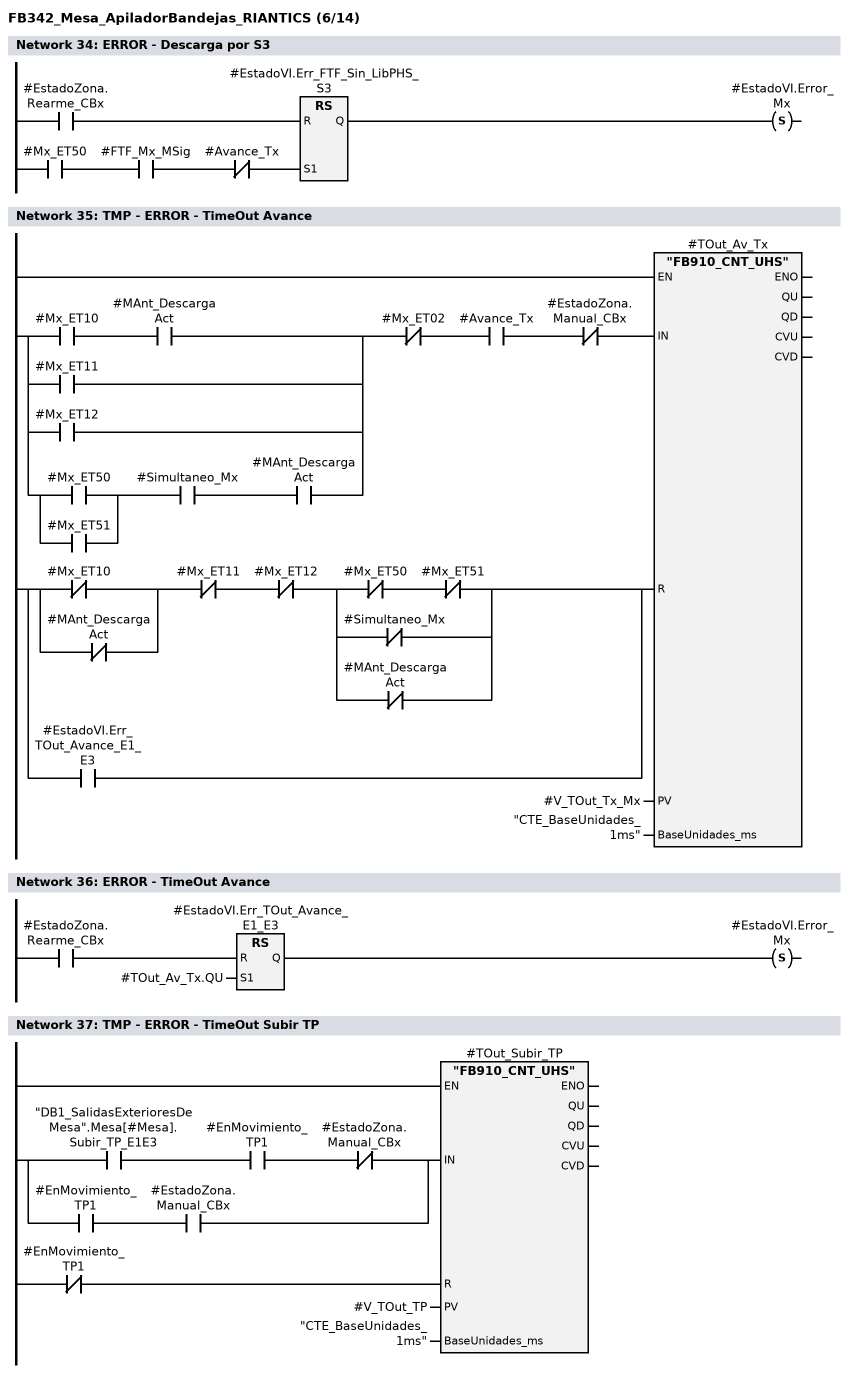
   RUNG wire#powerrail
      Contact( #EstadoZona.Rearme_CBx )
      S_RS(operand := #EstadoVI.Err_FTF_Sin_LibPHS_S3, s1 := wire#w1)
      S_Coil( #EstadoVI.Error_Mx )
   END_RUNG
   RUNG wire#powerrail
      Contact( #Mx_ET50 )
      Contact( #FTF_Mx_MSig )
      I_Contact( #Avance_Tx )
   END_RUNG wire#w1
   // the same network as SCL:
   IF #EstadoZona.Rearme_CBx THEN
       #EstadoVI.Err_FTF_Sin_LibPHS_S3 := FALSE;   // RS flip-flop
   END_IF;
   IF #Mx_ET50 AND #FTF_Mx_MSig AND NOT #Avance_Tx THEN #EstadoVI.Err_FTF_Sin_LibPHS_S3 := TRUE; END_IF;
   IF #EstadoVI.Err_FTF_Sin_LibPHS_S3 THEN #EstadoVI.Error_Mx := TRUE; END_IF;
END_REGION

REGION Network 35: TMP - ERROR - TimeOut Avance
   RUNG wire#powerrail
      #TOut_Av_Tx(IN := wire#w3, R := wire#w6, PV := #V_TOut_Tx_Mx, BaseUnidades_ms := "CTE_BaseUnidades_1ms", QU =>, QD =>, CVU =>, CVD =>)
   END_RUNG
   RUNG wire#powerrail
      Contact( #Mx_ET10 )
      Contact( #MAnt_DescargaAct )
      wire#w1
      I_Contact( #Mx_ET02 )
      Contact( #Avance_Tx )
      I_Contact( #EstadoZona.Manual_CBx )
   END_RUNG wire#w3
   RUNG wire#powerrail
      Contact( #Mx_ET11 )
   END_RUNG wire#w1
   RUNG wire#powerrail
      Contact( #Mx_ET12 )
   END_RUNG wire#w1
   RUNG wire#powerrail
      Contact( #Mx_ET50 )
      wire#w2
      Contact( #Simultaneo_Mx )
      Contact( #MAnt_DescargaAct )
   END_RUNG wire#w1
   RUNG wire#powerrail
      Contact( #Mx_ET51 )
   END_RUNG wire#w2
   RUNG wire#powerrail
      I_Contact( #Mx_ET10 )
      wire#w4
      I_Contact( #Mx_ET11 )
      I_Contact( #Mx_ET12 )
      wire#w5
      I_Contact( #Mx_ET50 )
      I_Contact( #Mx_ET51 )
   END_RUNG wire#w6
   RUNG wire#powerrail
      I_Contact( #MAnt_DescargaAct )
   END_RUNG wire#w4
   RUNG wire#w5
      I_Contact( #Simultaneo_Mx )
   END_RUNG wire#w6
   RUNG wire#w5
      I_Contact( #MAnt_DescargaAct )
   END_RUNG wire#w6
   RUNG wire#powerrail
      Contact( #EstadoVI.Err_TOut_Avance_E1_E3 )
   END_RUNG wire#w6
   // the same network as SCL:
   #TOut_Av_Tx(IN := ((#Mx_ET10 AND #MAnt_DescargaAct) OR #Mx_ET11 OR #Mx_ET12 OR ((#Mx_ET50 OR #Mx_ET51) AND #Simultaneo_Mx AND #MAnt_DescargaAct)) AND NOT #Mx_ET02 AND #Avance_Tx AND NOT #EstadoZona.Manual_CBx,   // "FB910_CNT_UHS"
               R := ((NOT #Mx_ET10 OR NOT #MAnt_DescargaAct) AND NOT #Mx_ET11 AND NOT #Mx_ET12 AND ((NOT #Mx_ET50 AND NOT #Mx_ET51) OR NOT #Simultaneo_Mx OR NOT #MAnt_DescargaAct)) OR #EstadoVI.Err_TOut_Avance_E1_E3,
               PV := #V_TOut_Tx_Mx,
               BaseUnidades_ms := "CTE_BaseUnidades_1ms");
END_REGION

REGION Network 36: ERROR - TimeOut Avance
   RUNG wire#powerrail
      Contact( #EstadoZona.Rearme_CBx )
      S_RS(operand := #EstadoVI.Err_TOut_Avance_E1_E3, s1 := #TOut_Av_Tx.QU)
      S_Coil( #EstadoVI.Error_Mx )
   END_RUNG
   // the same network as SCL:
   IF #EstadoZona.Rearme_CBx THEN
       #EstadoVI.Err_TOut_Avance_E1_E3 := FALSE;   // RS flip-flop
   END_IF;
   IF #TOut_Av_Tx.QU THEN #EstadoVI.Err_TOut_Avance_E1_E3 := TRUE; END_IF;
   IF #EstadoVI.Err_TOut_Avance_E1_E3 THEN #EstadoVI.Error_Mx := TRUE; END_IF;
END_REGION

REGION Network 37: TMP - ERROR - TimeOut Subir TP
   RUNG wire#powerrail
      #TOut_Subir_TP(IN := wire#w1, R := wire#w2, PV := #V_TOut_TP, BaseUnidades_ms := "CTE_BaseUnidades_1ms", QU =>, QD =>, CVU =>, CVD =>)
   END_RUNG
   RUNG wire#powerrail
      Contact( "DB1_SalidasExterioresDeMesa".Mesa[#Mesa].Subir_TP_E1E3 )
      Contact( #EnMovimiento_TP1 )
      I_Contact( #EstadoZona.Manual_CBx )
   END_RUNG wire#w1
   RUNG wire#powerrail
      Contact( #EnMovimiento_TP1 )
      Contact( #EstadoZona.Manual_CBx )
   END_RUNG wire#w1
   RUNG wire#powerrail
      I_Contact( #EnMovimiento_TP1 )
   END_RUNG wire#w2
   // the same network as SCL:
   #TOut_Subir_TP(IN := ("DB1_SalidasExterioresDeMesa".Mesa[#Mesa].Subir_TP_E1E3 AND #EnMovimiento_TP1 AND NOT #EstadoZona.Manual_CBx) OR (#EnMovimiento_TP1 AND #EstadoZona.Manual_CBx),   // "FB910_CNT_UHS"
                  R := NOT #EnMovimiento_TP1,
                  PV := #V_TOut_TP,
                  BaseUnidades_ms := "CTE_BaseUnidades_1ms");
END_REGION

REGION Network 38: ERROR - TimeOut Subir TP
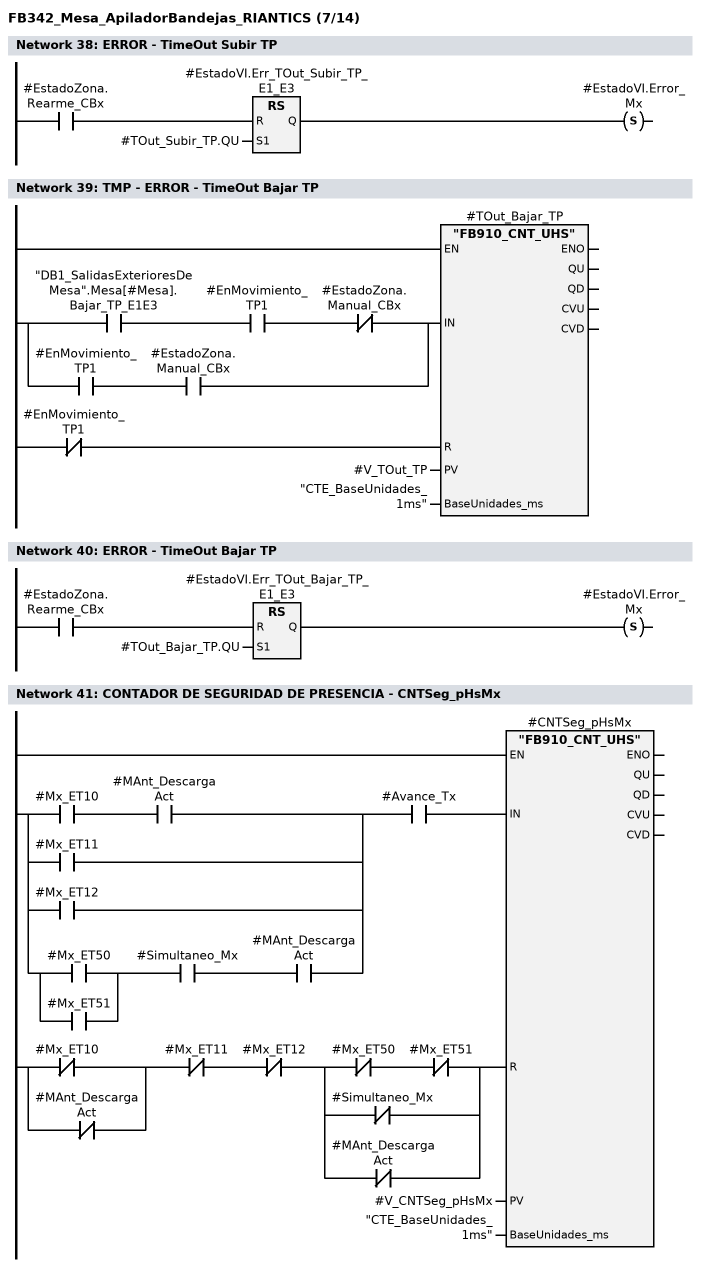
   RUNG wire#powerrail
      Contact( #EstadoZona.Rearme_CBx )
      S_RS(operand := #EstadoVI.Err_TOut_Subir_TP_E1_E3, s1 := #TOut_Subir_TP.QU)
      S_Coil( #EstadoVI.Error_Mx )
   END_RUNG
   // the same network as SCL:
   IF #EstadoZona.Rearme_CBx THEN
       #EstadoVI.Err_TOut_Subir_TP_E1_E3 := FALSE;   // RS flip-flop
   END_IF;
   IF #TOut_Subir_TP.QU THEN #EstadoVI.Err_TOut_Subir_TP_E1_E3 := TRUE; END_IF;
   IF #EstadoVI.Err_TOut_Subir_TP_E1_E3 THEN #EstadoVI.Error_Mx := TRUE; END_IF;
END_REGION

REGION Network 39: TMP - ERROR - TimeOut Bajar TP
   RUNG wire#powerrail
      #TOut_Bajar_TP(IN := wire#w1, R := wire#w2, PV := #V_TOut_TP, BaseUnidades_ms := "CTE_BaseUnidades_1ms", QU =>, QD =>, CVU =>, CVD =>)
   END_RUNG
   RUNG wire#powerrail
      Contact( "DB1_SalidasExterioresDeMesa".Mesa[#Mesa].Bajar_TP_E1E3 )
      Contact( #EnMovimiento_TP1 )
      I_Contact( #EstadoZona.Manual_CBx )
   END_RUNG wire#w1
   RUNG wire#powerrail
      Contact( #EnMovimiento_TP1 )
      Contact( #EstadoZona.Manual_CBx )
   END_RUNG wire#w1
   RUNG wire#powerrail
      I_Contact( #EnMovimiento_TP1 )
   END_RUNG wire#w2
   // the same network as SCL:
   #TOut_Bajar_TP(IN := ("DB1_SalidasExterioresDeMesa".Mesa[#Mesa].Bajar_TP_E1E3 AND #EnMovimiento_TP1 AND NOT #EstadoZona.Manual_CBx) OR (#EnMovimiento_TP1 AND #EstadoZona.Manual_CBx),   // "FB910_CNT_UHS"
                  R := NOT #EnMovimiento_TP1,
                  PV := #V_TOut_TP,
                  BaseUnidades_ms := "CTE_BaseUnidades_1ms");
END_REGION

REGION Network 40: ERROR - TimeOut Bajar TP
   RUNG wire#powerrail
      Contact( #EstadoZona.Rearme_CBx )
      S_RS(operand := #EstadoVI.Err_TOut_Bajar_TP_E1_E3, s1 := #TOut_Bajar_TP.QU)
      S_Coil( #EstadoVI.Error_Mx )
   END_RUNG
   // the same network as SCL:
   IF #EstadoZona.Rearme_CBx THEN
       #EstadoVI.Err_TOut_Bajar_TP_E1_E3 := FALSE;   // RS flip-flop
   END_IF;
   IF #TOut_Bajar_TP.QU THEN #EstadoVI.Err_TOut_Bajar_TP_E1_E3 := TRUE; END_IF;
   IF #EstadoVI.Err_TOut_Bajar_TP_E1_E3 THEN #EstadoVI.Error_Mx := TRUE; END_IF;
END_REGION

REGION Network 41: CONTADOR DE SEGURIDAD DE PRESENCIA - CNTSeg_pHsMx
   RUNG wire#powerrail
      #CNTSeg_pHsMx(IN := wire#w3, R := wire#w6, PV := #V_CNTSeg_pHsMx, BaseUnidades_ms := "CTE_BaseUnidades_1ms", QU =>, QD =>, CVU =>, CVD =>)
   END_RUNG
   RUNG wire#powerrail
      Contact( #Mx_ET10 )
      Contact( #MAnt_DescargaAct )
      wire#w1
      Contact( #Avance_Tx )
   END_RUNG wire#w3
   RUNG wire#powerrail
      Contact( #Mx_ET11 )
   END_RUNG wire#w1
   RUNG wire#powerrail
      Contact( #Mx_ET12 )
   END_RUNG wire#w1
   RUNG wire#powerrail
      Contact( #Mx_ET50 )
      wire#w2
      Contact( #Simultaneo_Mx )
      Contact( #MAnt_DescargaAct )
   END_RUNG wire#w1
   RUNG wire#powerrail
      Contact( #Mx_ET51 )
   END_RUNG wire#w2
   RUNG wire#powerrail
      I_Contact( #Mx_ET10 )
      wire#w4
      I_Contact( #Mx_ET11 )
      I_Contact( #Mx_ET12 )
      wire#w5
      I_Contact( #Mx_ET50 )
      I_Contact( #Mx_ET51 )
   END_RUNG wire#w6
   RUNG wire#powerrail
      I_Contact( #MAnt_DescargaAct )
   END_RUNG wire#w4
   RUNG wire#w5
      I_Contact( #Simultaneo_Mx )
   END_RUNG wire#w6
   RUNG wire#w5
      I_Contact( #MAnt_DescargaAct )
   END_RUNG wire#w6
   // the same network as SCL:
   #CNTSeg_pHsMx(IN := ((#Mx_ET10 AND #MAnt_DescargaAct) OR #Mx_ET11 OR #Mx_ET12 OR ((#Mx_ET50 OR #Mx_ET51) AND #Simultaneo_Mx AND #MAnt_DescargaAct)) AND #Avance_Tx,   // "FB910_CNT_UHS"
                 R := (NOT #Mx_ET10 OR NOT #MAnt_DescargaAct) AND NOT #Mx_ET11 AND NOT #Mx_ET12 AND ((NOT #Mx_ET50 AND NOT #Mx_ET51) OR NOT #Simultaneo_Mx OR NOT #MAnt_DescargaAct),
                 PV := #V_CNTSeg_pHsMx,
                 BaseUnidades_ms := "CTE_BaseUnidades_1ms");
END_REGION

REGION Network 42: CONTADOR DE PRESENCIA - CNT_pHsMx
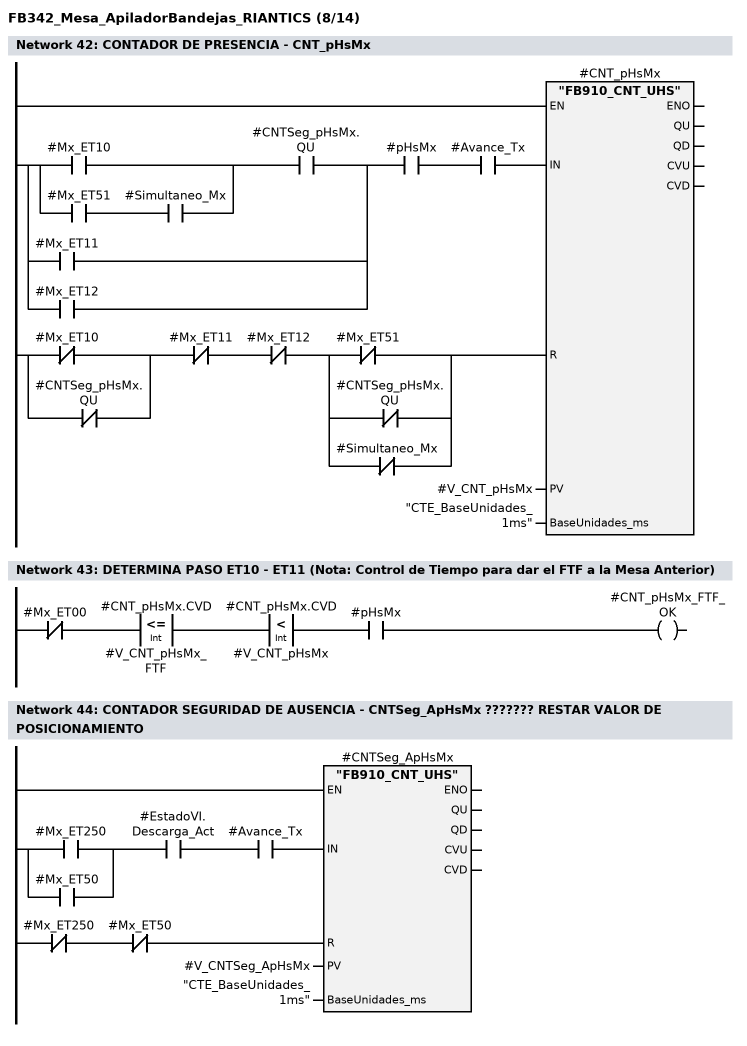
   RUNG wire#powerrail
      #CNT_pHsMx(IN := wire#w3, R := wire#w6, PV := #V_CNT_pHsMx, BaseUnidades_ms := "CTE_BaseUnidades_1ms", QU =>, QD =>, CVU =>, CVD =>)
   END_RUNG
   RUNG wire#powerrail
      Contact( #Mx_ET10 )
      wire#w1
      Contact( #CNTSeg_pHsMx.QU )
      wire#w2
      Contact( #pHsMx )
      Contact( #Avance_Tx )
   END_RUNG wire#w3
   RUNG wire#powerrail
      Contact( #Mx_ET51 )
      Contact( #Simultaneo_Mx )
   END_RUNG wire#w1
   RUNG wire#powerrail
      Contact( #Mx_ET11 )
   END_RUNG wire#w2
   RUNG wire#powerrail
      Contact( #Mx_ET12 )
   END_RUNG wire#w2
   RUNG wire#powerrail
      I_Contact( #Mx_ET10 )
      wire#w4
      I_Contact( #Mx_ET11 )
      I_Contact( #Mx_ET12 )
      wire#w5
      I_Contact( #Mx_ET51 )
   END_RUNG wire#w6
   RUNG wire#powerrail
      I_Contact( #CNTSeg_pHsMx.QU )
   END_RUNG wire#w4
   RUNG wire#w5
      I_Contact( #CNTSeg_pHsMx.QU )
   END_RUNG wire#w6
   RUNG wire#w5
      I_Contact( #Simultaneo_Mx )
   END_RUNG wire#w6
   // the same network as SCL:
   #CNT_pHsMx(IN := (((#Mx_ET10 OR (#Mx_ET51 AND #Simultaneo_Mx)) AND #CNTSeg_pHsMx.QU) OR #Mx_ET11 OR #Mx_ET12) AND #pHsMx AND #Avance_Tx,   // "FB910_CNT_UHS"
              R := (NOT #Mx_ET10 OR NOT #CNTSeg_pHsMx.QU) AND NOT #Mx_ET11 AND NOT #Mx_ET12 AND (NOT #Mx_ET51 OR NOT #CNTSeg_pHsMx.QU OR NOT #Simultaneo_Mx),
              PV := #V_CNT_pHsMx,
              BaseUnidades_ms := "CTE_BaseUnidades_1ms");
END_REGION

REGION Network 43: DETERMINA PASO ET10 - ET11 (Nota: Control de Tiempo para dar el FTF a la Mesa Anterior)
   RUNG wire#powerrail
      I_Contact( #Mx_ET00 )
      { S7_Templates := "SrcType := Int" } LE_Contact(in1 := #CNT_pHsMx.CVD, in2 := #V_CNT_pHsMx_FTF)
      { S7_Templates := "SrcType := Int" } LT_Contact(in1 := #CNT_pHsMx.CVD, in2 := #V_CNT_pHsMx)
      Contact( #pHsMx )
      Coil( #CNT_pHsMx_FTF_OK )
   END_RUNG
   // the same network as SCL:
   #CNT_pHsMx_FTF_OK := NOT #Mx_ET00 AND (#CNT_pHsMx.CVD <= #V_CNT_pHsMx_FTF) AND (#CNT_pHsMx.CVD < #V_CNT_pHsMx) AND #pHsMx;
END_REGION

REGION Network 44: CONTADOR SEGURIDAD DE AUSENCIA - CNTSeg_ApHsMx ??????? RESTAR VALOR DE POSICIONAMIENTO
   RUNG wire#powerrail
      #CNTSeg_ApHsMx(IN := wire#w2, R := wire#w3, PV := #V_CNTSeg_ApHsMx, BaseUnidades_ms := "CTE_BaseUnidades_1ms", QU =>, QD =>, CVU =>, CVD =>)
   END_RUNG
   RUNG wire#powerrail
      Contact( #Mx_ET250 )
      wire#w1
      Contact( #EstadoVI.Descarga_Act )
      Contact( #Avance_Tx )
   END_RUNG wire#w2
   RUNG wire#powerrail
      Contact( #Mx_ET50 )
   END_RUNG wire#w1
   RUNG wire#powerrail
      I_Contact( #Mx_ET250 )
      I_Contact( #Mx_ET50 )
   END_RUNG wire#w3
   // the same network as SCL:
   #CNTSeg_ApHsMx(IN := (#Mx_ET250 OR #Mx_ET50) AND #EstadoVI.Descarga_Act AND #Avance_Tx,   // "FB910_CNT_UHS"
                  R := NOT #Mx_ET250 AND NOT #Mx_ET50,
                  PV := #V_CNTSeg_ApHsMx,
                  BaseUnidades_ms := "CTE_BaseUnidades_1ms");
END_REGION

REGION Network 45: CONTADOR DE LA AUSENCIA - CNT_ApHsMX
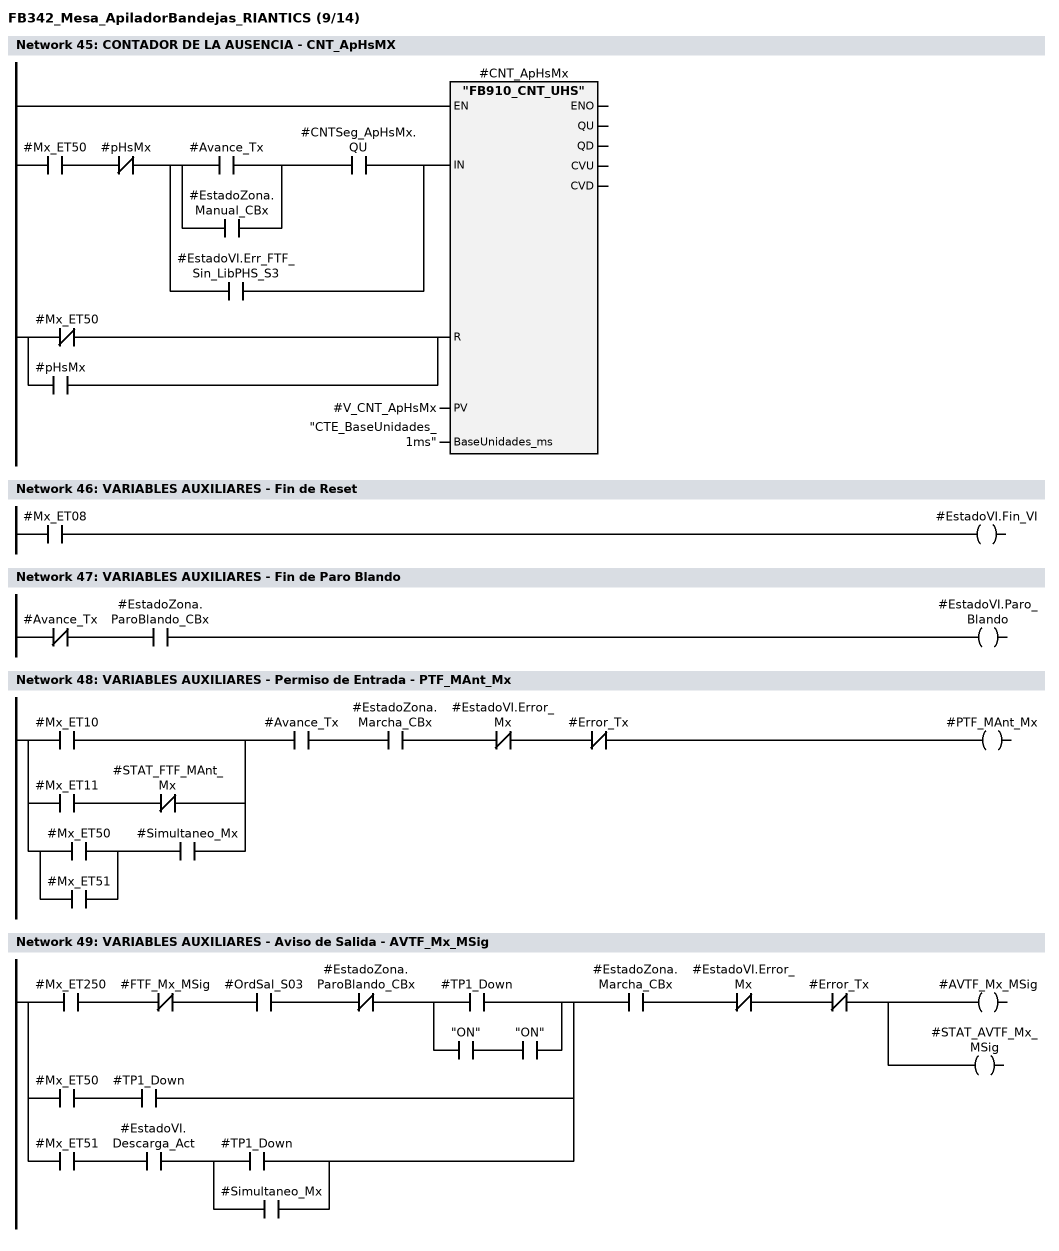
   RUNG wire#powerrail
      #CNT_ApHsMx(IN := wire#w3, R := wire#w4, PV := #V_CNT_ApHsMx, BaseUnidades_ms := "CTE_BaseUnidades_1ms", QU =>, QD =>, CVU =>, CVD =>)
   END_RUNG
   RUNG wire#powerrail
      Contact( #Mx_ET50 )
      I_Contact( #pHsMx )
      wire#w1
      Contact( #Avance_Tx )
      wire#w2
      Contact( #CNTSeg_ApHsMx.QU )
   END_RUNG wire#w3
   RUNG wire#w1
      Contact( #EstadoZona.Manual_CBx )
   END_RUNG wire#w2
   RUNG wire#w1
      Contact( #EstadoVI.Err_FTF_Sin_LibPHS_S3 )
   END_RUNG wire#w3
   RUNG wire#powerrail
      I_Contact( #Mx_ET50 )
   END_RUNG wire#w4
   RUNG wire#powerrail
      Contact( #pHsMx )
   END_RUNG wire#w4
   // the same network as SCL:
   #CNT_ApHsMx(IN := #Mx_ET50 AND NOT #pHsMx AND (((#Avance_Tx OR #EstadoZona.Manual_CBx) AND #CNTSeg_ApHsMx.QU) OR #EstadoVI.Err_FTF_Sin_LibPHS_S3),   // "FB910_CNT_UHS"
               R := NOT #Mx_ET50 OR #pHsMx,
               PV := #V_CNT_ApHsMx,
               BaseUnidades_ms := "CTE_BaseUnidades_1ms");
END_REGION

REGION Network 46: VARIABLES AUXILIARES - Fin de Reset
   RUNG wire#powerrail
      Contact( #Mx_ET08 )
      Coil( #EstadoVI.Fin_VI )
   END_RUNG
   // the same network as SCL:
   #EstadoVI.Fin_VI := #Mx_ET08;
END_REGION

REGION Network 47: VARIABLES AUXILIARES - Fin de Paro Blando
   RUNG wire#powerrail
      I_Contact( #Avance_Tx )
      Contact( #EstadoZona.ParoBlando_CBx )
      Coil( #EstadoVI.Paro_Blando )
   END_RUNG
   // the same network as SCL:
   #EstadoVI.Paro_Blando := NOT #Avance_Tx AND #EstadoZona.ParoBlando_CBx;
END_REGION

REGION Network 48: VARIABLES AUXILIARES - Permiso de Entrada - PTF_MAnt_Mx
   RUNG wire#powerrail
      Contact( #Mx_ET10 )
      wire#w1
      Contact( #Avance_Tx )
      Contact( #EstadoZona.Marcha_CBx )
      I_Contact( #EstadoVI.Error_Mx )
      I_Contact( #Error_Tx )
      Coil( #PTF_MAnt_Mx )
   END_RUNG
   RUNG wire#powerrail
      Contact( #Mx_ET11 )
      I_Contact( #STAT_FTF_MAnt_Mx )
   END_RUNG wire#w1
   RUNG wire#powerrail
      Contact( #Mx_ET50 )
      wire#w2
      Contact( #Simultaneo_Mx )
   END_RUNG wire#w1
   RUNG wire#powerrail
      Contact( #Mx_ET51 )
   END_RUNG wire#w2
   // the same network as SCL:
   #PTF_MAnt_Mx := (#Mx_ET10 OR (#Mx_ET11 AND NOT #STAT_FTF_MAnt_Mx) OR ((#Mx_ET50 OR #Mx_ET51) AND #Simultaneo_Mx)) AND #Avance_Tx AND #EstadoZona.Marcha_CBx AND NOT #EstadoVI.Error_Mx AND NOT #Error_Tx;
END_REGION

REGION Network 49: VARIABLES AUXILIARES - Aviso de Salida - AVTF_Mx_MSig
   RUNG wire#powerrail
      Contact( #Mx_ET250 )
      I_Contact( #FTF_Mx_MSig )
      Contact( #OrdSal_S03 )
      I_Contact( #EstadoZona.ParoBlando_CBx )
      wire#w1
      Contact( #TP1_Down )
      wire#w2
      Contact( #EstadoZona.Marcha_CBx )
      I_Contact( #EstadoVI.Error_Mx )
      I_Contact( #Error_Tx )
      wire#w4
      Coil( #AVTF_Mx_MSig )
   END_RUNG
   RUNG wire#w1
      Contact( "ON" )
      Contact( "ON" )
   END_RUNG wire#w2
   RUNG wire#powerrail
      Contact( #Mx_ET50 )
      Contact( #TP1_Down )
   END_RUNG wire#w2
   RUNG wire#powerrail
      Contact( #Mx_ET51 )
      Contact( #EstadoVI.Descarga_Act )
      wire#w3
      Contact( #TP1_Down )
   END_RUNG wire#w2
   RUNG wire#w3
      Contact( #Simultaneo_Mx )
   END_RUNG wire#w2
   RUNG wire#w4
      Coil( #STAT_AVTF_Mx_MSig )
   END_RUNG
   // the same network as SCL:
   #AVTF_Mx_MSig := ((#Mx_ET250 AND NOT #FTF_Mx_MSig AND #OrdSal_S03 AND NOT #EstadoZona.ParoBlando_CBx AND (#TP1_Down OR ("ON" AND "ON"))) OR (#Mx_ET50 AND #TP1_Down) OR (#Mx_ET51 AND #EstadoVI.Descarga_Act AND (#TP1_Down OR #Simultaneo_Mx))) AND #EstadoZona.Marcha_CBx AND NOT #EstadoVI.Error_Mx AND NOT #Error_Tx;
   #STAT_AVTF_Mx_MSig := #AVTF_Mx_MSig;
END_REGION

REGION Network 50: VARIABLES AUXILIARES - P_Mens_Mx_MSig (Nota: solo en ET51)
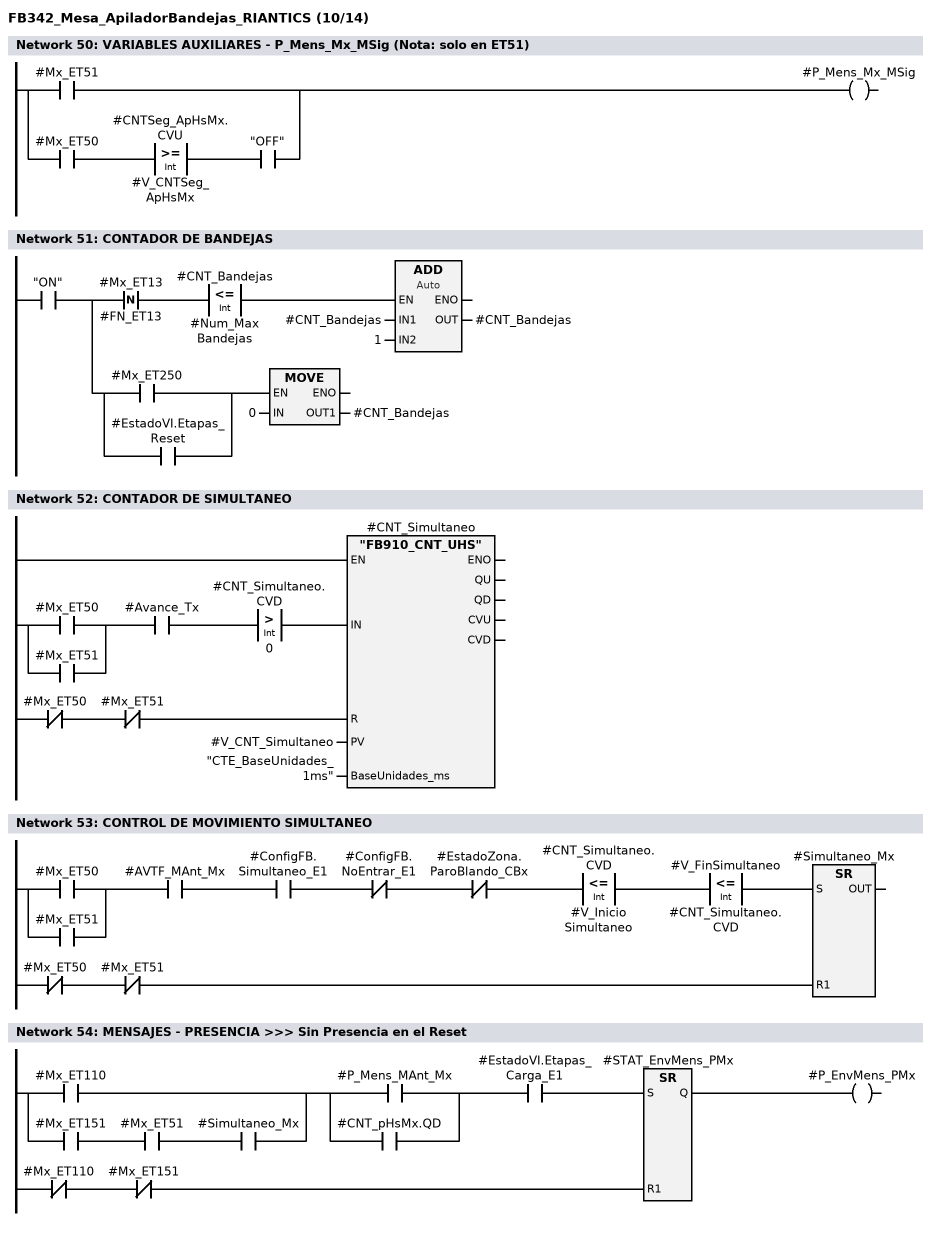
   RUNG wire#powerrail
      Contact( #Mx_ET51 )
      wire#w1
      Coil( #P_Mens_Mx_MSig )
   END_RUNG
   RUNG wire#powerrail
      Contact( #Mx_ET50 )
      { S7_Templates := "SrcType := Int" } GE_Contact(in1 := #CNTSeg_ApHsMx.CVU, in2 := #V_CNTSeg_ApHsMx)
      Contact( "OFF" )
   END_RUNG wire#w1
   // the same network as SCL:
   #P_Mens_Mx_MSig := #Mx_ET51 OR (#Mx_ET50 AND (#CNTSeg_ApHsMx.CVU >= #V_CNTSeg_ApHsMx) AND "OFF");
END_REGION

REGION Network 51: CONTADOR DE BANDEJAS
   RUNG wire#powerrail
      Contact( "ON" )
      wire#w1
      N_Contact(operand := #Mx_ET13, bit := #FN_ET13)
      { S7_Templates := "SrcType := Int" } LE_Contact(in1 := #CNT_Bandejas, in2 := #Num_MaxBandejas)
      Add(in1 := #CNT_Bandejas, in2 := 1, out => #CNT_Bandejas)
   END_RUNG
   RUNG wire#w1
      Contact( #Mx_ET250 )
      wire#w2
      Move(in := 0, out1 => #CNT_Bandejas)
   END_RUNG
   RUNG wire#w1
      Contact( #EstadoVI.Etapas_Reset )
   END_RUNG wire#w2
   // the same network as SCL:
   #_w1 := "ON" AND NOT #Mx_ET13 AND #FN_ET13;   // falling edge of #Mx_ET13
   #FN_ET13 := #Mx_ET13;
   IF #_w1 AND (#CNT_Bandejas <= #Num_MaxBandejas) THEN #CNT_Bandejas := #CNT_Bandejas + 1; END_IF;
   IF "ON" AND (#Mx_ET250 OR #EstadoVI.Etapas_Reset) THEN #CNT_Bandejas := 0; END_IF;
END_REGION

REGION Network 52: CONTADOR DE SIMULTANEO
   RUNG wire#powerrail
      #CNT_Simultaneo(IN := wire#w2, R := wire#w3, PV := #V_CNT_Simultaneo, BaseUnidades_ms := "CTE_BaseUnidades_1ms", QU =>, QD =>, CVU =>, CVD =>)
   END_RUNG
   RUNG wire#powerrail
      Contact( #Mx_ET50 )
      wire#w1
      Contact( #Avance_Tx )
      { S7_Templates := "SrcType := Int" } GT_Contact(in1 := #CNT_Simultaneo.CVD, in2 := 0)
   END_RUNG wire#w2
   RUNG wire#powerrail
      Contact( #Mx_ET51 )
   END_RUNG wire#w1
   RUNG wire#powerrail
      I_Contact( #Mx_ET50 )
      I_Contact( #Mx_ET51 )
   END_RUNG wire#w3
   // the same network as SCL:
   #CNT_Simultaneo(IN := (#Mx_ET50 OR #Mx_ET51) AND #Avance_Tx AND (#CNT_Simultaneo.CVD > 0),   // "FB910_CNT_UHS"
                   R := NOT #Mx_ET50 AND NOT #Mx_ET51,
                   PV := #V_CNT_Simultaneo,
                   BaseUnidades_ms := "CTE_BaseUnidades_1ms");
END_REGION

REGION Network 53: CONTROL DE MOVIMIENTO SIMULTANEO
   RUNG wire#powerrail
      Contact( #Mx_ET50 )
      wire#w1
      Contact( #AVTF_MAnt_Mx )
      Contact( #ConfigFB.Simultaneo_E1 )
      I_Contact( #ConfigFB.NoEntrar_E1 )
      I_Contact( #EstadoZona.ParoBlando_CBx )
      { S7_Templates := "SrcType := Int" } LE_Contact(in1 := #CNT_Simultaneo.CVD, in2 := #V_InicioSimultaneo)
      { S7_Templates := "SrcType := Int" } LE_Contact(in1 := #V_FinSimultaneo, in2 := #CNT_Simultaneo.CVD)
      S_SR(operand := #Simultaneo_Mx, r1 := wire#w2)
   END_RUNG
   RUNG wire#powerrail
      Contact( #Mx_ET51 )
   END_RUNG wire#w1
   RUNG wire#powerrail
      I_Contact( #Mx_ET50 )
      I_Contact( #Mx_ET51 )
   END_RUNG wire#w2
   // the same network as SCL:
   IF (#Mx_ET50 OR #Mx_ET51) AND #AVTF_MAnt_Mx AND #ConfigFB.Simultaneo_E1 AND NOT #ConfigFB.NoEntrar_E1 AND NOT #EstadoZona.ParoBlando_CBx AND (#CNT_Simultaneo.CVD <= #V_InicioSimultaneo) AND (#V_FinSimultaneo <= #CNT_Simultaneo.CVD) THEN
       #Simultaneo_Mx := TRUE;   // SR flip-flop
   END_IF;
   IF NOT #Mx_ET50 AND NOT #Mx_ET51 THEN #Simultaneo_Mx := FALSE; END_IF;
END_REGION

REGION Network 54: MENSAJES - PRESENCIA >>> Sin Presencia en el Reset
   RUNG wire#powerrail
      Contact( #Mx_ET110 )
      wire#w1
      Contact( #P_Mens_MAnt_Mx )
      wire#w2
      Contact( #EstadoVI.Etapas_Carga_E1 )
      S_SR(operand := #STAT_EnvMens_PMx, r1 := wire#w3)
      Coil( #P_EnvMens_PMx )
   END_RUNG
   RUNG wire#powerrail
      Contact( #Mx_ET151 )
      Contact( #Mx_ET51 )
      Contact( #Simultaneo_Mx )
   END_RUNG wire#w1
   RUNG wire#w1
      Contact( #CNT_pHsMx.QD )
   END_RUNG wire#w2
   RUNG wire#powerrail
      I_Contact( #Mx_ET110 )
      I_Contact( #Mx_ET151 )
   END_RUNG wire#w3
   // the same network as SCL:
   IF (#Mx_ET110 OR (#Mx_ET151 AND #Mx_ET51 AND #Simultaneo_Mx)) AND (#P_Mens_MAnt_Mx OR #CNT_pHsMx.QD) AND #EstadoVI.Etapas_Carga_E1 THEN
       #STAT_EnvMens_PMx := TRUE;   // SR flip-flop
   END_IF;
   IF NOT #Mx_ET110 AND NOT #Mx_ET151 THEN #STAT_EnvMens_PMx := FALSE; END_IF;
   #P_EnvMens_PMx := #STAT_EnvMens_PMx;
END_REGION

REGION Network 55: MENSAJES - PROTOCOLO INICIADO
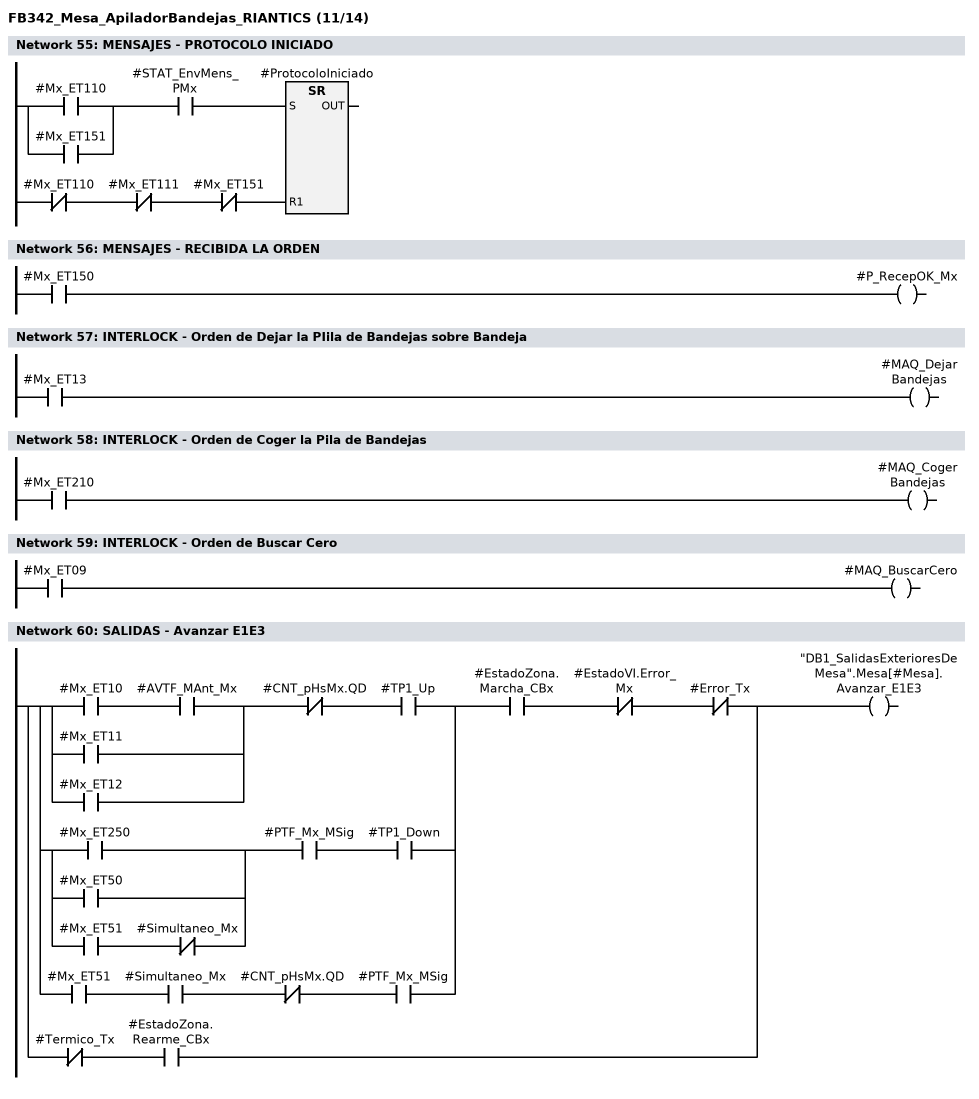
   RUNG wire#powerrail
      Contact( #Mx_ET110 )
      wire#w1
      Contact( #STAT_EnvMens_PMx )
      S_SR(operand := #ProtocoloIniciado, r1 := wire#w2)
   END_RUNG
   RUNG wire#powerrail
      Contact( #Mx_ET151 )
   END_RUNG wire#w1
   RUNG wire#powerrail
      I_Contact( #Mx_ET110 )
      I_Contact( #Mx_ET111 )
      I_Contact( #Mx_ET151 )
   END_RUNG wire#w2
   // the same network as SCL:
   IF (#Mx_ET110 OR #Mx_ET151) AND #STAT_EnvMens_PMx THEN
       #ProtocoloIniciado := TRUE;   // SR flip-flop
   END_IF;
   IF NOT #Mx_ET110 AND NOT #Mx_ET111 AND NOT #Mx_ET151 THEN #ProtocoloIniciado := FALSE; END_IF;
END_REGION

REGION Network 56: MENSAJES - RECIBIDA LA ORDEN
   RUNG wire#powerrail
      Contact( #Mx_ET150 )
      Coil( #P_RecepOK_Mx )
   END_RUNG
   // the same network as SCL:
   #P_RecepOK_Mx := #Mx_ET150;
END_REGION

REGION Network 57: INTERLOCK - Orden de Dejar la PIila de Bandejas sobre Bandeja
   RUNG wire#powerrail
      Contact( #Mx_ET13 )
      Coil( #MAQ_DejarBandejas )
   END_RUNG
   // the same network as SCL:
   #MAQ_DejarBandejas := #Mx_ET13;
END_REGION

REGION Network 58: INTERLOCK - Orden de Coger la Pila de Bandejas
   RUNG wire#powerrail
      Contact( #Mx_ET210 )
      Coil( #MAQ_CogerBandejas )
   END_RUNG
   // the same network as SCL:
   #MAQ_CogerBandejas := #Mx_ET210;
END_REGION

REGION Network 59: INTERLOCK - Orden de Buscar Cero
   RUNG wire#powerrail
      Contact( #Mx_ET09 )
      Coil( #MAQ_BuscarCero )
   END_RUNG
   // the same network as SCL:
   #MAQ_BuscarCero := #Mx_ET09;
END_REGION

REGION Network 60: SALIDAS - Avanzar E1E3
   RUNG wire#powerrail
      Contact( #Mx_ET10 )
      Contact( #AVTF_MAnt_Mx )
      wire#w1
      I_Contact( #CNT_pHsMx.QD )
      Contact( #TP1_Up )
      wire#w2
      Contact( #EstadoZona.Marcha_CBx )
      I_Contact( #EstadoVI.Error_Mx )
      I_Contact( #Error_Tx )
      wire#w4
      Coil( "DB1_SalidasExterioresDeMesa".Mesa[#Mesa].Avanzar_E1E3 )
   END_RUNG
   RUNG wire#powerrail
      Contact( #Mx_ET11 )
   END_RUNG wire#w1
   RUNG wire#powerrail
      Contact( #Mx_ET12 )
   END_RUNG wire#w1
   RUNG wire#powerrail
      Contact( #Mx_ET250 )
      wire#w3
      Contact( #PTF_Mx_MSig )
      Contact( #TP1_Down )
   END_RUNG wire#w2
   RUNG wire#powerrail
      Contact( #Mx_ET50 )
   END_RUNG wire#w3
   RUNG wire#powerrail
      Contact( #Mx_ET51 )
      I_Contact( #Simultaneo_Mx )
   END_RUNG wire#w3
   RUNG wire#powerrail
      Contact( #Mx_ET51 )
      Contact( #Simultaneo_Mx )
      I_Contact( #CNT_pHsMx.QD )
      Contact( #PTF_Mx_MSig )
   END_RUNG wire#w2
   RUNG wire#powerrail
      I_Contact( #Termico_Tx )
      Contact( #EstadoZona.Rearme_CBx )
   END_RUNG wire#w4
   // the same network as SCL:
   "DB1_SalidasExterioresDeMesa".Mesa[#Mesa].Avanzar_E1E3 := (((((#Mx_ET10 AND #AVTF_MAnt_Mx) OR #Mx_ET11 OR #Mx_ET12) AND NOT #CNT_pHsMx.QD AND #TP1_Up) OR ((#Mx_ET250 OR #Mx_ET50 OR (#Mx_ET51 AND NOT #Simultaneo_Mx)) AND #PTF_Mx_MSig AND #TP1_Down) OR (#Mx_ET51 AND #Simultaneo_Mx AND NOT #CNT_pHsMx.QD AND #PTF_Mx_MSig)) AND #EstadoZona.Marcha_CBx AND NOT #EstadoVI.Error_Mx AND NOT #Error_Tx) OR (NOT #Termico_Tx AND #EstadoZona.Rearme_CBx);
END_REGION

REGION Network 61: SALIDAS - Parar E1E3
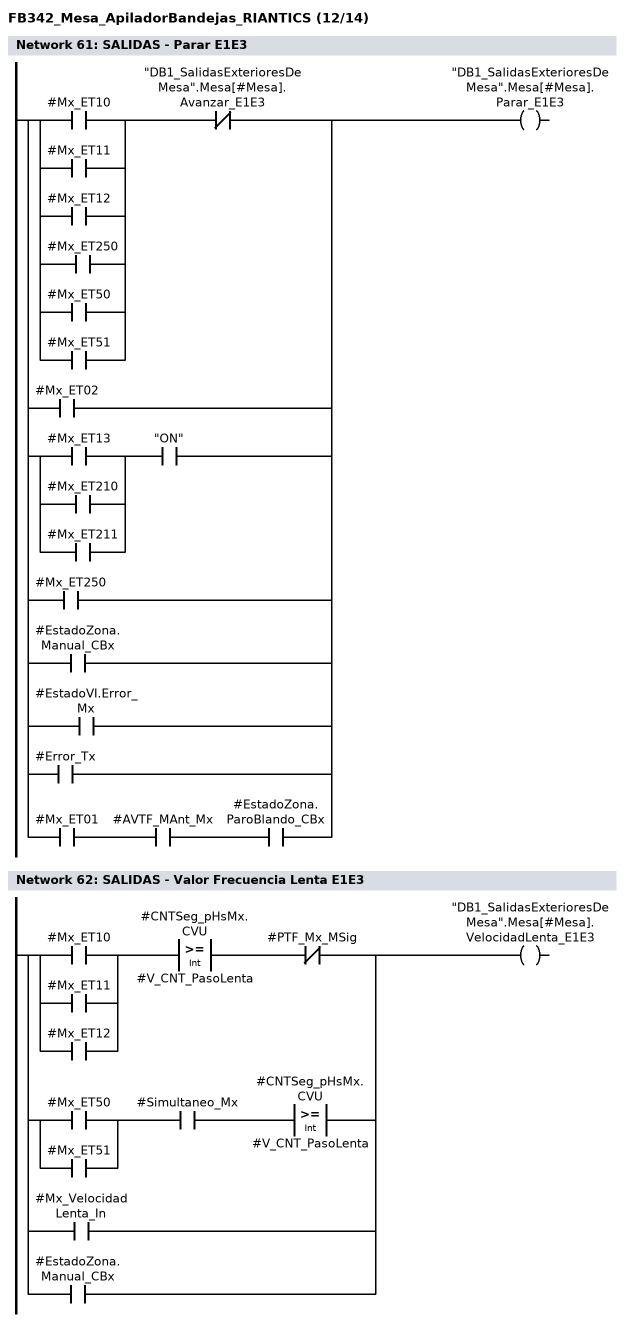
   RUNG wire#powerrail
      Contact( #Mx_ET10 )
      wire#w1
      I_Contact( "DB1_SalidasExterioresDeMesa".Mesa[#Mesa].Avanzar_E1E3 )
      wire#w2
      Coil( "DB1_SalidasExterioresDeMesa".Mesa[#Mesa].Parar_E1E3 )
   END_RUNG
   RUNG wire#powerrail
      Contact( #Mx_ET11 )
   END_RUNG wire#w1
   RUNG wire#powerrail
      Contact( #Mx_ET12 )
   END_RUNG wire#w1
   RUNG wire#powerrail
      Contact( #Mx_ET250 )
   END_RUNG wire#w1
   RUNG wire#powerrail
      Contact( #Mx_ET50 )
   END_RUNG wire#w1
   RUNG wire#powerrail
      Contact( #Mx_ET51 )
   END_RUNG wire#w1
   RUNG wire#powerrail
      Contact( #Mx_ET02 )
   END_RUNG wire#w2
   RUNG wire#powerrail
      Contact( #Mx_ET13 )
      wire#w3
      Contact( "ON" )
   END_RUNG wire#w2
   RUNG wire#powerrail
      Contact( #Mx_ET210 )
   END_RUNG wire#w3
   RUNG wire#powerrail
      Contact( #Mx_ET211 )
   END_RUNG wire#w3
   RUNG wire#powerrail
      Contact( #Mx_ET250 )
   END_RUNG wire#w2
   RUNG wire#powerrail
      Contact( #EstadoZona.Manual_CBx )
   END_RUNG wire#w2
   RUNG wire#powerrail
      Contact( #EstadoVI.Error_Mx )
   END_RUNG wire#w2
   RUNG wire#powerrail
      Contact( #Error_Tx )
   END_RUNG wire#w2
   RUNG wire#powerrail
      Contact( #Mx_ET01 )
      Contact( #AVTF_MAnt_Mx )
      Contact( #EstadoZona.ParoBlando_CBx )
   END_RUNG wire#w2
   // the same network as SCL:
   "DB1_SalidasExterioresDeMesa".Mesa[#Mesa].Parar_E1E3 := ((#Mx_ET10 OR #Mx_ET11 OR #Mx_ET12 OR #Mx_ET250 OR #Mx_ET50 OR #Mx_ET51) AND NOT "DB1_SalidasExterioresDeMesa".Mesa[#Mesa].Avanzar_E1E3) OR #Mx_ET02 OR ((#Mx_ET13 OR #Mx_ET210 OR #Mx_ET211) AND "ON") OR #Mx_ET250 OR #EstadoZona.Manual_CBx OR #EstadoVI.Error_Mx OR #Error_Tx OR (#Mx_ET01 AND #AVTF_MAnt_Mx AND #EstadoZona.ParoBlando_CBx);
END_REGION

REGION Network 62: SALIDAS - Valor Frecuencia Lenta E1E3
   RUNG wire#powerrail
      Contact( #Mx_ET10 )
      wire#w1
      { S7_Templates := "SrcType := Int" } GE_Contact(in1 := #CNTSeg_pHsMx.CVU, in2 := #V_CNT_PasoLenta)
      I_Contact( #PTF_Mx_MSig )
      wire#w2
      Coil( "DB1_SalidasExterioresDeMesa".Mesa[#Mesa].VelocidadLenta_E1E3 )
   END_RUNG
   RUNG wire#powerrail
      Contact( #Mx_ET11 )
   END_RUNG wire#w1
   RUNG wire#powerrail
      Contact( #Mx_ET12 )
   END_RUNG wire#w1
   RUNG wire#powerrail
      Contact( #Mx_ET50 )
      wire#w3
      Contact( #Simultaneo_Mx )
      { S7_Templates := "SrcType := Int" } GE_Contact(in1 := #CNTSeg_pHsMx.CVU, in2 := #V_CNT_PasoLenta)
   END_RUNG wire#w2
   RUNG wire#powerrail
      Contact( #Mx_ET51 )
   END_RUNG wire#w3
   RUNG wire#powerrail
      Contact( #Mx_VelocidadLenta_In )
   END_RUNG wire#w2
   RUNG wire#powerrail
      Contact( #EstadoZona.Manual_CBx )
   END_RUNG wire#w2
   // the same network as SCL:
   "DB1_SalidasExterioresDeMesa".Mesa[#Mesa].VelocidadLenta_E1E3 := ((#Mx_ET10 OR #Mx_ET11 OR #Mx_ET12) AND (#CNTSeg_pHsMx.CVU >= #V_CNT_PasoLenta) AND NOT #PTF_Mx_MSig) OR ((#Mx_ET50 OR #Mx_ET51) AND #Simultaneo_Mx AND (#CNTSeg_pHsMx.CVU >= #V_CNT_PasoLenta)) OR #Mx_VelocidadLenta_In OR #EstadoZona.Manual_CBx;
END_REGION

REGION Network 63: SALIDAS - Bajar Tope TP1 NOTA: Tope E1 >> S3
   // ACTIVAREMOS EL TOPE SOLO CUANDO HAYA YA PERMISO DE SALIDA. ESTO PARA LAS MAQUINAS QUE TENGAN ACTUADOR ELECTRICO. EN UNO NEUMATICO SE PUEDEN QUITAR LOS DOS OFFS
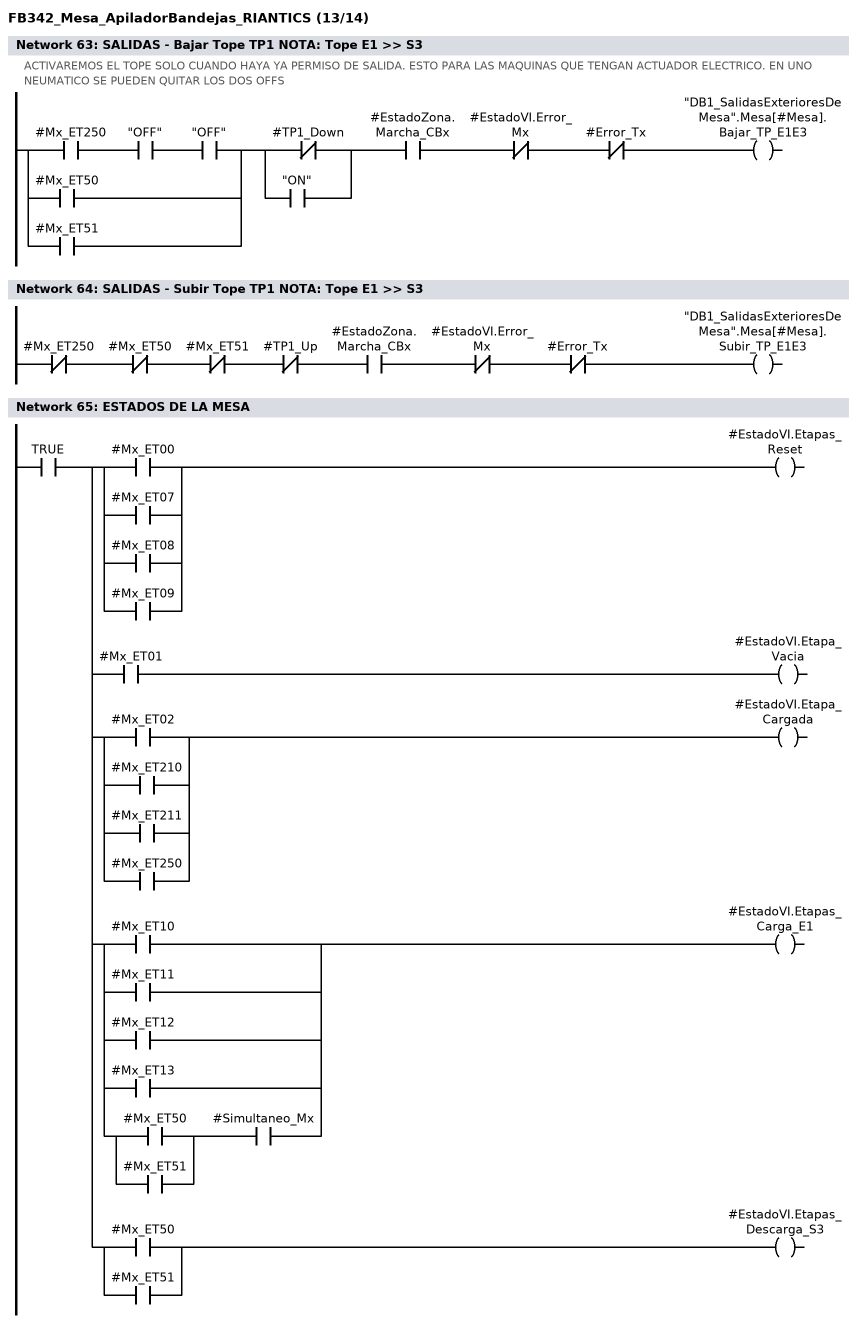
   RUNG wire#powerrail
      Contact( #Mx_ET250 )
      Contact( "OFF" )
      Contact( "OFF" )
      wire#w1
      I_Contact( #TP1_Down )
      wire#w2
      Contact( #EstadoZona.Marcha_CBx )
      I_Contact( #EstadoVI.Error_Mx )
      I_Contact( #Error_Tx )
      Coil( "DB1_SalidasExterioresDeMesa".Mesa[#Mesa].Bajar_TP_E1E3 )
   END_RUNG
   RUNG wire#powerrail
      Contact( #Mx_ET50 )
   END_RUNG wire#w1
   RUNG wire#powerrail
      Contact( #Mx_ET51 )
   END_RUNG wire#w1
   RUNG wire#w1
      Contact( "ON" )
   END_RUNG wire#w2
   // the same network as SCL:
   "DB1_SalidasExterioresDeMesa".Mesa[#Mesa].Bajar_TP_E1E3 := ((#Mx_ET250 AND "OFF" AND "OFF") OR #Mx_ET50 OR #Mx_ET51) AND (NOT #TP1_Down OR "ON") AND #EstadoZona.Marcha_CBx AND NOT #EstadoVI.Error_Mx AND NOT #Error_Tx;
END_REGION

REGION Network 64: SALIDAS - Subir Tope TP1 NOTA: Tope E1 >> S3
   RUNG wire#powerrail
      I_Contact( #Mx_ET250 )
      I_Contact( #Mx_ET50 )
      I_Contact( #Mx_ET51 )
      I_Contact( #TP1_Up )
      Contact( #EstadoZona.Marcha_CBx )
      I_Contact( #EstadoVI.Error_Mx )
      I_Contact( #Error_Tx )
      Coil( "DB1_SalidasExterioresDeMesa".Mesa[#Mesa].Subir_TP_E1E3 )
   END_RUNG
   // the same network as SCL:
   "DB1_SalidasExterioresDeMesa".Mesa[#Mesa].Subir_TP_E1E3 := NOT #Mx_ET250 AND NOT #Mx_ET50 AND NOT #Mx_ET51 AND NOT #TP1_Up AND #EstadoZona.Marcha_CBx AND NOT #EstadoVI.Error_Mx AND NOT #Error_Tx;
END_REGION

REGION Network 65: ESTADOS DE LA MESA
   RUNG wire#powerrail
      Contact( TRUE )
      wire#w1
      Contact( #Mx_ET00 )
      wire#w2
      Coil( #EstadoVI.Etapas_Reset )
   END_RUNG
   RUNG wire#w1
      Contact( #Mx_ET07 )
   END_RUNG wire#w2
   RUNG wire#w1
      Contact( #Mx_ET08 )
   END_RUNG wire#w2
   RUNG wire#w1
      Contact( #Mx_ET09 )
   END_RUNG wire#w2
   RUNG wire#w1
      Contact( #Mx_ET01 )
      Coil( #EstadoVI.Etapa_Vacia )
   END_RUNG
   RUNG wire#w1
      Contact( #Mx_ET02 )
      wire#w3
      Coil( #EstadoVI.Etapa_Cargada )
   END_RUNG
   RUNG wire#w1
      Contact( #Mx_ET210 )
   END_RUNG wire#w3
   RUNG wire#w1
      Contact( #Mx_ET211 )
   END_RUNG wire#w3
   RUNG wire#w1
      Contact( #Mx_ET250 )
   END_RUNG wire#w3
   RUNG wire#w1
      Contact( #Mx_ET10 )
      wire#w4
      Coil( #EstadoVI.Etapas_Carga_E1 )
   END_RUNG
   RUNG wire#w1
      Contact( #Mx_ET11 )
   END_RUNG wire#w4
   RUNG wire#w1
      Contact( #Mx_ET12 )
   END_RUNG wire#w4
   RUNG wire#w1
      Contact( #Mx_ET13 )
   END_RUNG wire#w4
   RUNG wire#w1
      Contact( #Mx_ET50 )
      wire#w5
      Contact( #Simultaneo_Mx )
   END_RUNG wire#w4
   RUNG wire#w1
      Contact( #Mx_ET51 )
   END_RUNG wire#w5
   RUNG wire#w1
      Contact( #Mx_ET50 )
      wire#w6
      Coil( #EstadoVI.Etapas_Descarga_S3 )
   END_RUNG
   RUNG wire#w1
      Contact( #Mx_ET51 )
   END_RUNG wire#w6
   // the same network as SCL:
   #EstadoVI.Etapas_Reset := TRUE AND (#Mx_ET00 OR #Mx_ET07 OR #Mx_ET08 OR #Mx_ET09);
   #EstadoVI.Etapa_Vacia := TRUE AND #Mx_ET01;
   #EstadoVI.Etapa_Cargada := TRUE AND (#Mx_ET02 OR #Mx_ET210 OR #Mx_ET211 OR #Mx_ET250);
   #EstadoVI.Etapas_Carga_E1 := TRUE AND (#Mx_ET10 OR #Mx_ET11 OR #Mx_ET12 OR #Mx_ET13 OR ((#Mx_ET50 OR #Mx_ET51) AND #Simultaneo_Mx));
   #EstadoVI.Etapas_Descarga_S3 := TRUE AND (#Mx_ET50 OR #Mx_ET51);
END_REGION

REGION Network 66: ENTRADAS DE LA MESA
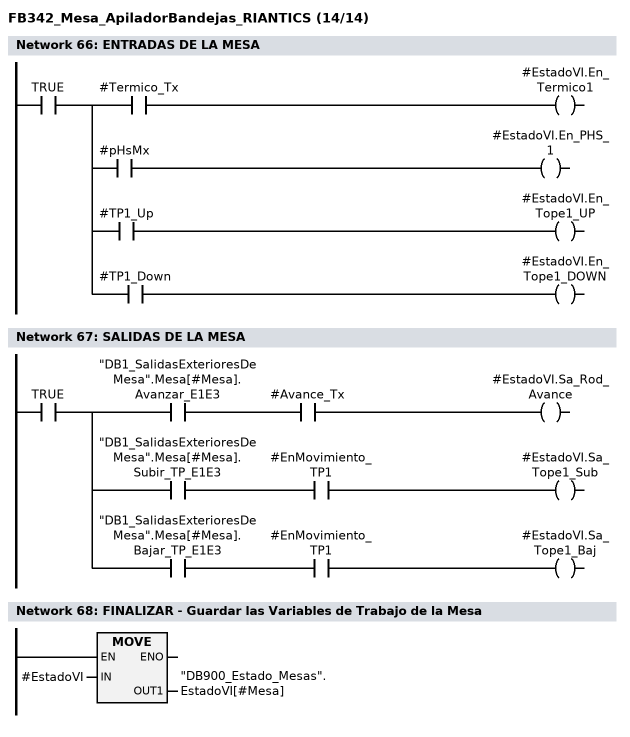
   RUNG wire#powerrail
      Contact( TRUE )
      wire#w1
      Contact( #Termico_Tx )
      Coil( #EstadoVI.En_Termico1 )
   END_RUNG
   RUNG wire#w1
      Contact( #pHsMx )
      Coil( #EstadoVI.En_PHS_1 )
   END_RUNG
   RUNG wire#w1
      Contact( #TP1_Up )
      Coil( #EstadoVI.En_Tope1_UP )
   END_RUNG
   RUNG wire#w1
      Contact( #TP1_Down )
      Coil( #EstadoVI.En_Tope1_DOWN )
   END_RUNG
   // the same network as SCL:
   #EstadoVI.En_Termico1 := TRUE AND #Termico_Tx;
   #EstadoVI.En_PHS_1 := TRUE AND #pHsMx;
   #EstadoVI.En_Tope1_UP := TRUE AND #TP1_Up;
   #EstadoVI.En_Tope1_DOWN := TRUE AND #TP1_Down;
END_REGION

REGION Network 67: SALIDAS DE LA MESA
   RUNG wire#powerrail
      Contact( TRUE )
      wire#w1
      Contact( "DB1_SalidasExterioresDeMesa".Mesa[#Mesa].Avanzar_E1E3 )
      Contact( #Avance_Tx )
      Coil( #EstadoVI.Sa_Rod_Avance )
   END_RUNG
   RUNG wire#w1
      Contact( "DB1_SalidasExterioresDeMesa".Mesa[#Mesa].Subir_TP_E1E3 )
      Contact( #EnMovimiento_TP1 )
      Coil( #EstadoVI.Sa_Tope1_Sub )
   END_RUNG
   RUNG wire#w1
      Contact( "DB1_SalidasExterioresDeMesa".Mesa[#Mesa].Bajar_TP_E1E3 )
      Contact( #EnMovimiento_TP1 )
      Coil( #EstadoVI.Sa_Tope1_Baj )
   END_RUNG
   // the same network as SCL:
   #EstadoVI.Sa_Rod_Avance := TRUE AND "DB1_SalidasExterioresDeMesa".Mesa[#Mesa].Avanzar_E1E3 AND #Avance_Tx;
   #EstadoVI.Sa_Tope1_Sub := TRUE AND "DB1_SalidasExterioresDeMesa".Mesa[#Mesa].Subir_TP_E1E3 AND #EnMovimiento_TP1;
   #EstadoVI.Sa_Tope1_Baj := TRUE AND "DB1_SalidasExterioresDeMesa".Mesa[#Mesa].Bajar_TP_E1E3 AND #EnMovimiento_TP1;
END_REGION

REGION Network 68: FINALIZAR - Guardar las Variables de Trabajo de la Mesa
   RUNG wire#powerrail
      Move(in := #EstadoVI, out1 => "DB900_Estado_Mesas".EstadoVI[#Mesa])
   END_RUNG
   // the same network as SCL:
   "DB900_Estado_Mesas".EstadoVI[#Mesa] := #EstadoVI;
END_REGION
END_FUNCTION_BLOCK

FUNCTION_BLOCK "FB343_ApiladorBandejas_RIANTICS"   // FB343, LAD
{ S7_Optimized_Access := 'FALSE' }
// stored: AutoNumber false, SetENOAutomatically false
   VAR_INPUT
      Maquina : UInt;   // Numero de Maquina (Mesa)
      Error_Tx : Bool;   // Error en el Tx
      EnTension : Bool;   // Existe Tension en la Maquina
      MAQx_Desabilitada : Bool;   // Config MAQ. >>> DesHabilitada
      Termico_Elevacion : Bool;   // Termico de la Elevacion
      Pos_DW : Bool;   // Posición Baja del Apilador
      Pos_mid_DW : Bool;
      Pos_mid_UP : Bool;
      Pos_UP : Bool;   // Posición Alta del Apilador
      EnMovimiento_Elevacion : Bool;   // En Movineto la Elevacion
      CargaSuelta : Bool;   // Carga Suelta en el Apilador
      CargaCogida : Bool;   // Carga Cogida en el Apilador
      EnMovimiento_Horquillado : Bool;   // En Movimiento el Hoquillado
      MAQ_DejarBandejas : Bool;   // Interlock >> Dejar Bandejas
      MAQ_CogerBandejas : Bool;   // Interlock >> Coger Bandejas
      MAQ_BuscarCero : Bool;   // Interlock >> Buscar Cero
      CogiendoDerecha : Bool;
      CogiendoIzquierda : Bool;
      DejandoDerecha : Bool;
      DejandoIzquierda : Bool;
      V_TOut_Elevacion : Int := 2000;   // TimeOut del Mov. de Elevacion
      V_TOut_Horquillado : Int := 2000;   // TimeOut del Mov. de Horquillado
   END_VAR
   VAR_OUTPUT
      MAQ_DejadasBandejas : Bool;   // Interlock >> Bandejas Dejadas
      MAQ_CojidasBandejas : Bool;   // Interlock >> Bandejas Cogidas
      MAQ_CeroEncontrado : Bool;   // Interlock >> Bandejas
   END_VAR
   VAR
      AP_ET00 : Bool;
      AP_ET01 : Bool;
      AP_ET100 : Bool;
      AP_ET101 : Bool;
      AP_ET102 : Bool;
      AP_ET103 : Bool;
      AP_ET104 : Bool;
      AP_ET50 : Bool;
      AP_ET51 : Bool;
      AP_ET52 : Bool;
      AP_ET53 : Bool;
      AP_ET54 : Bool;
      AP_ET60 : Bool;
      AP_ET61 : Bool;
      AP_ET62 : Bool;
      AP_ET63 : Bool;
      AP_ET64 : Bool;
      MA_Motor_Elev : Bool;
      MA_Slow_Velocity : Bool;
      MA_CogerCarga : Bool;   // Cerrar Cilindros para coger la pila
      MA_DejarCarga : Bool;   // Abrir Cilindros para dejas la pila
      TMP_ReposoCargaSuelta { S7_SetPoint := 'True'} : TON_TIME;
      TMP_EnTension { S7_SetPoint := 'True'} : "FB910_CNT_UHS";
      TOut_Elevacion { S7_SetPoint := 'True'} : "FB910_CNT_UHS";
      TOut_Horquillado { S7_SetPoint := 'True'} : "FB910_CNT_UHS";
      Manual : "MoviManualMaquina_Apilador_bandejas";
   END_VAR
   VAR_TEMP
      EstadoZona : "EstadoZona";   // Estado de Zona de la Mesa
      EstadoMAQ : "EstadoMaquina_Apilador_bandejas";   // Estado del Vehiculo Inteliguente de la Maquina
      Aux_ET00 : Bool;
   END_VAR
BEGIN

REGION Network 1: INICIALIZAR - Recoger las Variables de Estado de la Maquina
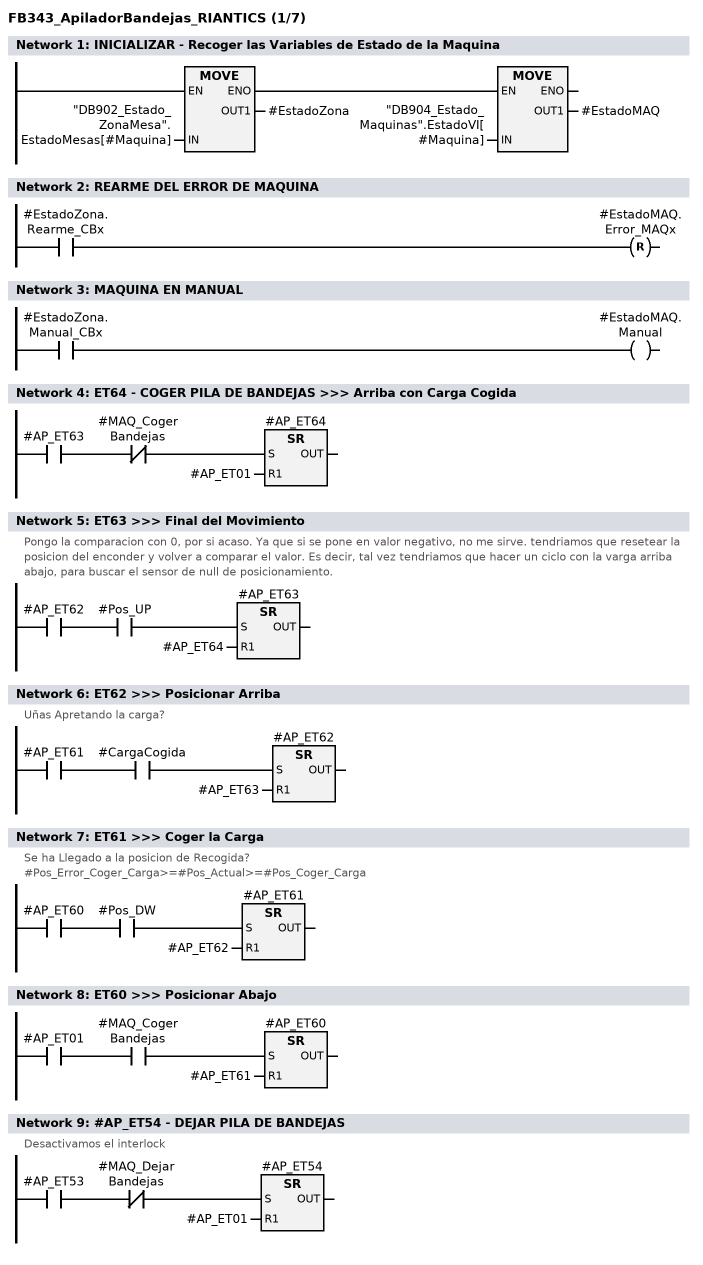
   RUNG wire#powerrail
      Move(in := "DB902_Estado_ZonaMesa".EstadoMesas[#Maquina], out1 => #EstadoZona)
      Move(in := "DB904_Estado_Maquinas".EstadoVI[#Maquina], out1 => #EstadoMAQ)
   END_RUNG
   // the same network as SCL:
   #EstadoZona := "DB902_Estado_ZonaMesa".EstadoMesas[#Maquina];
   #EstadoMAQ := "DB904_Estado_Maquinas".EstadoVI[#Maquina];
END_REGION

REGION Network 2: REARME DEL ERROR DE MAQUINA
   RUNG wire#powerrail
      Contact( #EstadoZona.Rearme_CBx )
      R_Coil( #EstadoMAQ.Error_MAQx )
   END_RUNG
   // the same network as SCL:
   IF #EstadoZona.Rearme_CBx THEN #EstadoMAQ.Error_MAQx := FALSE; END_IF;
END_REGION

REGION Network 3: MAQUINA EN MANUAL
   RUNG wire#powerrail
      Contact( #EstadoZona.Manual_CBx )
      Coil( #EstadoMAQ.Manual )
   END_RUNG
   // the same network as SCL:
   #EstadoMAQ.Manual := #EstadoZona.Manual_CBx;
END_REGION

REGION Network 4: ET64 - COGER PILA DE BANDEJAS >>> Arriba con Carga Cogida
   RUNG wire#powerrail
      Contact( #AP_ET63 )
      I_Contact( #MAQ_CogerBandejas )
      S_SR(operand := #AP_ET64, r1 := #AP_ET01)
   END_RUNG
   // the same network as SCL:
   IF #AP_ET63 AND NOT #MAQ_CogerBandejas THEN
       #AP_ET64 := TRUE;   // SR flip-flop
   END_IF;
   IF #AP_ET01 THEN #AP_ET64 := FALSE; END_IF;
END_REGION

REGION Network 5: ET63 >>> Final del Movimiento
   // Pongo la comparacion con 0, por si acaso. Ya que si se pone en valor negativo, no me sirve. tendriamos que resetear la posicion del enconder y volver a comparar el valor. Es decir, tal vez tendriamos que hacer un ciclo con la varga arriba abajo, para buscar el sensor de null de posicionamiento.
   RUNG wire#powerrail
      Contact( #AP_ET62 )
      Contact( #Pos_UP )
      S_SR(operand := #AP_ET63, r1 := #AP_ET64)
   END_RUNG
   // the same network as SCL:
   IF #AP_ET62 AND #Pos_UP THEN
       #AP_ET63 := TRUE;   // SR flip-flop
   END_IF;
   IF #AP_ET64 THEN #AP_ET63 := FALSE; END_IF;
END_REGION

REGION Network 6: ET62 >>> Posicionar Arriba
   // Uñas Apretando la carga?
   RUNG wire#powerrail
      Contact( #AP_ET61 )
      Contact( #CargaCogida )
      S_SR(operand := #AP_ET62, r1 := #AP_ET63)
   END_RUNG
   // the same network as SCL:
   IF #AP_ET61 AND #CargaCogida THEN
       #AP_ET62 := TRUE;   // SR flip-flop
   END_IF;
   IF #AP_ET63 THEN #AP_ET62 := FALSE; END_IF;
END_REGION

REGION Network 7: ET61 >>> Coger la Carga
   // Se ha Llegado a la posicion de Recogida?
   // #Pos_Error_Coger_Carga>=#Pos_Actual>=#Pos_Coger_Carga
   RUNG wire#powerrail
      Contact( #AP_ET60 )
      Contact( #Pos_DW )
      S_SR(operand := #AP_ET61, r1 := #AP_ET62)
   END_RUNG
   // the same network as SCL:
   IF #AP_ET60 AND #Pos_DW THEN
       #AP_ET61 := TRUE;   // SR flip-flop
   END_IF;
   IF #AP_ET62 THEN #AP_ET61 := FALSE; END_IF;
END_REGION

REGION Network 8: ET60 >>> Posicionar Abajo
   RUNG wire#powerrail
      Contact( #AP_ET01 )
      Contact( #MAQ_CogerBandejas )
      S_SR(operand := #AP_ET60, r1 := #AP_ET61)
   END_RUNG
   // the same network as SCL:
   IF #AP_ET01 AND #MAQ_CogerBandejas THEN
       #AP_ET60 := TRUE;   // SR flip-flop
   END_IF;
   IF #AP_ET61 THEN #AP_ET60 := FALSE; END_IF;
END_REGION

REGION Network 9: #AP_ET54 - DEJAR PILA DE BANDEJAS
   // Desactivamos el interlock
   RUNG wire#powerrail
      Contact( #AP_ET53 )
      I_Contact( #MAQ_DejarBandejas )
      S_SR(operand := #AP_ET54, r1 := #AP_ET01)
   END_RUNG
   // the same network as SCL:
   IF #AP_ET53 AND NOT #MAQ_DejarBandejas THEN
       #AP_ET54 := TRUE;   // SR flip-flop
   END_IF;
   IF #AP_ET01 THEN #AP_ET54 := FALSE; END_IF;
END_REGION

REGION Network 10: ET53 - Bajamos a posicion de espera. para optimizar mov,. apilador esperando>>> abajo con Carga Suelta
   // Coger carga
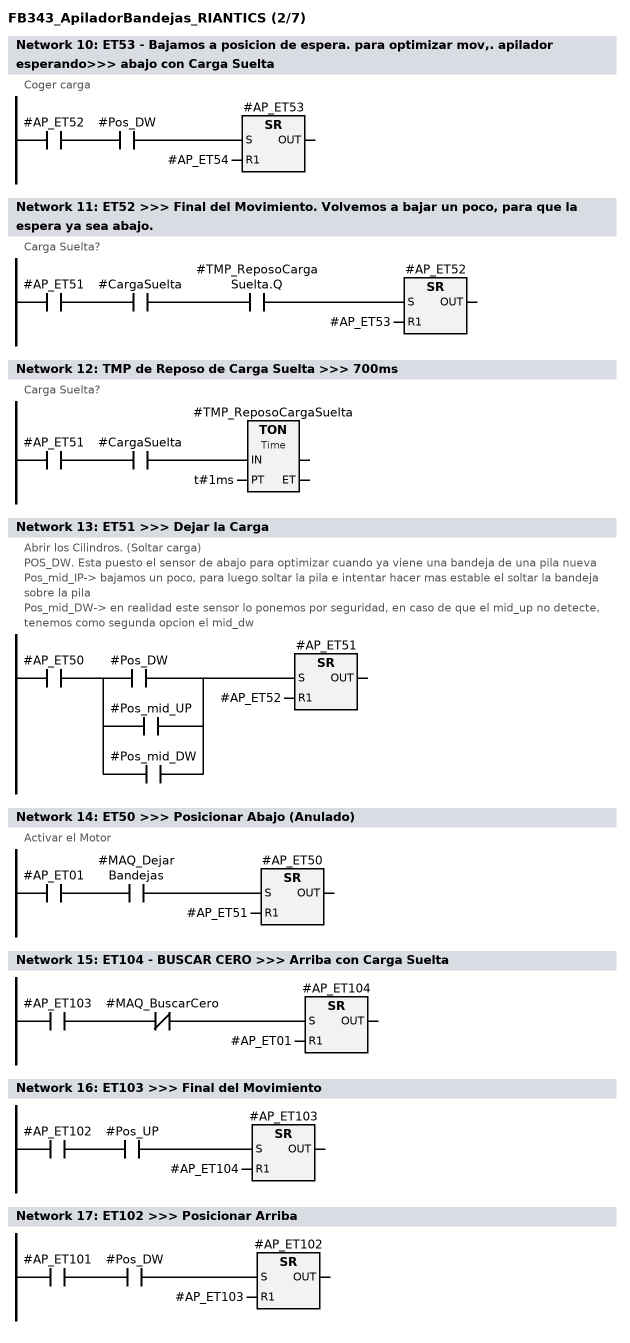
   RUNG wire#powerrail
      Contact( #AP_ET52 )
      Contact( #Pos_DW )
      S_SR(operand := #AP_ET53, r1 := #AP_ET54)
   END_RUNG
   // the same network as SCL:
   IF #AP_ET52 AND #Pos_DW THEN
       #AP_ET53 := TRUE;   // SR flip-flop
   END_IF;
   IF #AP_ET54 THEN #AP_ET53 := FALSE; END_IF;
END_REGION

REGION Network 11: ET52 >>> Final del Movimiento. Volvemos a bajar un poco, para que la espera ya sea abajo.
   // Carga Suelta?
   RUNG wire#powerrail
      Contact( #AP_ET51 )
      Contact( #CargaSuelta )
      Contact( #TMP_ReposoCargaSuelta.Q )
      S_SR(operand := #AP_ET52, r1 := #AP_ET53)
   END_RUNG
   // the same network as SCL:
   IF #AP_ET51 AND #CargaSuelta AND #TMP_ReposoCargaSuelta.Q THEN
       #AP_ET52 := TRUE;   // SR flip-flop
   END_IF;
   IF #AP_ET53 THEN #AP_ET52 := FALSE; END_IF;
END_REGION

REGION Network 12: TMP de Reposo de Carga Suelta >>> 700ms
   // Carga Suelta?
   RUNG wire#powerrail
      Contact( #AP_ET51 )
      Contact( #CargaSuelta )
      { S7_Templates := "time_type := Time" } #TMP_ReposoCargaSuelta.TON(pt := t#1ms, et =>)
   END_RUNG
   // the same network as SCL:
   #TMP_ReposoCargaSuelta(IN := #AP_ET51 AND #CargaSuelta, PT := t#1ms);   // TON
END_REGION

REGION Network 13: ET51 >>> Dejar la Carga
   // Abrir los Cilindros. (Soltar carga)
   // POS_DW. Esta puesto el sensor de abajo para optimizar cuando ya viene una bandeja de una pila nueva
   // Pos_mid_IP-> bajamos un poco, para luego soltar la pila e intentar hacer mas estable el soltar la bandeja sobre la pila
   // Pos_mid_DW-> en realidad este sensor lo ponemos por seguridad, en caso de que el mid_up no detecte, tenemos como segunda opcion el mid_dw
   RUNG wire#powerrail
      Contact( #AP_ET50 )
      wire#w1
      Contact( #Pos_DW )
      wire#w2
      S_SR(operand := #AP_ET51, r1 := #AP_ET52)
   END_RUNG
   RUNG wire#w1
      Contact( #Pos_mid_UP )
   END_RUNG wire#w2
   RUNG wire#w1
      Contact( #Pos_mid_DW )
   END_RUNG wire#w2
   // the same network as SCL:
   IF #AP_ET50 AND (#Pos_DW OR #Pos_mid_UP OR #Pos_mid_DW) THEN
       #AP_ET51 := TRUE;   // SR flip-flop
   END_IF;
   IF #AP_ET52 THEN #AP_ET51 := FALSE; END_IF;
END_REGION

REGION Network 14: ET50 >>> Posicionar Abajo (Anulado)
   // Activar el Motor
   RUNG wire#powerrail
      Contact( #AP_ET01 )
      Contact( #MAQ_DejarBandejas )
      S_SR(operand := #AP_ET50, r1 := #AP_ET51)
   END_RUNG
   // the same network as SCL:
   IF #AP_ET01 AND #MAQ_DejarBandejas THEN
       #AP_ET50 := TRUE;   // SR flip-flop
   END_IF;
   IF #AP_ET51 THEN #AP_ET50 := FALSE; END_IF;
END_REGION

REGION Network 15: ET104 - BUSCAR CERO >>> Arriba con Carga Suelta
   RUNG wire#powerrail
      Contact( #AP_ET103 )
      I_Contact( #MAQ_BuscarCero )
      S_SR(operand := #AP_ET104, r1 := #AP_ET01)
   END_RUNG
   // the same network as SCL:
   IF #AP_ET103 AND NOT #MAQ_BuscarCero THEN
       #AP_ET104 := TRUE;   // SR flip-flop
   END_IF;
   IF #AP_ET01 THEN #AP_ET104 := FALSE; END_IF;
END_REGION

REGION Network 16: ET103 >>> Final del Movimiento
   RUNG wire#powerrail
      Contact( #AP_ET102 )
      Contact( #Pos_UP )
      S_SR(operand := #AP_ET103, r1 := #AP_ET104)
   END_RUNG
   // the same network as SCL:
   IF #AP_ET102 AND #Pos_UP THEN
       #AP_ET103 := TRUE;   // SR flip-flop
   END_IF;
   IF #AP_ET104 THEN #AP_ET103 := FALSE; END_IF;
END_REGION

REGION Network 17: ET102 >>> Posicionar Arriba
   RUNG wire#powerrail
      Contact( #AP_ET101 )
      Contact( #Pos_DW )
      S_SR(operand := #AP_ET102, r1 := #AP_ET103)
   END_RUNG
   // the same network as SCL:
   IF #AP_ET101 AND #Pos_DW THEN
       #AP_ET102 := TRUE;   // SR flip-flop
   END_IF;
   IF #AP_ET103 THEN #AP_ET102 := FALSE; END_IF;
END_REGION

REGION Network 18: ET101 >>> Buscar la Posicion cero (Abajo)
   // Activar el Motor
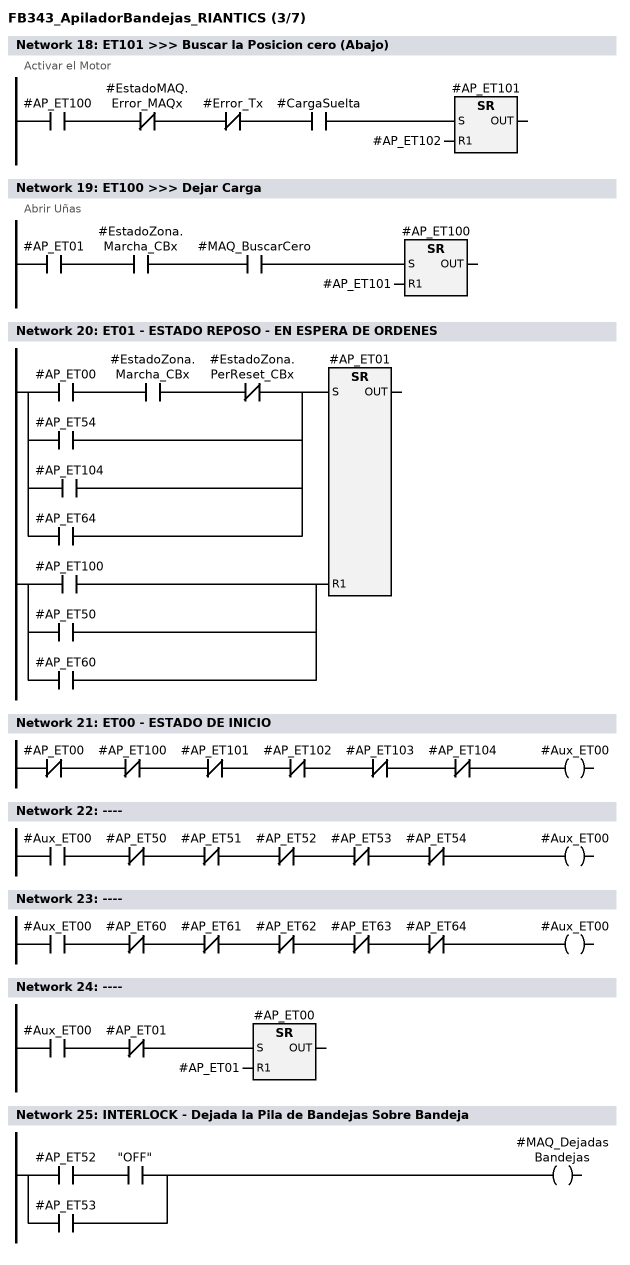
   RUNG wire#powerrail
      Contact( #AP_ET100 )
      I_Contact( #EstadoMAQ.Error_MAQx )
      I_Contact( #Error_Tx )
      Contact( #CargaSuelta )
      S_SR(operand := #AP_ET101, r1 := #AP_ET102)
   END_RUNG
   // the same network as SCL:
   IF #AP_ET100 AND NOT #EstadoMAQ.Error_MAQx AND NOT #Error_Tx AND #CargaSuelta THEN
       #AP_ET101 := TRUE;   // SR flip-flop
   END_IF;
   IF #AP_ET102 THEN #AP_ET101 := FALSE; END_IF;
END_REGION

REGION Network 19: ET100 >>> Dejar Carga
   // Abrir Uñas
   RUNG wire#powerrail
      Contact( #AP_ET01 )
      Contact( #EstadoZona.Marcha_CBx )
      Contact( #MAQ_BuscarCero )
      S_SR(operand := #AP_ET100, r1 := #AP_ET101)
   END_RUNG
   // the same network as SCL:
   IF #AP_ET01 AND #EstadoZona.Marcha_CBx AND #MAQ_BuscarCero THEN
       #AP_ET100 := TRUE;   // SR flip-flop
   END_IF;
   IF #AP_ET101 THEN #AP_ET100 := FALSE; END_IF;
END_REGION

REGION Network 20: ET01 - ESTADO REPOSO - EN ESPERA DE ORDENES
   RUNG wire#powerrail
      Contact( #AP_ET00 )
      Contact( #EstadoZona.Marcha_CBx )
      I_Contact( #EstadoZona.PerReset_CBx )
      wire#w1
      S_SR(operand := #AP_ET01, r1 := wire#w2)
   END_RUNG
   RUNG wire#powerrail
      Contact( #AP_ET54 )
   END_RUNG wire#w1
   RUNG wire#powerrail
      Contact( #AP_ET104 )
   END_RUNG wire#w1
   RUNG wire#powerrail
      Contact( #AP_ET64 )
   END_RUNG wire#w1
   RUNG wire#powerrail
      Contact( #AP_ET100 )
   END_RUNG wire#w2
   RUNG wire#powerrail
      Contact( #AP_ET50 )
   END_RUNG wire#w2
   RUNG wire#powerrail
      Contact( #AP_ET60 )
   END_RUNG wire#w2
   // the same network as SCL:
   IF (#AP_ET00 AND #EstadoZona.Marcha_CBx AND NOT #EstadoZona.PerReset_CBx) OR #AP_ET54 OR #AP_ET104 OR #AP_ET64 THEN
       #AP_ET01 := TRUE;   // SR flip-flop
   END_IF;
   IF #AP_ET100 OR #AP_ET50 OR #AP_ET60 THEN #AP_ET01 := FALSE; END_IF;
END_REGION

REGION Network 21: ET00 - ESTADO DE INICIO
   RUNG wire#powerrail
      I_Contact( #AP_ET00 )
      I_Contact( #AP_ET100 )
      I_Contact( #AP_ET101 )
      I_Contact( #AP_ET102 )
      I_Contact( #AP_ET103 )
      I_Contact( #AP_ET104 )
      Coil( #Aux_ET00 )
   END_RUNG
   // the same network as SCL:
   #Aux_ET00 := NOT #AP_ET00 AND NOT #AP_ET100 AND NOT #AP_ET101 AND NOT #AP_ET102 AND NOT #AP_ET103 AND NOT #AP_ET104;
END_REGION

REGION Network 22: ----
   RUNG wire#powerrail
      Contact( #Aux_ET00 )
      I_Contact( #AP_ET50 )
      I_Contact( #AP_ET51 )
      I_Contact( #AP_ET52 )
      I_Contact( #AP_ET53 )
      I_Contact( #AP_ET54 )
      Coil( #Aux_ET00 )
   END_RUNG
   // the same network as SCL:
   #Aux_ET00 := #Aux_ET00 AND NOT #AP_ET50 AND NOT #AP_ET51 AND NOT #AP_ET52 AND NOT #AP_ET53 AND NOT #AP_ET54;
END_REGION

REGION Network 23: ----
   RUNG wire#powerrail
      Contact( #Aux_ET00 )
      I_Contact( #AP_ET60 )
      I_Contact( #AP_ET61 )
      I_Contact( #AP_ET62 )
      I_Contact( #AP_ET63 )
      I_Contact( #AP_ET64 )
      Coil( #Aux_ET00 )
   END_RUNG
   // the same network as SCL:
   #Aux_ET00 := #Aux_ET00 AND NOT #AP_ET60 AND NOT #AP_ET61 AND NOT #AP_ET62 AND NOT #AP_ET63 AND NOT #AP_ET64;
END_REGION

REGION Network 24: ----
   RUNG wire#powerrail
      Contact( #Aux_ET00 )
      I_Contact( #AP_ET01 )
      S_SR(operand := #AP_ET00, r1 := #AP_ET01)
   END_RUNG
   // the same network as SCL:
   IF #Aux_ET00 AND NOT #AP_ET01 THEN
       #AP_ET00 := TRUE;   // SR flip-flop
   END_IF;
   IF #AP_ET01 THEN #AP_ET00 := FALSE; END_IF;
END_REGION

REGION Network 25: INTERLOCK - Dejada la Pila de Bandejas Sobre Bandeja
   RUNG wire#powerrail
      Contact( #AP_ET52 )
      Contact( "OFF" )
      wire#w1
      Coil( #MAQ_DejadasBandejas )
   END_RUNG
   RUNG wire#powerrail
      Contact( #AP_ET53 )
   END_RUNG wire#w1
   // the same network as SCL:
   #MAQ_DejadasBandejas := (#AP_ET52 AND "OFF") OR #AP_ET53;
END_REGION

REGION Network 26: VARIABLES AUXILIARES - Fin de Reset
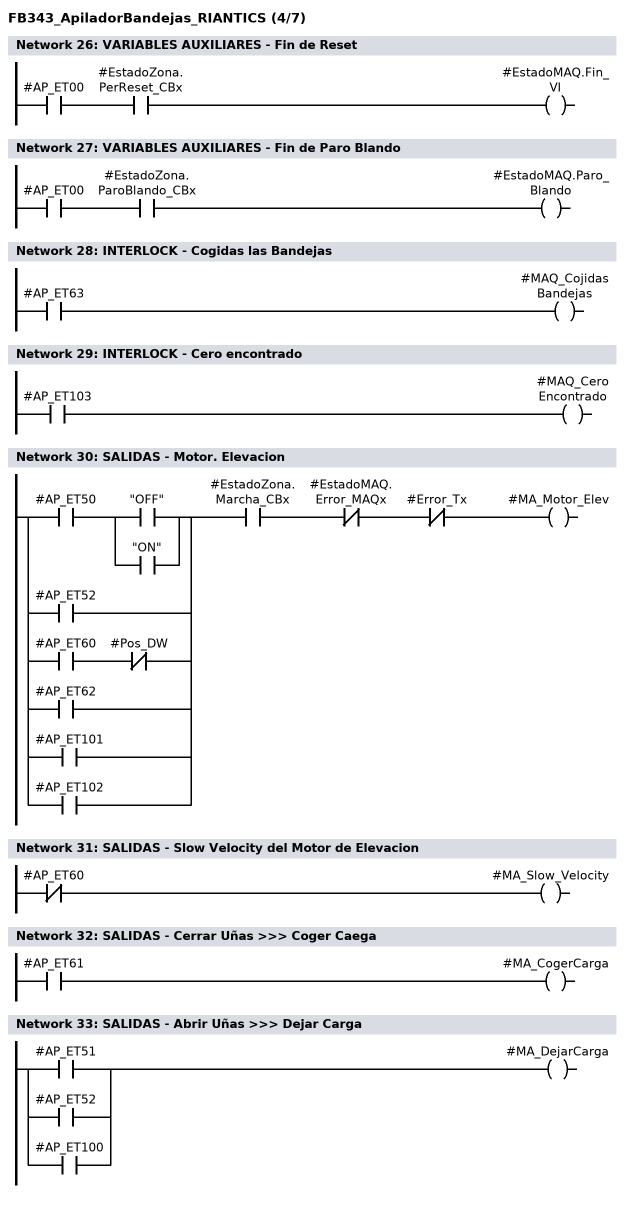
   RUNG wire#powerrail
      Contact( #AP_ET00 )
      Contact( #EstadoZona.PerReset_CBx )
      Coil( #EstadoMAQ.Fin_VI )
   END_RUNG
   // the same network as SCL:
   #EstadoMAQ.Fin_VI := #AP_ET00 AND #EstadoZona.PerReset_CBx;
END_REGION

REGION Network 27: VARIABLES AUXILIARES - Fin de Paro Blando
   RUNG wire#powerrail
      Contact( #AP_ET00 )
      Contact( #EstadoZona.ParoBlando_CBx )
      Coil( #EstadoMAQ.Paro_Blando )
   END_RUNG
   // the same network as SCL:
   #EstadoMAQ.Paro_Blando := #AP_ET00 AND #EstadoZona.ParoBlando_CBx;
END_REGION

REGION Network 28: INTERLOCK - Cogidas las Bandejas
   RUNG wire#powerrail
      Contact( #AP_ET63 )
      Coil( #MAQ_CojidasBandejas )
   END_RUNG
   // the same network as SCL:
   #MAQ_CojidasBandejas := #AP_ET63;
END_REGION

REGION Network 29: INTERLOCK - Cero encontrado
   RUNG wire#powerrail
      Contact( #AP_ET103 )
      Coil( #MAQ_CeroEncontrado )
   END_RUNG
   // the same network as SCL:
   #MAQ_CeroEncontrado := #AP_ET103;
END_REGION

REGION Network 30: SALIDAS - Motor. Elevacion
   RUNG wire#powerrail
      Contact( #AP_ET50 )
      wire#w1
      Contact( "OFF" )
      wire#w2
      Contact( #EstadoZona.Marcha_CBx )
      I_Contact( #EstadoMAQ.Error_MAQx )
      I_Contact( #Error_Tx )
      Coil( #MA_Motor_Elev )
   END_RUNG
   RUNG wire#w1
      Contact( "ON" )
   END_RUNG wire#w2
   RUNG wire#powerrail
      Contact( #AP_ET52 )
   END_RUNG wire#w2
   RUNG wire#powerrail
      Contact( #AP_ET60 )
      I_Contact( #Pos_DW )
   END_RUNG wire#w2
   RUNG wire#powerrail
      Contact( #AP_ET62 )
   END_RUNG wire#w2
   RUNG wire#powerrail
      Contact( #AP_ET101 )
   END_RUNG wire#w2
   RUNG wire#powerrail
      Contact( #AP_ET102 )
   END_RUNG wire#w2
   // the same network as SCL:
   #MA_Motor_Elev := ((#AP_ET50 AND ("OFF" OR "ON")) OR #AP_ET52 OR (#AP_ET60 AND NOT #Pos_DW) OR #AP_ET62 OR #AP_ET101 OR #AP_ET102) AND #EstadoZona.Marcha_CBx AND NOT #EstadoMAQ.Error_MAQx AND NOT #Error_Tx;
END_REGION

REGION Network 31: SALIDAS - Slow Velocity del Motor de Elevacion
   RUNG wire#powerrail
      I_Contact( #AP_ET60 )
      Coil( #MA_Slow_Velocity )
   END_RUNG
   // the same network as SCL:
   #MA_Slow_Velocity := NOT #AP_ET60;
END_REGION

REGION Network 32: SALIDAS - Cerrar Uñas >>> Coger Caega
   RUNG wire#powerrail
      Contact( #AP_ET61 )
      Coil( #MA_CogerCarga )
   END_RUNG
   // the same network as SCL:
   #MA_CogerCarga := #AP_ET61;
END_REGION

REGION Network 33: SALIDAS - Abrir Uñas >>> Dejar Carga
   RUNG wire#powerrail
      Contact( #AP_ET51 )
      wire#w1
      Coil( #MA_DejarCarga )
   END_RUNG
   RUNG wire#powerrail
      Contact( #AP_ET52 )
   END_RUNG wire#w1
   RUNG wire#powerrail
      Contact( #AP_ET100 )
   END_RUNG wire#w1
   // the same network as SCL:
   #MA_DejarCarga := #AP_ET51 OR #AP_ET52 OR #AP_ET100;
END_REGION

REGION Network 34: TMP - Espera En Tension
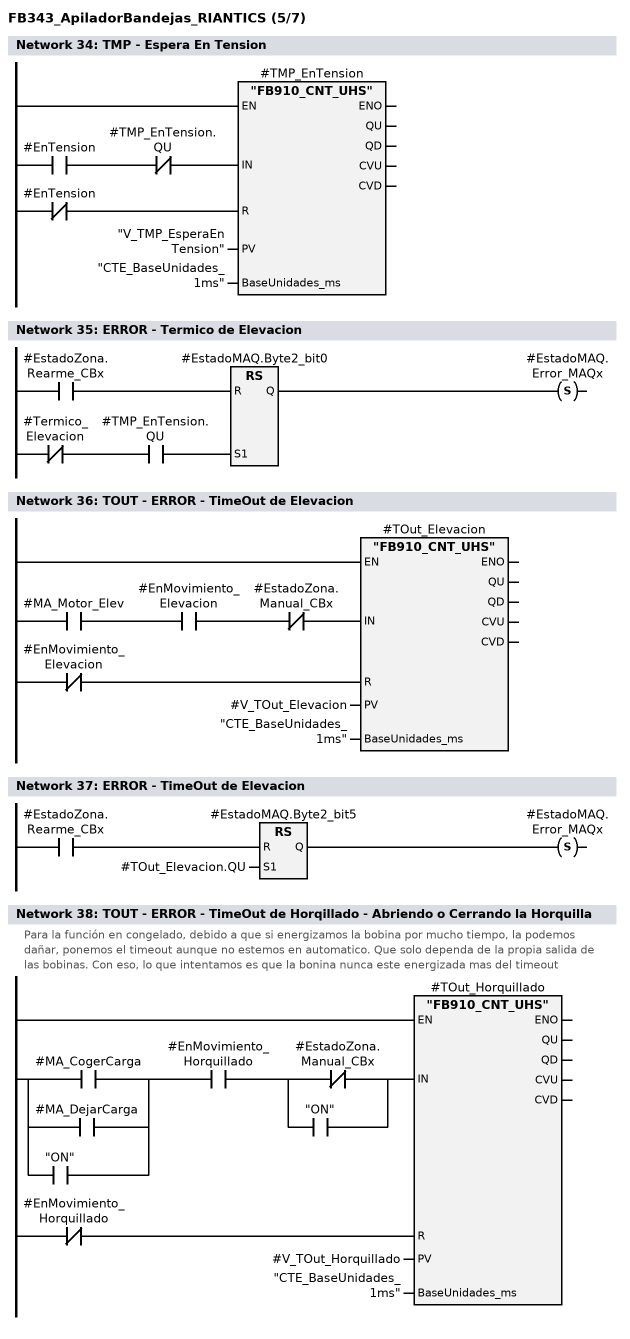
   RUNG wire#powerrail
      #TMP_EnTension(IN := wire#w1, R := wire#w2, PV := "V_TMP_EsperaEnTension", BaseUnidades_ms := "CTE_BaseUnidades_1ms", QU =>, QD =>, CVU =>, CVD =>)
   END_RUNG
   RUNG wire#powerrail
      Contact( #EnTension )
      I_Contact( #TMP_EnTension.QU )
   END_RUNG wire#w1
   RUNG wire#powerrail
      I_Contact( #EnTension )
   END_RUNG wire#w2
   // the same network as SCL:
   #TMP_EnTension(IN := #EnTension AND NOT #TMP_EnTension.QU,   // "FB910_CNT_UHS"
                  R := NOT #EnTension,
                  PV := "V_TMP_EsperaEnTension",
                  BaseUnidades_ms := "CTE_BaseUnidades_1ms");
END_REGION

REGION Network 35: ERROR - Termico de Elevacion
   RUNG wire#powerrail
      Contact( #EstadoZona.Rearme_CBx )
      S_RS(operand := #EstadoMAQ.Byte2_bit0, s1 := wire#w1)
      S_Coil( #EstadoMAQ.Error_MAQx )
   END_RUNG
   RUNG wire#powerrail
      I_Contact( #Termico_Elevacion )
      Contact( #TMP_EnTension.QU )
   END_RUNG wire#w1
   // the same network as SCL:
   IF #EstadoZona.Rearme_CBx THEN
       #EstadoMAQ.Byte2_bit0 := FALSE;   // RS flip-flop
   END_IF;
   IF NOT #Termico_Elevacion AND #TMP_EnTension.QU THEN #EstadoMAQ.Byte2_bit0 := TRUE; END_IF;
   IF #EstadoMAQ.Byte2_bit0 THEN #EstadoMAQ.Error_MAQx := TRUE; END_IF;
END_REGION

REGION Network 36: TOUT - ERROR - TimeOut de Elevacion
   RUNG wire#powerrail
      #TOut_Elevacion(IN := wire#w1, R := wire#w2, PV := #V_TOut_Elevacion, BaseUnidades_ms := "CTE_BaseUnidades_1ms", QU =>, QD =>, CVU =>, CVD =>)
   END_RUNG
   RUNG wire#powerrail
      Contact( #MA_Motor_Elev )
      Contact( #EnMovimiento_Elevacion )
      I_Contact( #EstadoZona.Manual_CBx )
   END_RUNG wire#w1
   RUNG wire#powerrail
      I_Contact( #EnMovimiento_Elevacion )
   END_RUNG wire#w2
   // the same network as SCL:
   #TOut_Elevacion(IN := #MA_Motor_Elev AND #EnMovimiento_Elevacion AND NOT #EstadoZona.Manual_CBx,   // "FB910_CNT_UHS"
                   R := NOT #EnMovimiento_Elevacion,
                   PV := #V_TOut_Elevacion,
                   BaseUnidades_ms := "CTE_BaseUnidades_1ms");
END_REGION

REGION Network 37: ERROR - TimeOut de Elevacion
   RUNG wire#powerrail
      Contact( #EstadoZona.Rearme_CBx )
      S_RS(operand := #EstadoMAQ.Byte2_bit5, s1 := #TOut_Elevacion.QU)
      S_Coil( #EstadoMAQ.Error_MAQx )
   END_RUNG
   // the same network as SCL:
   IF #EstadoZona.Rearme_CBx THEN
       #EstadoMAQ.Byte2_bit5 := FALSE;   // RS flip-flop
   END_IF;
   IF #TOut_Elevacion.QU THEN #EstadoMAQ.Byte2_bit5 := TRUE; END_IF;
   IF #EstadoMAQ.Byte2_bit5 THEN #EstadoMAQ.Error_MAQx := TRUE; END_IF;
END_REGION

REGION Network 38: TOUT - ERROR - TimeOut de Horqillado - Abriendo o Cerrando la Horquilla
   // Para la función en congelado, debido a que si energizamos la bobina por mucho tiempo, la podemos dañar, ponemos el timeout aunque no estemos en automatico. Que solo dependa de la propia salida de las bobinas. Con eso, lo que intentamos es que la bonina nunca este energizada mas del timeout
   RUNG wire#powerrail
      #TOut_Horquillado(IN := wire#w3, R := wire#w4, PV := #V_TOut_Horquillado, BaseUnidades_ms := "CTE_BaseUnidades_1ms", QU =>, QD =>, CVU =>, CVD =>)
   END_RUNG
   RUNG wire#powerrail
      Contact( #MA_CogerCarga )
      wire#w1
      Contact( #EnMovimiento_Horquillado )
      wire#w2
      I_Contact( #EstadoZona.Manual_CBx )
   END_RUNG wire#w3
   RUNG wire#powerrail
      Contact( #MA_DejarCarga )
   END_RUNG wire#w1
   RUNG wire#powerrail
      Contact( "ON" )
   END_RUNG wire#w1
   RUNG wire#w2
      Contact( "ON" )
   END_RUNG wire#w3
   RUNG wire#powerrail
      I_Contact( #EnMovimiento_Horquillado )
   END_RUNG wire#w4
   // the same network as SCL:
   #TOut_Horquillado(IN := (#MA_CogerCarga OR #MA_DejarCarga OR "ON") AND #EnMovimiento_Horquillado AND (NOT #EstadoZona.Manual_CBx OR "ON"),   // "FB910_CNT_UHS"
                     R := NOT #EnMovimiento_Horquillado,
                     PV := #V_TOut_Horquillado,
                     BaseUnidades_ms := "CTE_BaseUnidades_1ms");
END_REGION

REGION Network 39: ERROR - TimeOut de Horqillado - Abriendo la Horquilla
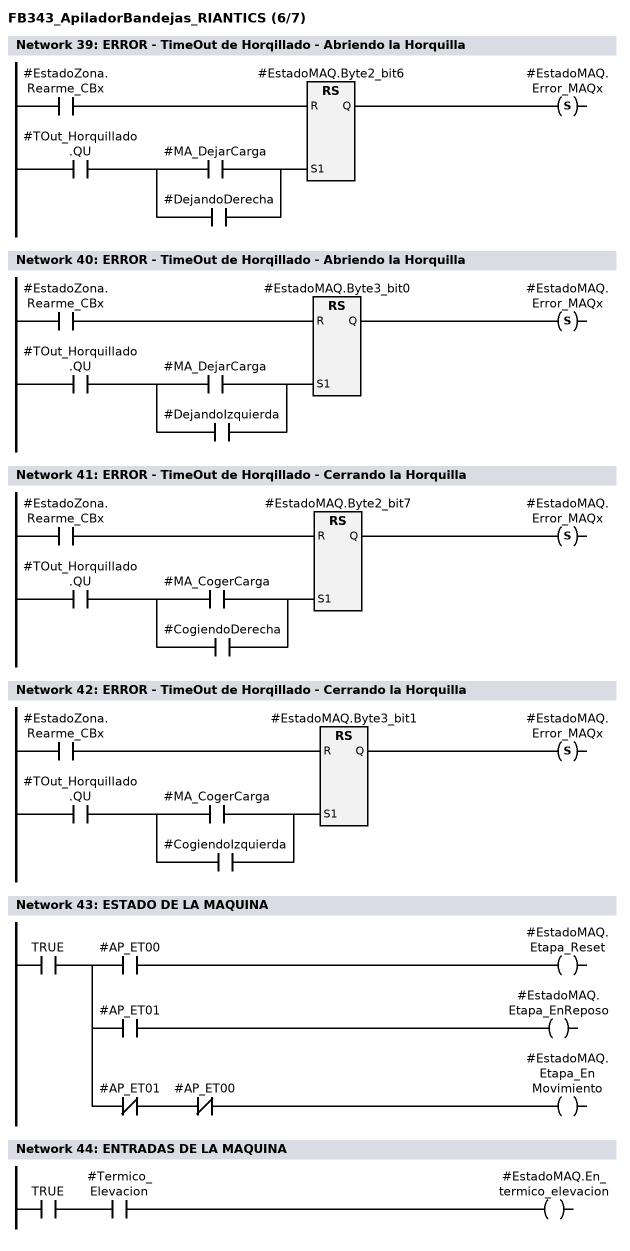
   RUNG wire#powerrail
      Contact( #EstadoZona.Rearme_CBx )
      S_RS(operand := #EstadoMAQ.Byte2_bit6, s1 := wire#w2)
      S_Coil( #EstadoMAQ.Error_MAQx )
   END_RUNG
   RUNG wire#powerrail
      Contact( #TOut_Horquillado.QU )
      wire#w1
      Contact( #MA_DejarCarga )
   END_RUNG wire#w2
   RUNG wire#w1
      Contact( #DejandoDerecha )
   END_RUNG wire#w2
   // the same network as SCL:
   IF #EstadoZona.Rearme_CBx THEN
       #EstadoMAQ.Byte2_bit6 := FALSE;   // RS flip-flop
   END_IF;
   IF #TOut_Horquillado.QU AND (#MA_DejarCarga OR #DejandoDerecha) THEN
       #EstadoMAQ.Byte2_bit6 := TRUE;
   END_IF;
   IF #EstadoMAQ.Byte2_bit6 THEN #EstadoMAQ.Error_MAQx := TRUE; END_IF;
END_REGION

REGION Network 40: ERROR - TimeOut de Horqillado - Abriendo la Horquilla
   RUNG wire#powerrail
      Contact( #EstadoZona.Rearme_CBx )
      S_RS(operand := #EstadoMAQ.Byte3_bit0, s1 := wire#w2)
      S_Coil( #EstadoMAQ.Error_MAQx )
   END_RUNG
   RUNG wire#powerrail
      Contact( #TOut_Horquillado.QU )
      wire#w1
      Contact( #MA_DejarCarga )
   END_RUNG wire#w2
   RUNG wire#w1
      Contact( #DejandoIzquierda )
   END_RUNG wire#w2
   // the same network as SCL:
   IF #EstadoZona.Rearme_CBx THEN
       #EstadoMAQ.Byte3_bit0 := FALSE;   // RS flip-flop
   END_IF;
   IF #TOut_Horquillado.QU AND (#MA_DejarCarga OR #DejandoIzquierda) THEN
       #EstadoMAQ.Byte3_bit0 := TRUE;
   END_IF;
   IF #EstadoMAQ.Byte3_bit0 THEN #EstadoMAQ.Error_MAQx := TRUE; END_IF;
END_REGION

REGION Network 41: ERROR - TimeOut de Horqillado - Cerrando la Horquilla
   RUNG wire#powerrail
      Contact( #EstadoZona.Rearme_CBx )
      S_RS(operand := #EstadoMAQ.Byte2_bit7, s1 := wire#w2)
      S_Coil( #EstadoMAQ.Error_MAQx )
   END_RUNG
   RUNG wire#powerrail
      Contact( #TOut_Horquillado.QU )
      wire#w1
      Contact( #MA_CogerCarga )
   END_RUNG wire#w2
   RUNG wire#w1
      Contact( #CogiendoDerecha )
   END_RUNG wire#w2
   // the same network as SCL:
   IF #EstadoZona.Rearme_CBx THEN
       #EstadoMAQ.Byte2_bit7 := FALSE;   // RS flip-flop
   END_IF;
   IF #TOut_Horquillado.QU AND (#MA_CogerCarga OR #CogiendoDerecha) THEN
       #EstadoMAQ.Byte2_bit7 := TRUE;
   END_IF;
   IF #EstadoMAQ.Byte2_bit7 THEN #EstadoMAQ.Error_MAQx := TRUE; END_IF;
END_REGION

REGION Network 42: ERROR - TimeOut de Horqillado - Cerrando la Horquilla
   RUNG wire#powerrail
      Contact( #EstadoZona.Rearme_CBx )
      S_RS(operand := #EstadoMAQ.Byte3_bit1, s1 := wire#w2)
      S_Coil( #EstadoMAQ.Error_MAQx )
   END_RUNG
   RUNG wire#powerrail
      Contact( #TOut_Horquillado.QU )
      wire#w1
      Contact( #MA_CogerCarga )
   END_RUNG wire#w2
   RUNG wire#w1
      Contact( #CogiendoIzquierda )
   END_RUNG wire#w2
   // the same network as SCL:
   IF #EstadoZona.Rearme_CBx THEN
       #EstadoMAQ.Byte3_bit1 := FALSE;   // RS flip-flop
   END_IF;
   IF #TOut_Horquillado.QU AND (#MA_CogerCarga OR #CogiendoIzquierda) THEN
       #EstadoMAQ.Byte3_bit1 := TRUE;
   END_IF;
   IF #EstadoMAQ.Byte3_bit1 THEN #EstadoMAQ.Error_MAQx := TRUE; END_IF;
END_REGION

REGION Network 43: ESTADO DE LA MAQUINA
   RUNG wire#powerrail
      Contact( TRUE )
      wire#w1
      Contact( #AP_ET00 )
      Coil( #EstadoMAQ.Etapa_Reset )
   END_RUNG
   RUNG wire#w1
      Contact( #AP_ET01 )
      Coil( #EstadoMAQ.Etapa_EnReposo )
   END_RUNG
   RUNG wire#w1
      I_Contact( #AP_ET01 )
      I_Contact( #AP_ET00 )
      Coil( #EstadoMAQ.Etapa_EnMovimiento )
   END_RUNG
   // the same network as SCL:
   #EstadoMAQ.Etapa_Reset := TRUE AND #AP_ET00;
   #EstadoMAQ.Etapa_EnReposo := TRUE AND #AP_ET01;
   #EstadoMAQ.Etapa_EnMovimiento := TRUE AND NOT #AP_ET01 AND NOT #AP_ET00;
END_REGION

REGION Network 44: ENTRADAS DE LA MAQUINA
   RUNG wire#powerrail
      Contact( TRUE )
      Contact( #Termico_Elevacion )
      Coil( #EstadoMAQ.En_termico_elevacion )
   END_RUNG
   // the same network as SCL:
   #EstadoMAQ.En_termico_elevacion := TRUE AND #Termico_Elevacion;
END_REGION

REGION Network 45: ---
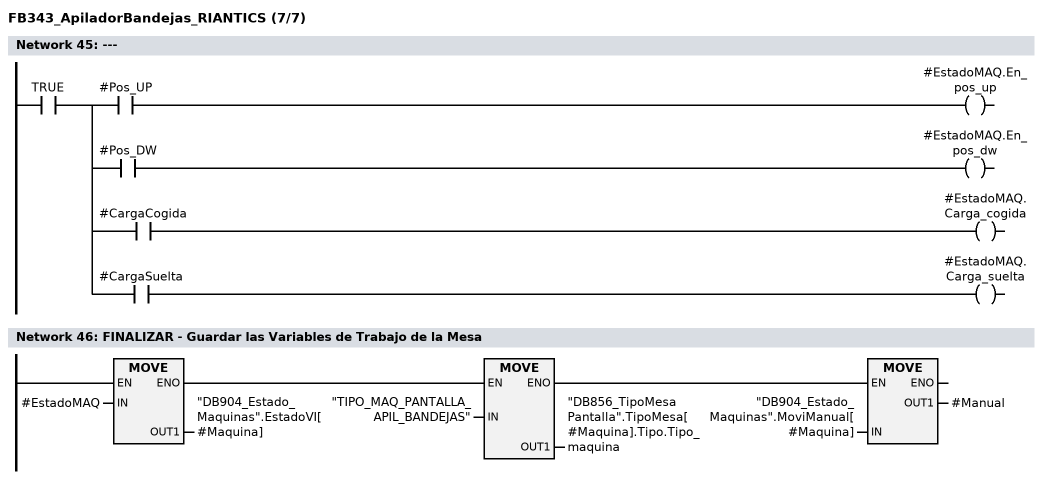
   RUNG wire#powerrail
      Contact( TRUE )
      wire#w1
      Contact( #Pos_UP )
      Coil( #EstadoMAQ.En_pos_up )
   END_RUNG
   RUNG wire#w1
      Contact( #Pos_DW )
      Coil( #EstadoMAQ.En_pos_dw )
   END_RUNG
   RUNG wire#w1
      Contact( #CargaCogida )
      Coil( #EstadoMAQ.Carga_cogida )
   END_RUNG
   RUNG wire#w1
      Contact( #CargaSuelta )
      Coil( #EstadoMAQ.Carga_suelta )
   END_RUNG
   // the same network as SCL:
   #EstadoMAQ.En_pos_up := TRUE AND #Pos_UP;
   #EstadoMAQ.En_pos_dw := TRUE AND #Pos_DW;
   #EstadoMAQ.Carga_cogida := TRUE AND #CargaCogida;
   #EstadoMAQ.Carga_suelta := TRUE AND #CargaSuelta;
END_REGION

REGION Network 46: FINALIZAR - Guardar las Variables de Trabajo de la Mesa
   RUNG wire#powerrail
      Move(in := #EstadoMAQ, out1 => "DB904_Estado_Maquinas".EstadoVI[#Maquina])
      Move(in := "TIPO_MAQ_PANTALLA_APIL_BANDEJAS", out1 => "DB856_TipoMesaPantalla".TipoMesa[#Maquina].Tipo.Tipo_maquina)
      Move(in := "DB904_Estado_Maquinas".MoviManual[#Maquina], out1 => #Manual)
   END_RUNG
   // the same network as SCL:
   "DB904_Estado_Maquinas".EstadoVI[#Maquina] := #EstadoMAQ;
   "DB856_TipoMesaPantalla".TipoMesa[#Maquina].Tipo.Tipo_maquina := "TIPO_MAQ_PANTALLA_APIL_BANDEJAS";
   #Manual := "DB904_Estado_Maquinas".MoviManual[#Maquina];
END_REGION
END_FUNCTION_BLOCK

FUNCTION_BLOCK "FB350_Apilador_DesApilador_Paletas"   // FB350, LAD
TITLE = Control del Ramal de Salidas
{ S7_Optimized_Access := 'FALSE' }
AUTHOR : MAQUINA
NAME : 20181114
VERSION : 3.5
// Dani Palacios: Modificación octubre 2017 para poder desabilitar la maquina con un bit (por ejemplo en la puesta a punto si no esta montada o en el simulador)
// La modificación esta sin probar y es todo lo relativo a la variable Maquina_Desabilitada
// (bloqueo evolución desde etapa 0, bloqueo activación salidas en etapa 0 , fin vi sin mirar detectores y activación posición de reposo sin mirar detectores y variabkles de fin de movimiento).
// ES RESPONSABILIDAD DEL QUE DESABILITA LA MAQUINA QUE ESTA ESTE EN UNA POSICION QUE PERMITA EL MOVIMIENTO DE LAS CARGAS A TRAVES DE ELLA
// stored: AutoNumber false, SetENOAutomatically false
   VAR_INPUT
      Maquina : UInt;   // Numero de Maquina (Mesa)
      Error_Tx : Bool;   // Error en el Tx
      EnTension : Bool;   // Existe Tension en la Mesa
      MAQx_Desabilitada : Bool;   // Config MAQ. >>> DesHabilitada
      MAQx_ReposoDW : Bool;   // Config MAQ. >>> Pos. Reposo Abajo
      Termico_Elevacion : Bool;   // Termico de la Elevacion
      Termico_HorqDch : Bool;   // Termico de la Horquilla Derecha
      Termico_HorqIzq : Bool;   // Termico de la horquilla Izquierda
      pHsMx : Bool;   // pHs de la Mesa
      EnMovimiento_Tx : Bool;   // En Movimiento Tx
      pHs_LlenoApilador : Bool;   // Lleno el Apilador
      pHs_ConCargaApilador : Bool;   // ConCarga Apilador
      EM_UP : Bool;   // Emergencia Arriba del Apilador
      EM_DW : Bool;   // Emergencia Abajo del Apilador
      Pos_Dw : Bool;   // Posición Baja del Apilador
      Pos_Mid : Bool;   // Posición Media del Apilador
      Pos_Up : Bool;   // Posición Alta del Apilador
      Horq1_Der_Recogida : Bool;
      Horq2_Der_Recogida : Bool;
      Horq1_Izq_Recogida : Bool;
      Horq2_Izq_Recogida : Bool;
      Horq1_Der_Extendida : Bool;
      Horq2_Der_Extendida : Bool;
      Horq1_Izq_Extendida : Bool;
      Horq2_Izq_Extendida : Bool;
      EnMovimiento_Elevacion : Bool;   // En Movineto la Elevacion
      EnMovimiento_Horquillado : Bool;   // En Movimiento el Hoquillado
      PasarReposo_Apilador : Bool;   // Pasar a Reposo >>> Interlock Maquina
      CogerPila_Apilador : Bool;   // Coger la Pila >>> Interlock Maquina
      DispensarPaleta_Apilador : Bool;   // Dispensar Paleta >>> Interlock Maquina
      DispensarpPila_Apilador : Bool;   // Dispensar Pila >>> Interlock Maquina
      V_TIM_EstabilidadMov : Time := T#200MS;   // TIM de Estabilidad de los Mov.
      V_TOut_Elevacion : Int := 10000;   // TimeOut del Mov. de Elevacion
      V_TOut_Horquillado : Int := 3000;   // TimeOut del Mov. de Horquillado
   END_VAR
   VAR_OUTPUT
      Quieto_Apilador : Bool;   // Quieto >>> Interlock Maquina
      FinMovimiento_Apilador : Bool;   // Fin Movimiento >>> Interlock Maquina
   END_VAR
   VAR_IN_OUT
      StatusLleno_Apilador : Bool;   // Status Lleno >>> Interlock Maquina
      StatusSemiLleno_Apilador : Bool;   // Status SemiLleno >>> Interlock Maquina
      StatusVacio_Apilador : Bool;   // Status Vacio >>> Interlock Maquina
   END_VAR
   VAR
      Ap_ET00 : Bool;
      Ap_ET100 : Bool;
      Ap_ET101 : Bool;
      Ap_ET102 : Bool;
      Ap_ET103 : Bool;
      Ap_ET104 : Bool;
      Ap_ET105 : Bool;
      Ap_ET106 : Bool;
      Ap_ET107 : Bool;
      Ap_ET108 : Bool;
      Ap_ET109 : Bool;
      Ap_ET11 : Bool;
      Ap_ET12 : Bool;
      Ap_ET13 : Bool;
      Ap_ET14 : Bool;
      Ap_ET15 : Bool;
      Ap_ET16 : Bool;
      Ap_ET21 : Bool;
      Ap_ET22 : Bool;
      Ap_ET23 : Bool;
      Ap_ET24 : Bool;
      Ap_ET31 : Bool;
      Ap_ET32 : Bool;
      Ap_ET41 : Bool;
      Ap_ET42 : Bool;
      Ap_ET43 : Bool;
      Ap_ET44 : Bool;
      Ap_ET50 : Bool;
      Ap_ET51 : Bool;
      PosicionConocida : Bool;   // Interna >> Posicion Conocida
      Apilador_Lleno : Bool;   // Interna >> Lleno el Apilador
      HorquillasRecogidas : Bool;   // Carga Suelta en el Apilador
      HorquillasExtendidas : Bool;   // Carga Cogida en el Apilador
      STAT_FinMovimiento : Bool;   // Interna >> Fin Movimitnto del Apilador
      STAT_Quieto : Bool;   // Interna >> Quieto el Apilador
      CambioDir_SubidaBajada : Bool;   // Interna >> Cambio de Dir. Subida o Bajada
      MA_Ir_Up : Bool;   // ???
      MA_Ir_Dw : Bool;   // ???
      MA_Ir_Mid_Bajando : Bool;   // ???
      MA_Ir_Mid_Subiendo : Bool;   // ???
      MA_DejarCarga : Bool;   // ???
      MA_CogerCarga : Bool;   // ???
      TIM_EstabilidadMov { S7_SetPoint := 'True'} : TON_TIME;
      TMP_EnTension { S7_SetPoint := 'True'} : "FB910_CNT_UHS";
      TOut_Elevacion { S7_SetPoint := 'True'} : "FB910_CNT_UHS";
      TOut_Horquillado { S7_SetPoint := 'True'} : "FB910_CNT_UHS";
      Manual : "MoviManualMaquina_DesApilador";
   END_VAR
   VAR_TEMP
      EstadoZona : "EstadoZona";   // Estado de Zona de la Mesa
      EstadoMAQ : "EstadoMaquina_ApiladorDesapilador";   // Estado del Vehiculo Inteliguente de la Maquina
      Aux_ET00 : Bool;
   END_VAR
   VAR_TEMP   // added for the SCL form of the ladder/FBD networks
      _w1 : Bool;
   END_VAR
BEGIN

REGION Network 1: INICIALIZAR - Recoger las Variables de Estado de la Maquina
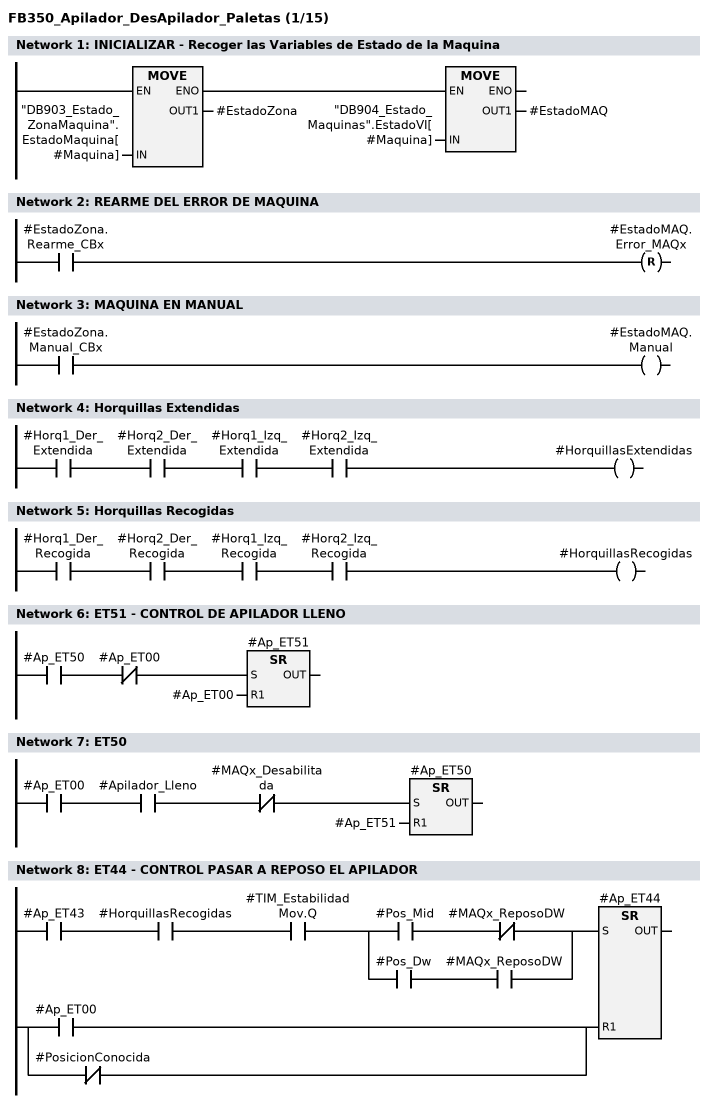
   RUNG wire#powerrail
      Move(in := "DB903_Estado_ZonaMaquina".EstadoMaquina[#Maquina], out1 => #EstadoZona)
      Move(in := "DB904_Estado_Maquinas".EstadoVI[#Maquina], out1 => #EstadoMAQ)
   END_RUNG
   // the same network as SCL:
   #EstadoZona := "DB903_Estado_ZonaMaquina".EstadoMaquina[#Maquina];
   #EstadoMAQ := "DB904_Estado_Maquinas".EstadoVI[#Maquina];
END_REGION

REGION Network 2: REARME DEL ERROR DE MAQUINA
   RUNG wire#powerrail
      Contact( #EstadoZona.Rearme_CBx )
      R_Coil( #EstadoMAQ.Error_MAQx )
   END_RUNG
   // the same network as SCL:
   IF #EstadoZona.Rearme_CBx THEN #EstadoMAQ.Error_MAQx := FALSE; END_IF;
END_REGION

REGION Network 3: MAQUINA EN MANUAL
   RUNG wire#powerrail
      Contact( #EstadoZona.Manual_CBx )
      Coil( #EstadoMAQ.Manual )
   END_RUNG
   // the same network as SCL:
   #EstadoMAQ.Manual := #EstadoZona.Manual_CBx;
END_REGION

REGION Network 4: Horquillas Extendidas
   RUNG wire#powerrail
      Contact( #Horq1_Der_Extendida )
      Contact( #Horq2_Der_Extendida )
      Contact( #Horq1_Izq_Extendida )
      Contact( #Horq2_Izq_Extendida )
      Coil( #HorquillasExtendidas )
   END_RUNG
   // the same network as SCL:
   #HorquillasExtendidas := #Horq1_Der_Extendida AND #Horq2_Der_Extendida AND #Horq1_Izq_Extendida AND #Horq2_Izq_Extendida;
END_REGION

REGION Network 5: Horquillas Recogidas
   RUNG wire#powerrail
      Contact( #Horq1_Der_Recogida )
      Contact( #Horq2_Der_Recogida )
      Contact( #Horq1_Izq_Recogida )
      Contact( #Horq2_Izq_Recogida )
      Coil( #HorquillasRecogidas )
   END_RUNG
   // the same network as SCL:
   #HorquillasRecogidas := #Horq1_Der_Recogida AND #Horq2_Der_Recogida AND #Horq1_Izq_Recogida AND #Horq2_Izq_Recogida;
END_REGION

REGION Network 6: ET51 - CONTROL DE APILADOR LLENO
   RUNG wire#powerrail
      Contact( #Ap_ET50 )
      I_Contact( #Ap_ET00 )
      S_SR(operand := #Ap_ET51, r1 := #Ap_ET00)
   END_RUNG
   // the same network as SCL:
   IF #Ap_ET50 AND NOT #Ap_ET00 THEN
       #Ap_ET51 := TRUE;   // SR flip-flop
   END_IF;
   IF #Ap_ET00 THEN #Ap_ET51 := FALSE; END_IF;
END_REGION

REGION Network 7: ET50
   RUNG wire#powerrail
      Contact( #Ap_ET00 )
      Contact( #Apilador_Lleno )
      I_Contact( #MAQx_Desabilitada )
      S_SR(operand := #Ap_ET50, r1 := #Ap_ET51)
   END_RUNG
   // the same network as SCL:
   IF #Ap_ET00 AND #Apilador_Lleno AND NOT #MAQx_Desabilitada THEN
       #Ap_ET50 := TRUE;   // SR flip-flop
   END_IF;
   IF #Ap_ET51 THEN #Ap_ET50 := FALSE; END_IF;
END_REGION

REGION Network 8: ET44 - CONTROL PASAR A REPOSO EL APILADOR
   RUNG wire#powerrail
      Contact( #Ap_ET43 )
      Contact( #HorquillasRecogidas )
      Contact( #TIM_EstabilidadMov.Q )
      wire#w1
      Contact( #Pos_Mid )
      I_Contact( #MAQx_ReposoDW )
      wire#w2
      S_SR(operand := #Ap_ET44, r1 := wire#w3)
   END_RUNG
   RUNG wire#w1
      Contact( #Pos_Dw )
      Contact( #MAQx_ReposoDW )
   END_RUNG wire#w2
   RUNG wire#powerrail
      Contact( #Ap_ET00 )
   END_RUNG wire#w3
   RUNG wire#powerrail
      I_Contact( #PosicionConocida )
   END_RUNG wire#w3
   // the same network as SCL:
   IF #Ap_ET43 AND #HorquillasRecogidas AND #TIM_EstabilidadMov.Q AND ((#Pos_Mid AND NOT #MAQx_ReposoDW) OR (#Pos_Dw AND #MAQx_ReposoDW)) THEN
       #Ap_ET44 := TRUE;   // SR flip-flop
   END_IF;
   IF #Ap_ET00 OR NOT #PosicionConocida THEN #Ap_ET44 := FALSE; END_IF;
END_REGION

REGION Network 9: ET43
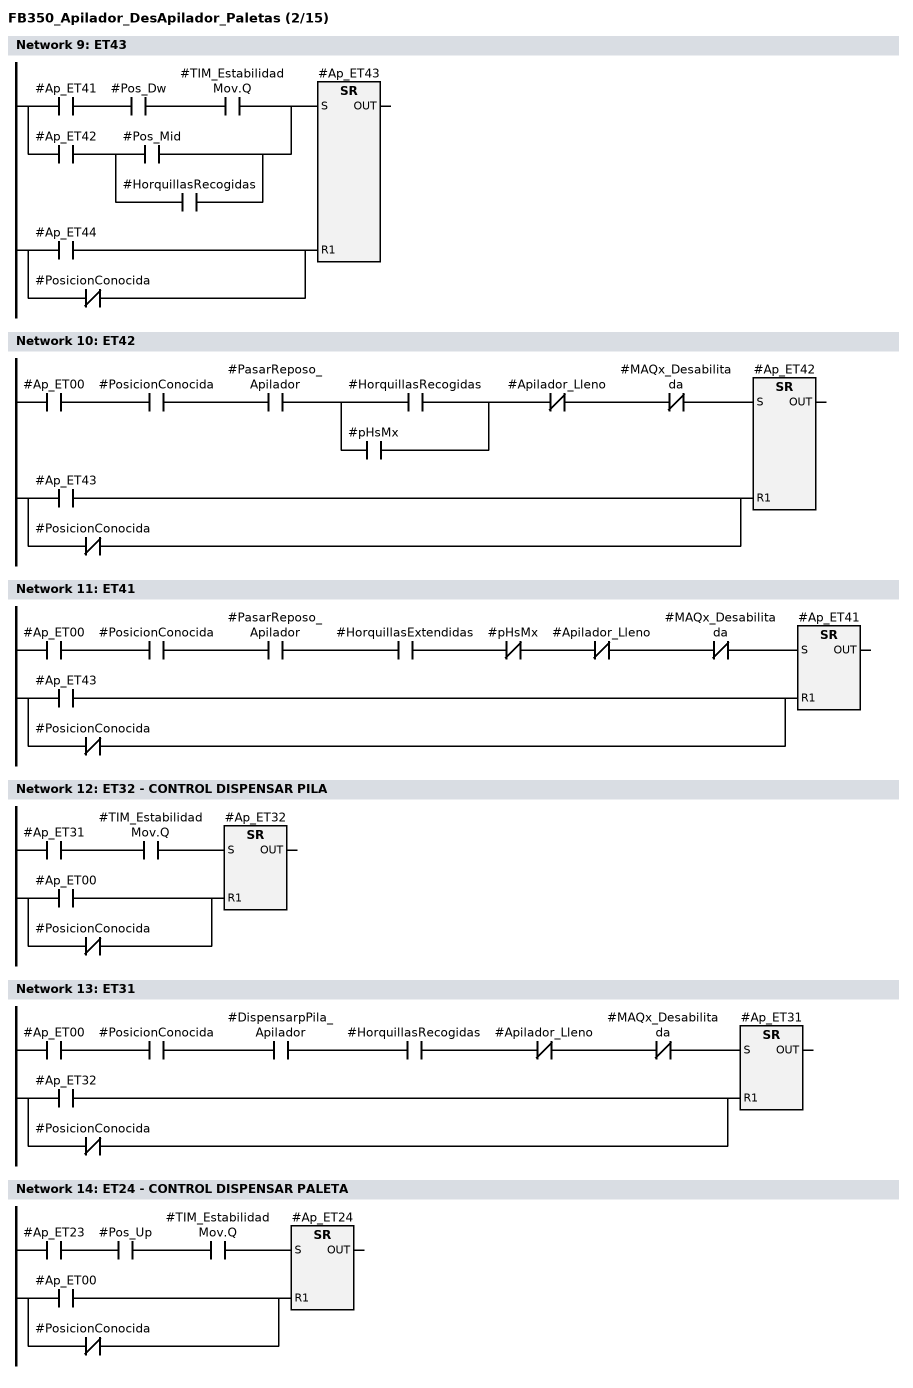
   RUNG wire#powerrail
      Contact( #Ap_ET41 )
      Contact( #Pos_Dw )
      Contact( #TIM_EstabilidadMov.Q )
      wire#w1
      S_SR(operand := #Ap_ET43, r1 := wire#w3)
   END_RUNG
   RUNG wire#powerrail
      Contact( #Ap_ET42 )
      wire#w2
      Contact( #Pos_Mid )
   END_RUNG wire#w1
   RUNG wire#w2
      Contact( #HorquillasRecogidas )
   END_RUNG wire#w1
   RUNG wire#powerrail
      Contact( #Ap_ET44 )
   END_RUNG wire#w3
   RUNG wire#powerrail
      I_Contact( #PosicionConocida )
   END_RUNG wire#w3
   // the same network as SCL:
   IF (#Ap_ET41 AND #Pos_Dw AND #TIM_EstabilidadMov.Q) OR (#Ap_ET42 AND (#Pos_Mid OR #HorquillasRecogidas)) THEN
       #Ap_ET43 := TRUE;   // SR flip-flop
   END_IF;
   IF #Ap_ET44 OR NOT #PosicionConocida THEN #Ap_ET43 := FALSE; END_IF;
END_REGION

REGION Network 10: ET42
   RUNG wire#powerrail
      Contact( #Ap_ET00 )
      Contact( #PosicionConocida )
      Contact( #PasarReposo_Apilador )
      wire#w1
      Contact( #HorquillasRecogidas )
      wire#w2
      I_Contact( #Apilador_Lleno )
      I_Contact( #MAQx_Desabilitada )
      S_SR(operand := #Ap_ET42, r1 := wire#w3)
   END_RUNG
   RUNG wire#w1
      Contact( #pHsMx )
   END_RUNG wire#w2
   RUNG wire#powerrail
      Contact( #Ap_ET43 )
   END_RUNG wire#w3
   RUNG wire#powerrail
      I_Contact( #PosicionConocida )
   END_RUNG wire#w3
   // the same network as SCL:
   IF #Ap_ET00 AND #PosicionConocida AND #PasarReposo_Apilador AND (#HorquillasRecogidas OR #pHsMx) AND NOT #Apilador_Lleno AND NOT #MAQx_Desabilitada THEN
       #Ap_ET42 := TRUE;   // SR flip-flop
   END_IF;
   IF #Ap_ET43 OR NOT #PosicionConocida THEN #Ap_ET42 := FALSE; END_IF;
END_REGION

REGION Network 11: ET41
   RUNG wire#powerrail
      Contact( #Ap_ET00 )
      Contact( #PosicionConocida )
      Contact( #PasarReposo_Apilador )
      Contact( #HorquillasExtendidas )
      I_Contact( #pHsMx )
      I_Contact( #Apilador_Lleno )
      I_Contact( #MAQx_Desabilitada )
      S_SR(operand := #Ap_ET41, r1 := wire#w1)
   END_RUNG
   RUNG wire#powerrail
      Contact( #Ap_ET43 )
   END_RUNG wire#w1
   RUNG wire#powerrail
      I_Contact( #PosicionConocida )
   END_RUNG wire#w1
   // the same network as SCL:
   IF #Ap_ET00 AND #PosicionConocida AND #PasarReposo_Apilador AND #HorquillasExtendidas AND NOT #pHsMx AND NOT #Apilador_Lleno AND NOT #MAQx_Desabilitada THEN
       #Ap_ET41 := TRUE;   // SR flip-flop
   END_IF;
   IF #Ap_ET43 OR NOT #PosicionConocida THEN #Ap_ET41 := FALSE; END_IF;
END_REGION

REGION Network 12: ET32 - CONTROL DISPENSAR PILA
   RUNG wire#powerrail
      Contact( #Ap_ET31 )
      Contact( #TIM_EstabilidadMov.Q )
      S_SR(operand := #Ap_ET32, r1 := wire#w1)
   END_RUNG
   RUNG wire#powerrail
      Contact( #Ap_ET00 )
   END_RUNG wire#w1
   RUNG wire#powerrail
      I_Contact( #PosicionConocida )
   END_RUNG wire#w1
   // the same network as SCL:
   IF #Ap_ET31 AND #TIM_EstabilidadMov.Q THEN
       #Ap_ET32 := TRUE;   // SR flip-flop
   END_IF;
   IF #Ap_ET00 OR NOT #PosicionConocida THEN #Ap_ET32 := FALSE; END_IF;
END_REGION

REGION Network 13: ET31
   RUNG wire#powerrail
      Contact( #Ap_ET00 )
      Contact( #PosicionConocida )
      Contact( #DispensarpPila_Apilador )
      Contact( #HorquillasRecogidas )
      I_Contact( #Apilador_Lleno )
      I_Contact( #MAQx_Desabilitada )
      S_SR(operand := #Ap_ET31, r1 := wire#w1)
   END_RUNG
   RUNG wire#powerrail
      Contact( #Ap_ET32 )
   END_RUNG wire#w1
   RUNG wire#powerrail
      I_Contact( #PosicionConocida )
   END_RUNG wire#w1
   // the same network as SCL:
   IF #Ap_ET00 AND #PosicionConocida AND #DispensarpPila_Apilador AND #HorquillasRecogidas AND NOT #Apilador_Lleno AND NOT #MAQx_Desabilitada THEN
       #Ap_ET31 := TRUE;   // SR flip-flop
   END_IF;
   IF #Ap_ET32 OR NOT #PosicionConocida THEN #Ap_ET31 := FALSE; END_IF;
END_REGION

REGION Network 14: ET24 - CONTROL DISPENSAR PALETA
   RUNG wire#powerrail
      Contact( #Ap_ET23 )
      Contact( #Pos_Up )
      Contact( #TIM_EstabilidadMov.Q )
      S_SR(operand := #Ap_ET24, r1 := wire#w1)
   END_RUNG
   RUNG wire#powerrail
      Contact( #Ap_ET00 )
   END_RUNG wire#w1
   RUNG wire#powerrail
      I_Contact( #PosicionConocida )
   END_RUNG wire#w1
   // the same network as SCL:
   IF #Ap_ET23 AND #Pos_Up AND #TIM_EstabilidadMov.Q THEN
       #Ap_ET24 := TRUE;   // SR flip-flop
   END_IF;
   IF #Ap_ET00 OR NOT #PosicionConocida THEN #Ap_ET24 := FALSE; END_IF;
END_REGION

REGION Network 15: ET23
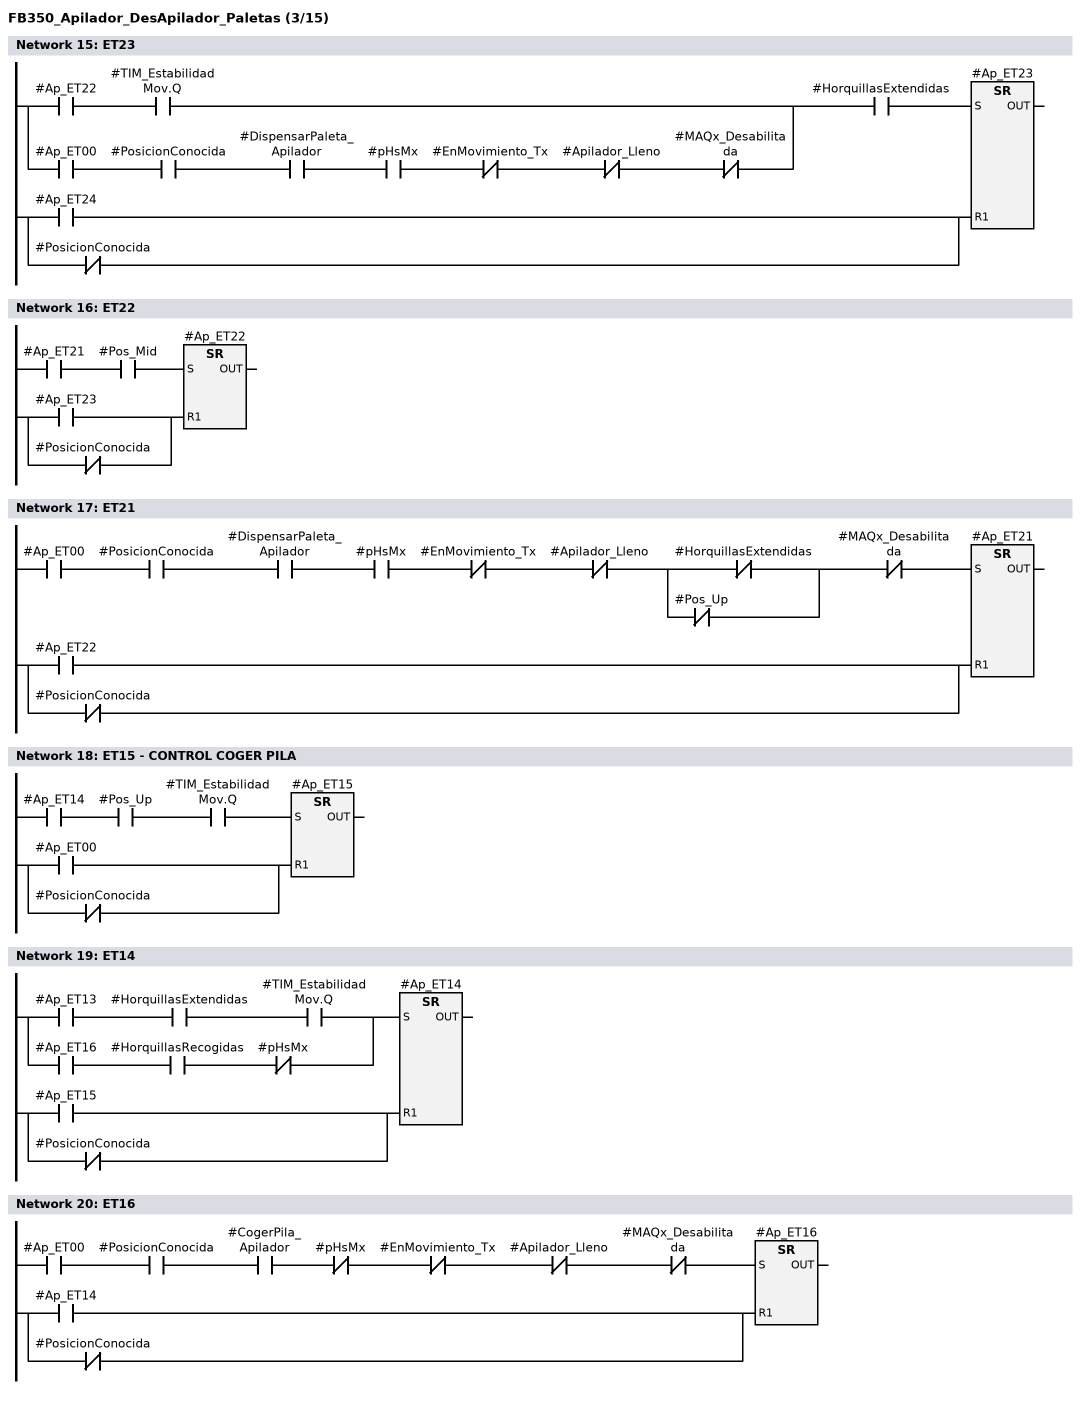
   RUNG wire#powerrail
      Contact( #Ap_ET22 )
      Contact( #TIM_EstabilidadMov.Q )
      wire#w1
      Contact( #HorquillasExtendidas )
      S_SR(operand := #Ap_ET23, r1 := wire#w2)
   END_RUNG
   RUNG wire#powerrail
      Contact( #Ap_ET00 )
      Contact( #PosicionConocida )
      Contact( #DispensarPaleta_Apilador )
      Contact( #pHsMx )
      I_Contact( #EnMovimiento_Tx )
      I_Contact( #Apilador_Lleno )
      I_Contact( #MAQx_Desabilitada )
   END_RUNG wire#w1
   RUNG wire#powerrail
      Contact( #Ap_ET24 )
   END_RUNG wire#w2
   RUNG wire#powerrail
      I_Contact( #PosicionConocida )
   END_RUNG wire#w2
   // the same network as SCL:
   IF ((#Ap_ET22 AND #TIM_EstabilidadMov.Q) OR (#Ap_ET00 AND #PosicionConocida AND #DispensarPaleta_Apilador AND #pHsMx AND NOT #EnMovimiento_Tx AND NOT #Apilador_Lleno AND NOT #MAQx_Desabilitada)) AND #HorquillasExtendidas THEN
       #Ap_ET23 := TRUE;   // SR flip-flop
   END_IF;
   IF #Ap_ET24 OR NOT #PosicionConocida THEN #Ap_ET23 := FALSE; END_IF;
END_REGION

REGION Network 16: ET22
   RUNG wire#powerrail
      Contact( #Ap_ET21 )
      Contact( #Pos_Mid )
      S_SR(operand := #Ap_ET22, r1 := wire#w1)
   END_RUNG
   RUNG wire#powerrail
      Contact( #Ap_ET23 )
   END_RUNG wire#w1
   RUNG wire#powerrail
      I_Contact( #PosicionConocida )
   END_RUNG wire#w1
   // the same network as SCL:
   IF #Ap_ET21 AND #Pos_Mid THEN
       #Ap_ET22 := TRUE;   // SR flip-flop
   END_IF;
   IF #Ap_ET23 OR NOT #PosicionConocida THEN #Ap_ET22 := FALSE; END_IF;
END_REGION

REGION Network 17: ET21
   RUNG wire#powerrail
      Contact( #Ap_ET00 )
      Contact( #PosicionConocida )
      Contact( #DispensarPaleta_Apilador )
      Contact( #pHsMx )
      I_Contact( #EnMovimiento_Tx )
      I_Contact( #Apilador_Lleno )
      wire#w1
      I_Contact( #HorquillasExtendidas )
      wire#w2
      I_Contact( #MAQx_Desabilitada )
      S_SR(operand := #Ap_ET21, r1 := wire#w3)
   END_RUNG
   RUNG wire#w1
      I_Contact( #Pos_Up )
   END_RUNG wire#w2
   RUNG wire#powerrail
      Contact( #Ap_ET22 )
   END_RUNG wire#w3
   RUNG wire#powerrail
      I_Contact( #PosicionConocida )
   END_RUNG wire#w3
   // the same network as SCL:
   IF #Ap_ET00 AND #PosicionConocida AND #DispensarPaleta_Apilador AND #pHsMx AND NOT #EnMovimiento_Tx AND NOT #Apilador_Lleno AND (NOT #HorquillasExtendidas OR NOT #Pos_Up) AND NOT #MAQx_Desabilitada THEN
       #Ap_ET21 := TRUE;   // SR flip-flop
   END_IF;
   IF #Ap_ET22 OR NOT #PosicionConocida THEN #Ap_ET21 := FALSE; END_IF;
END_REGION

REGION Network 18: ET15 - CONTROL COGER PILA
   RUNG wire#powerrail
      Contact( #Ap_ET14 )
      Contact( #Pos_Up )
      Contact( #TIM_EstabilidadMov.Q )
      S_SR(operand := #Ap_ET15, r1 := wire#w1)
   END_RUNG
   RUNG wire#powerrail
      Contact( #Ap_ET00 )
   END_RUNG wire#w1
   RUNG wire#powerrail
      I_Contact( #PosicionConocida )
   END_RUNG wire#w1
   // the same network as SCL:
   IF #Ap_ET14 AND #Pos_Up AND #TIM_EstabilidadMov.Q THEN
       #Ap_ET15 := TRUE;   // SR flip-flop
   END_IF;
   IF #Ap_ET00 OR NOT #PosicionConocida THEN #Ap_ET15 := FALSE; END_IF;
END_REGION

REGION Network 19: ET14
   RUNG wire#powerrail
      Contact( #Ap_ET13 )
      Contact( #HorquillasExtendidas )
      Contact( #TIM_EstabilidadMov.Q )
      wire#w1
      S_SR(operand := #Ap_ET14, r1 := wire#w2)
   END_RUNG
   RUNG wire#powerrail
      Contact( #Ap_ET16 )
      Contact( #HorquillasRecogidas )
      I_Contact( #pHsMx )
   END_RUNG wire#w1
   RUNG wire#powerrail
      Contact( #Ap_ET15 )
   END_RUNG wire#w2
   RUNG wire#powerrail
      I_Contact( #PosicionConocida )
   END_RUNG wire#w2
   // the same network as SCL:
   IF (#Ap_ET13 AND #HorquillasExtendidas AND #TIM_EstabilidadMov.Q) OR (#Ap_ET16 AND #HorquillasRecogidas AND NOT #pHsMx) THEN
       #Ap_ET14 := TRUE;   // SR flip-flop
   END_IF;
   IF #Ap_ET15 OR NOT #PosicionConocida THEN #Ap_ET14 := FALSE; END_IF;
END_REGION

REGION Network 20: ET16
   RUNG wire#powerrail
      Contact( #Ap_ET00 )
      Contact( #PosicionConocida )
      Contact( #CogerPila_Apilador )
      I_Contact( #pHsMx )
      I_Contact( #EnMovimiento_Tx )
      I_Contact( #Apilador_Lleno )
      I_Contact( #MAQx_Desabilitada )
      S_SR(operand := #Ap_ET16, r1 := wire#w1)
   END_RUNG
   RUNG wire#powerrail
      Contact( #Ap_ET14 )
   END_RUNG wire#w1
   RUNG wire#powerrail
      I_Contact( #PosicionConocida )
   END_RUNG wire#w1
   // the same network as SCL:
   IF #Ap_ET00 AND #PosicionConocida AND #CogerPila_Apilador AND NOT #pHsMx AND NOT #EnMovimiento_Tx AND NOT #Apilador_Lleno AND NOT #MAQx_Desabilitada THEN
       #Ap_ET16 := TRUE;   // SR flip-flop
   END_IF;
   IF #Ap_ET14 OR NOT #PosicionConocida THEN #Ap_ET16 := FALSE; END_IF;
END_REGION

REGION Network 21: ET13
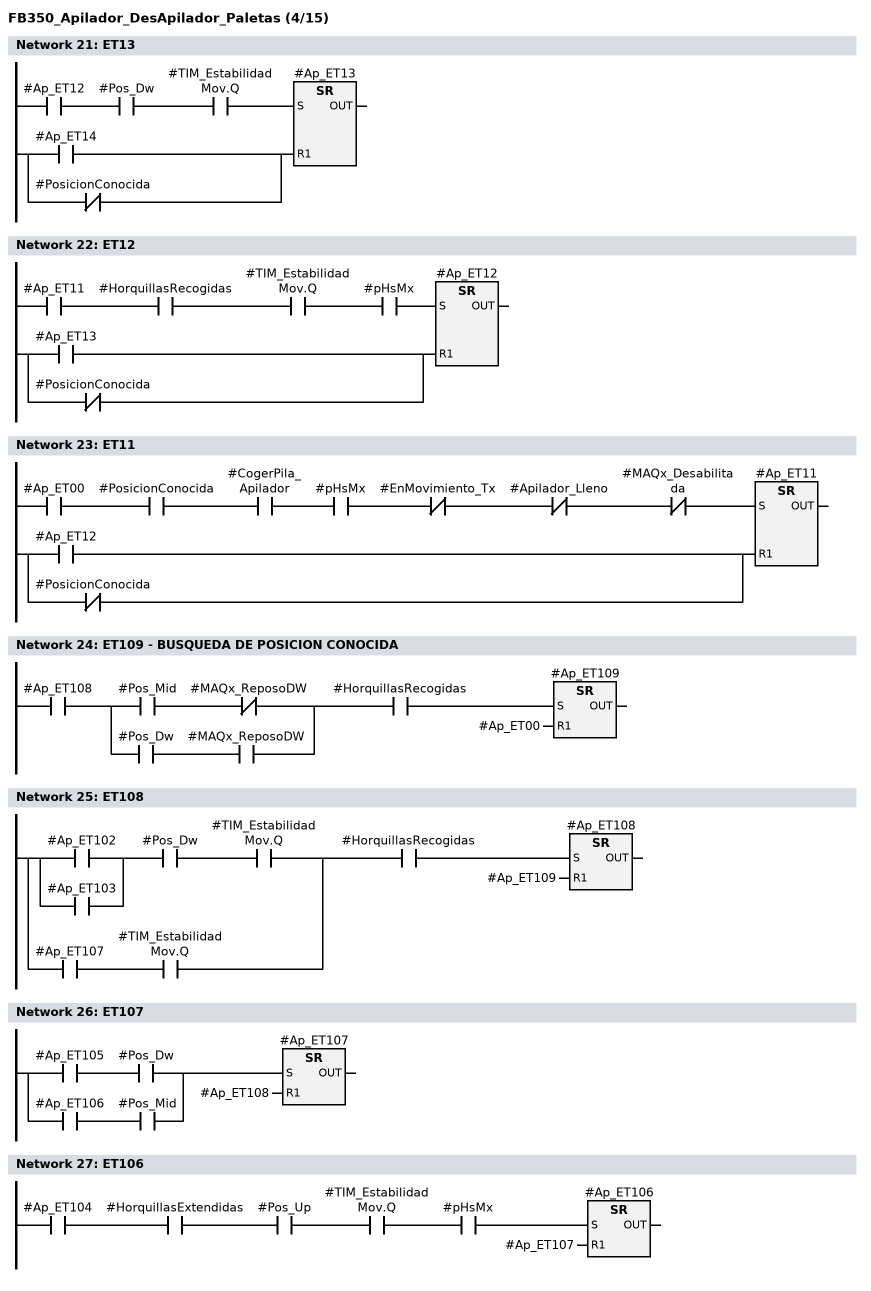
   RUNG wire#powerrail
      Contact( #Ap_ET12 )
      Contact( #Pos_Dw )
      Contact( #TIM_EstabilidadMov.Q )
      S_SR(operand := #Ap_ET13, r1 := wire#w1)
   END_RUNG
   RUNG wire#powerrail
      Contact( #Ap_ET14 )
   END_RUNG wire#w1
   RUNG wire#powerrail
      I_Contact( #PosicionConocida )
   END_RUNG wire#w1
   // the same network as SCL:
   IF #Ap_ET12 AND #Pos_Dw AND #TIM_EstabilidadMov.Q THEN
       #Ap_ET13 := TRUE;   // SR flip-flop
   END_IF;
   IF #Ap_ET14 OR NOT #PosicionConocida THEN #Ap_ET13 := FALSE; END_IF;
END_REGION

REGION Network 22: ET12
   RUNG wire#powerrail
      Contact( #Ap_ET11 )
      Contact( #HorquillasRecogidas )
      Contact( #TIM_EstabilidadMov.Q )
      Contact( #pHsMx )
      S_SR(operand := #Ap_ET12, r1 := wire#w1)
   END_RUNG
   RUNG wire#powerrail
      Contact( #Ap_ET13 )
   END_RUNG wire#w1
   RUNG wire#powerrail
      I_Contact( #PosicionConocida )
   END_RUNG wire#w1
   // the same network as SCL:
   IF #Ap_ET11 AND #HorquillasRecogidas AND #TIM_EstabilidadMov.Q AND #pHsMx THEN
       #Ap_ET12 := TRUE;   // SR flip-flop
   END_IF;
   IF #Ap_ET13 OR NOT #PosicionConocida THEN #Ap_ET12 := FALSE; END_IF;
END_REGION

REGION Network 23: ET11
   RUNG wire#powerrail
      Contact( #Ap_ET00 )
      Contact( #PosicionConocida )
      Contact( #CogerPila_Apilador )
      Contact( #pHsMx )
      I_Contact( #EnMovimiento_Tx )
      I_Contact( #Apilador_Lleno )
      I_Contact( #MAQx_Desabilitada )
      S_SR(operand := #Ap_ET11, r1 := wire#w1)
   END_RUNG
   RUNG wire#powerrail
      Contact( #Ap_ET12 )
   END_RUNG wire#w1
   RUNG wire#powerrail
      I_Contact( #PosicionConocida )
   END_RUNG wire#w1
   // the same network as SCL:
   IF #Ap_ET00 AND #PosicionConocida AND #CogerPila_Apilador AND #pHsMx AND NOT #EnMovimiento_Tx AND NOT #Apilador_Lleno AND NOT #MAQx_Desabilitada THEN
       #Ap_ET11 := TRUE;   // SR flip-flop
   END_IF;
   IF #Ap_ET12 OR NOT #PosicionConocida THEN #Ap_ET11 := FALSE; END_IF;
END_REGION

REGION Network 24: ET109 - BUSQUEDA DE POSICION CONOCIDA
   RUNG wire#powerrail
      Contact( #Ap_ET108 )
      wire#w1
      Contact( #Pos_Mid )
      I_Contact( #MAQx_ReposoDW )
      wire#w2
      Contact( #HorquillasRecogidas )
      S_SR(operand := #Ap_ET109, r1 := #Ap_ET00)
   END_RUNG
   RUNG wire#w1
      Contact( #Pos_Dw )
      Contact( #MAQx_ReposoDW )
   END_RUNG wire#w2
   // the same network as SCL:
   IF #Ap_ET108 AND ((#Pos_Mid AND NOT #MAQx_ReposoDW) OR (#Pos_Dw AND #MAQx_ReposoDW)) AND #HorquillasRecogidas THEN
       #Ap_ET109 := TRUE;   // SR flip-flop
   END_IF;
   IF #Ap_ET00 THEN #Ap_ET109 := FALSE; END_IF;
END_REGION

REGION Network 25: ET108
   RUNG wire#powerrail
      Contact( #Ap_ET102 )
      wire#w1
      Contact( #Pos_Dw )
      Contact( #TIM_EstabilidadMov.Q )
      wire#w2
      Contact( #HorquillasRecogidas )
      S_SR(operand := #Ap_ET108, r1 := #Ap_ET109)
   END_RUNG
   RUNG wire#powerrail
      Contact( #Ap_ET103 )
   END_RUNG wire#w1
   RUNG wire#powerrail
      Contact( #Ap_ET107 )
      Contact( #TIM_EstabilidadMov.Q )
   END_RUNG wire#w2
   // the same network as SCL:
   IF (((#Ap_ET102 OR #Ap_ET103) AND #Pos_Dw AND #TIM_EstabilidadMov.Q) OR (#Ap_ET107 AND #TIM_EstabilidadMov.Q)) AND #HorquillasRecogidas THEN
       #Ap_ET108 := TRUE;   // SR flip-flop
   END_IF;
   IF #Ap_ET109 THEN #Ap_ET108 := FALSE; END_IF;
END_REGION

REGION Network 26: ET107
   RUNG wire#powerrail
      Contact( #Ap_ET105 )
      Contact( #Pos_Dw )
      wire#w1
      S_SR(operand := #Ap_ET107, r1 := #Ap_ET108)
   END_RUNG
   RUNG wire#powerrail
      Contact( #Ap_ET106 )
      Contact( #Pos_Mid )
   END_RUNG wire#w1
   // the same network as SCL:
   IF (#Ap_ET105 AND #Pos_Dw) OR (#Ap_ET106 AND #Pos_Mid) THEN
       #Ap_ET107 := TRUE;   // SR flip-flop
   END_IF;
   IF #Ap_ET108 THEN #Ap_ET107 := FALSE; END_IF;
END_REGION

REGION Network 27: ET106
   RUNG wire#powerrail
      Contact( #Ap_ET104 )
      Contact( #HorquillasExtendidas )
      Contact( #Pos_Up )
      Contact( #TIM_EstabilidadMov.Q )
      Contact( #pHsMx )
      S_SR(operand := #Ap_ET106, r1 := #Ap_ET107)
   END_RUNG
   // the same network as SCL:
   IF #Ap_ET104 AND #HorquillasExtendidas AND #Pos_Up AND #TIM_EstabilidadMov.Q AND #pHsMx THEN
       #Ap_ET106 := TRUE;   // SR flip-flop
   END_IF;
   IF #Ap_ET107 THEN #Ap_ET106 := FALSE; END_IF;
END_REGION

REGION Network 28: ET105
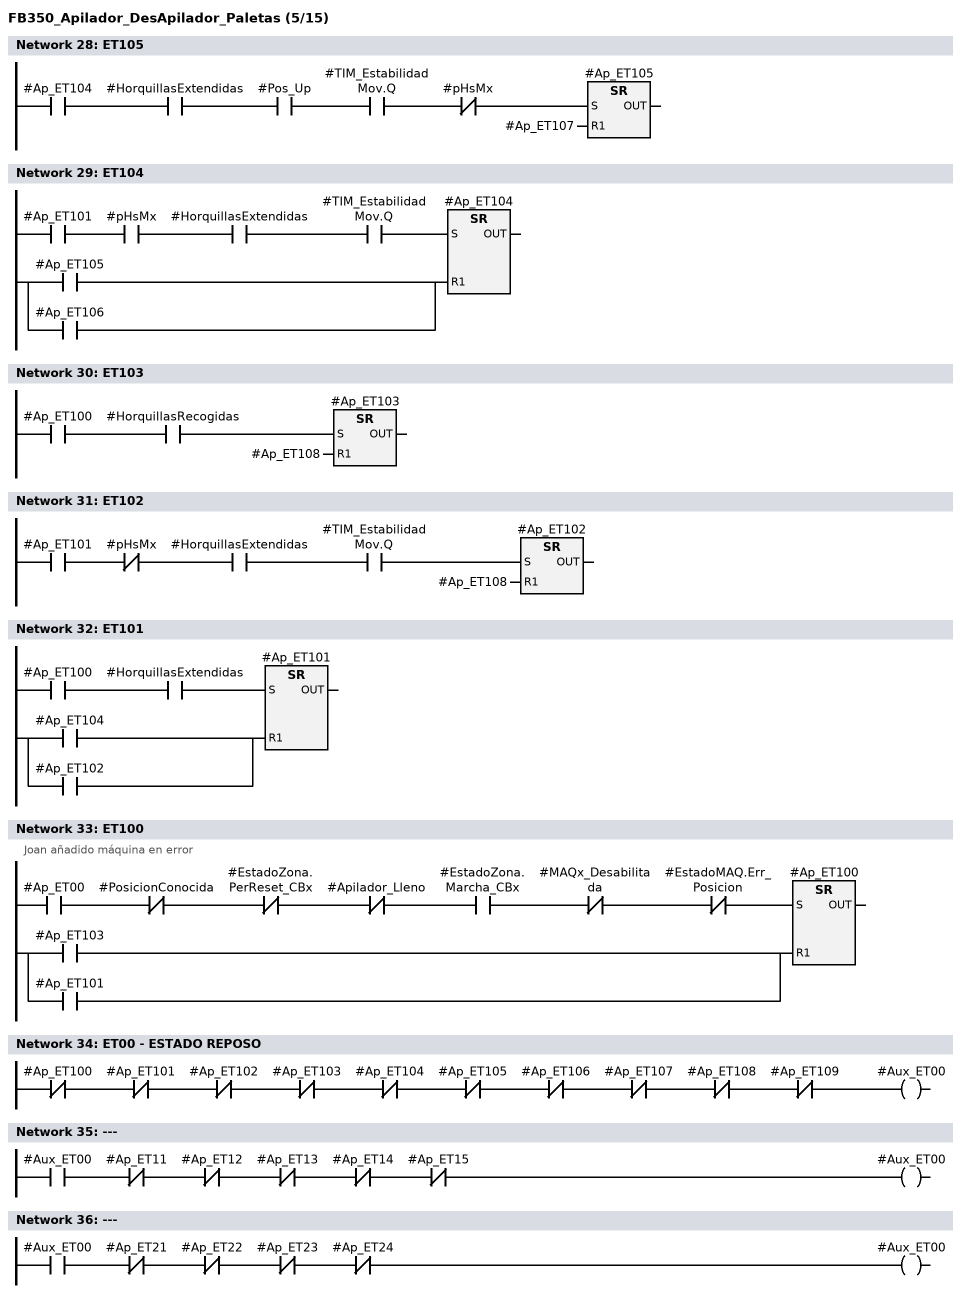
   RUNG wire#powerrail
      Contact( #Ap_ET104 )
      Contact( #HorquillasExtendidas )
      Contact( #Pos_Up )
      Contact( #TIM_EstabilidadMov.Q )
      I_Contact( #pHsMx )
      S_SR(operand := #Ap_ET105, r1 := #Ap_ET107)
   END_RUNG
   // the same network as SCL:
   IF #Ap_ET104 AND #HorquillasExtendidas AND #Pos_Up AND #TIM_EstabilidadMov.Q AND NOT #pHsMx THEN
       #Ap_ET105 := TRUE;   // SR flip-flop
   END_IF;
   IF #Ap_ET107 THEN #Ap_ET105 := FALSE; END_IF;
END_REGION

REGION Network 29: ET104
   RUNG wire#powerrail
      Contact( #Ap_ET101 )
      Contact( #pHsMx )
      Contact( #HorquillasExtendidas )
      Contact( #TIM_EstabilidadMov.Q )
      S_SR(operand := #Ap_ET104, r1 := wire#w1)
   END_RUNG
   RUNG wire#powerrail
      Contact( #Ap_ET105 )
   END_RUNG wire#w1
   RUNG wire#powerrail
      Contact( #Ap_ET106 )
   END_RUNG wire#w1
   // the same network as SCL:
   IF #Ap_ET101 AND #pHsMx AND #HorquillasExtendidas AND #TIM_EstabilidadMov.Q THEN
       #Ap_ET104 := TRUE;   // SR flip-flop
   END_IF;
   IF #Ap_ET105 OR #Ap_ET106 THEN #Ap_ET104 := FALSE; END_IF;
END_REGION

REGION Network 30: ET103
   RUNG wire#powerrail
      Contact( #Ap_ET100 )
      Contact( #HorquillasRecogidas )
      S_SR(operand := #Ap_ET103, r1 := #Ap_ET108)
   END_RUNG
   // the same network as SCL:
   IF #Ap_ET100 AND #HorquillasRecogidas THEN
       #Ap_ET103 := TRUE;   // SR flip-flop
   END_IF;
   IF #Ap_ET108 THEN #Ap_ET103 := FALSE; END_IF;
END_REGION

REGION Network 31: ET102
   RUNG wire#powerrail
      Contact( #Ap_ET101 )
      I_Contact( #pHsMx )
      Contact( #HorquillasExtendidas )
      Contact( #TIM_EstabilidadMov.Q )
      S_SR(operand := #Ap_ET102, r1 := #Ap_ET108)
   END_RUNG
   // the same network as SCL:
   IF #Ap_ET101 AND NOT #pHsMx AND #HorquillasExtendidas AND #TIM_EstabilidadMov.Q THEN
       #Ap_ET102 := TRUE;   // SR flip-flop
   END_IF;
   IF #Ap_ET108 THEN #Ap_ET102 := FALSE; END_IF;
END_REGION

REGION Network 32: ET101
   RUNG wire#powerrail
      Contact( #Ap_ET100 )
      Contact( #HorquillasExtendidas )
      S_SR(operand := #Ap_ET101, r1 := wire#w1)
   END_RUNG
   RUNG wire#powerrail
      Contact( #Ap_ET104 )
   END_RUNG wire#w1
   RUNG wire#powerrail
      Contact( #Ap_ET102 )
   END_RUNG wire#w1
   // the same network as SCL:
   IF #Ap_ET100 AND #HorquillasExtendidas THEN
       #Ap_ET101 := TRUE;   // SR flip-flop
   END_IF;
   IF #Ap_ET104 OR #Ap_ET102 THEN #Ap_ET101 := FALSE; END_IF;
END_REGION

REGION Network 33: ET100
   // Joan añadido máquina en error
   RUNG wire#powerrail
      Contact( #Ap_ET00 )
      I_Contact( #PosicionConocida )
      I_Contact( #EstadoZona.PerReset_CBx )
      I_Contact( #Apilador_Lleno )
      Contact( #EstadoZona.Marcha_CBx )
      I_Contact( #MAQx_Desabilitada )
      I_Contact( #EstadoMAQ.Err_Posicion )
      S_SR(operand := #Ap_ET100, r1 := wire#w1)
   END_RUNG
   RUNG wire#powerrail
      Contact( #Ap_ET103 )
   END_RUNG wire#w1
   RUNG wire#powerrail
      Contact( #Ap_ET101 )
   END_RUNG wire#w1
   // the same network as SCL:
   IF #Ap_ET00 AND NOT #PosicionConocida AND NOT #EstadoZona.PerReset_CBx AND NOT #Apilador_Lleno AND #EstadoZona.Marcha_CBx AND NOT #MAQx_Desabilitada AND NOT #EstadoMAQ.Err_Posicion THEN
       #Ap_ET100 := TRUE;   // SR flip-flop
   END_IF;
   IF #Ap_ET103 OR #Ap_ET101 THEN #Ap_ET100 := FALSE; END_IF;
END_REGION

REGION Network 34: ET00 - ESTADO REPOSO
   RUNG wire#powerrail
      I_Contact( #Ap_ET100 )
      I_Contact( #Ap_ET101 )
      I_Contact( #Ap_ET102 )
      I_Contact( #Ap_ET103 )
      I_Contact( #Ap_ET104 )
      I_Contact( #Ap_ET105 )
      I_Contact( #Ap_ET106 )
      I_Contact( #Ap_ET107 )
      I_Contact( #Ap_ET108 )
      I_Contact( #Ap_ET109 )
      Coil( #Aux_ET00 )
   END_RUNG
   // the same network as SCL:
   #Aux_ET00 := NOT #Ap_ET100 AND NOT #Ap_ET101 AND NOT #Ap_ET102 AND NOT #Ap_ET103 AND NOT #Ap_ET104 AND NOT #Ap_ET105 AND NOT #Ap_ET106 AND NOT #Ap_ET107 AND NOT #Ap_ET108 AND NOT #Ap_ET109;
END_REGION

REGION Network 35: ---
   RUNG wire#powerrail
      Contact( #Aux_ET00 )
      I_Contact( #Ap_ET11 )
      I_Contact( #Ap_ET12 )
      I_Contact( #Ap_ET13 )
      I_Contact( #Ap_ET14 )
      I_Contact( #Ap_ET15 )
      Coil( #Aux_ET00 )
   END_RUNG
   // the same network as SCL:
   #Aux_ET00 := #Aux_ET00 AND NOT #Ap_ET11 AND NOT #Ap_ET12 AND NOT #Ap_ET13 AND NOT #Ap_ET14 AND NOT #Ap_ET15;
END_REGION

REGION Network 36: ---
   RUNG wire#powerrail
      Contact( #Aux_ET00 )
      I_Contact( #Ap_ET21 )
      I_Contact( #Ap_ET22 )
      I_Contact( #Ap_ET23 )
      I_Contact( #Ap_ET24 )
      Coil( #Aux_ET00 )
   END_RUNG
   // the same network as SCL:
   #Aux_ET00 := #Aux_ET00 AND NOT #Ap_ET21 AND NOT #Ap_ET22 AND NOT #Ap_ET23 AND NOT #Ap_ET24;
END_REGION

REGION Network 37: ---
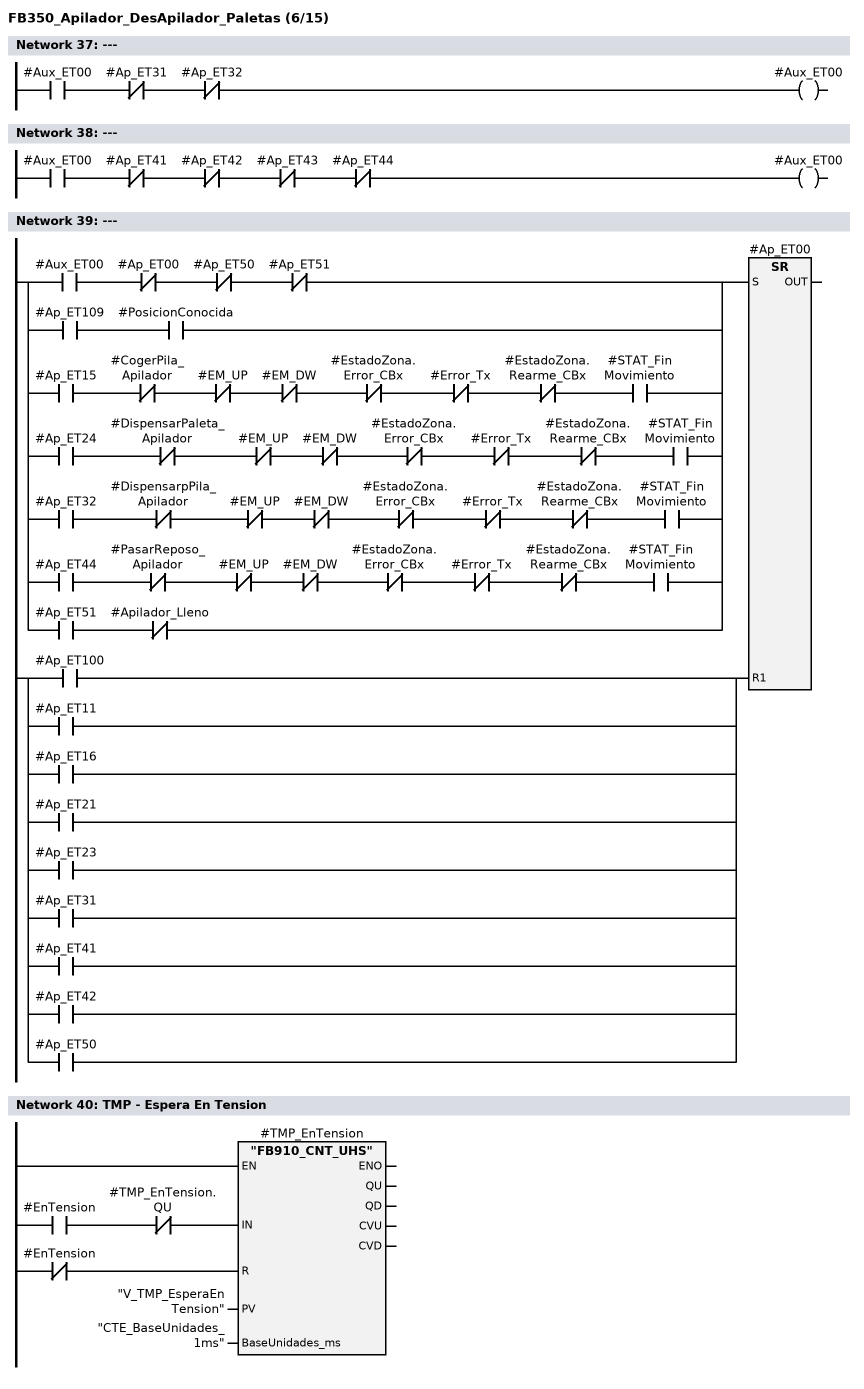
   RUNG wire#powerrail
      Contact( #Aux_ET00 )
      I_Contact( #Ap_ET31 )
      I_Contact( #Ap_ET32 )
      Coil( #Aux_ET00 )
   END_RUNG
   // the same network as SCL:
   #Aux_ET00 := #Aux_ET00 AND NOT #Ap_ET31 AND NOT #Ap_ET32;
END_REGION

REGION Network 38: ---
   RUNG wire#powerrail
      Contact( #Aux_ET00 )
      I_Contact( #Ap_ET41 )
      I_Contact( #Ap_ET42 )
      I_Contact( #Ap_ET43 )
      I_Contact( #Ap_ET44 )
      Coil( #Aux_ET00 )
   END_RUNG
   // the same network as SCL:
   #Aux_ET00 := #Aux_ET00 AND NOT #Ap_ET41 AND NOT #Ap_ET42 AND NOT #Ap_ET43 AND NOT #Ap_ET44;
END_REGION

REGION Network 39: ---
   RUNG wire#powerrail
      Contact( #Aux_ET00 )
      I_Contact( #Ap_ET00 )
      I_Contact( #Ap_ET50 )
      I_Contact( #Ap_ET51 )
      wire#w1
      S_SR(operand := #Ap_ET00, r1 := wire#w2)
   END_RUNG
   RUNG wire#powerrail
      Contact( #Ap_ET109 )
      Contact( #PosicionConocida )
   END_RUNG wire#w1
   RUNG wire#powerrail
      Contact( #Ap_ET15 )
      I_Contact( #CogerPila_Apilador )
      I_Contact( #EM_UP )
      I_Contact( #EM_DW )
      I_Contact( #EstadoZona.Error_CBx )
      I_Contact( #Error_Tx )
      I_Contact( #EstadoZona.Rearme_CBx )
      Contact( #STAT_FinMovimiento )
   END_RUNG wire#w1
   RUNG wire#powerrail
      Contact( #Ap_ET24 )
      I_Contact( #DispensarPaleta_Apilador )
      I_Contact( #EM_UP )
      I_Contact( #EM_DW )
      I_Contact( #EstadoZona.Error_CBx )
      I_Contact( #Error_Tx )
      I_Contact( #EstadoZona.Rearme_CBx )
      Contact( #STAT_FinMovimiento )
   END_RUNG wire#w1
   RUNG wire#powerrail
      Contact( #Ap_ET32 )
      I_Contact( #DispensarpPila_Apilador )
      I_Contact( #EM_UP )
      I_Contact( #EM_DW )
      I_Contact( #EstadoZona.Error_CBx )
      I_Contact( #Error_Tx )
      I_Contact( #EstadoZona.Rearme_CBx )
      Contact( #STAT_FinMovimiento )
   END_RUNG wire#w1
   RUNG wire#powerrail
      Contact( #Ap_ET44 )
      I_Contact( #PasarReposo_Apilador )
      I_Contact( #EM_UP )
      I_Contact( #EM_DW )
      I_Contact( #EstadoZona.Error_CBx )
      I_Contact( #Error_Tx )
      I_Contact( #EstadoZona.Rearme_CBx )
      Contact( #STAT_FinMovimiento )
   END_RUNG wire#w1
   RUNG wire#powerrail
      Contact( #Ap_ET51 )
      I_Contact( #Apilador_Lleno )
   END_RUNG wire#w1
   RUNG wire#powerrail
      Contact( #Ap_ET100 )
   END_RUNG wire#w2
   RUNG wire#powerrail
      Contact( #Ap_ET11 )
   END_RUNG wire#w2
   RUNG wire#powerrail
      Contact( #Ap_ET16 )
   END_RUNG wire#w2
   RUNG wire#powerrail
      Contact( #Ap_ET21 )
   END_RUNG wire#w2
   RUNG wire#powerrail
      Contact( #Ap_ET23 )
   END_RUNG wire#w2
   RUNG wire#powerrail
      Contact( #Ap_ET31 )
   END_RUNG wire#w2
   RUNG wire#powerrail
      Contact( #Ap_ET41 )
   END_RUNG wire#w2
   RUNG wire#powerrail
      Contact( #Ap_ET42 )
   END_RUNG wire#w2
   RUNG wire#powerrail
      Contact( #Ap_ET50 )
   END_RUNG wire#w2
   // the same network as SCL:
   IF (#Aux_ET00 AND NOT #Ap_ET00 AND NOT #Ap_ET50 AND NOT #Ap_ET51) OR (#Ap_ET109 AND #PosicionConocida) OR (#Ap_ET15 AND NOT #CogerPila_Apilador AND NOT #EM_UP AND NOT #EM_DW AND NOT #EstadoZona.Error_CBx AND NOT #Error_Tx AND NOT #EstadoZona.Rearme_CBx AND #STAT_FinMovimiento) OR (#Ap_ET24 AND NOT #DispensarPaleta_Apilador AND NOT #EM_UP AND NOT #EM_DW AND NOT #EstadoZona.Error_CBx AND NOT #Error_Tx AND NOT #EstadoZona.Rearme_CBx AND #STAT_FinMovimiento) OR (#Ap_ET32 AND NOT #DispensarpPila_Apilador AND NOT #EM_UP AND NOT #EM_DW AND NOT #EstadoZona.Error_CBx AND NOT #Error_Tx AND NOT #EstadoZona.Rearme_CBx AND #STAT_FinMovimiento) OR (#Ap_ET44 AND NOT #PasarReposo_Apilador AND NOT #EM_UP AND NOT #EM_DW AND NOT #EstadoZona.Error_CBx AND NOT #Error_Tx AND NOT #EstadoZona.Rearme_CBx AND #STAT_FinMovimiento) OR (#Ap_ET51 AND NOT #Apilador_Lleno) THEN
       #Ap_ET00 := TRUE;   // SR flip-flop
   END_IF;
   IF #Ap_ET100 OR #Ap_ET11 OR #Ap_ET16 OR #Ap_ET21 OR #Ap_ET23 OR #Ap_ET31 OR #Ap_ET41 OR #Ap_ET42 OR #Ap_ET50 THEN
       #Ap_ET00 := FALSE;
   END_IF;
END_REGION

REGION Network 40: TMP - Espera En Tension
   RUNG wire#powerrail
      #TMP_EnTension(IN := wire#w1, R := wire#w2, PV := "V_TMP_EsperaEnTension", BaseUnidades_ms := "CTE_BaseUnidades_1ms", QU =>, QD =>, CVU =>, CVD =>)
   END_RUNG
   RUNG wire#powerrail
      Contact( #EnTension )
      I_Contact( #TMP_EnTension.QU )
   END_RUNG wire#w1
   RUNG wire#powerrail
      I_Contact( #EnTension )
   END_RUNG wire#w2
   // the same network as SCL:
   #TMP_EnTension(IN := #EnTension AND NOT #TMP_EnTension.QU,   // "FB910_CNT_UHS"
                  R := NOT #EnTension,
                  PV := "V_TMP_EsperaEnTension",
                  BaseUnidades_ms := "CTE_BaseUnidades_1ms");
END_REGION

REGION Network 41: ERROR - Termico de Elevacion
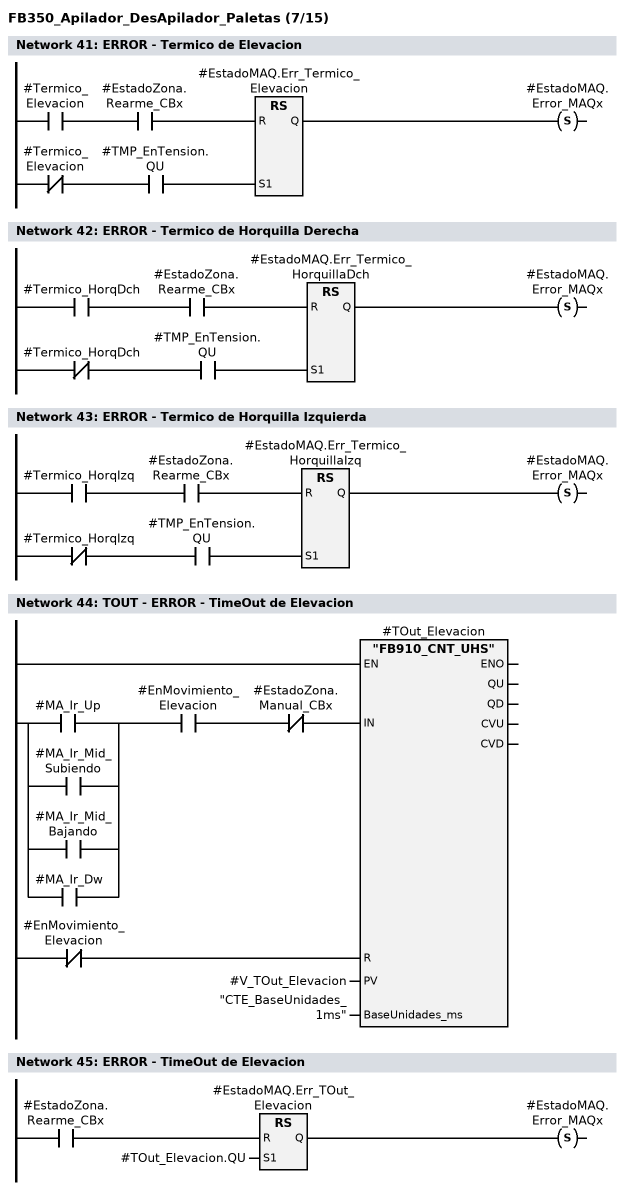
   RUNG wire#powerrail
      Contact( #Termico_Elevacion )
      Contact( #EstadoZona.Rearme_CBx )
      S_RS(operand := #EstadoMAQ.Err_Termico_Elevacion, s1 := wire#w1)
      S_Coil( #EstadoMAQ.Error_MAQx )
   END_RUNG
   RUNG wire#powerrail
      I_Contact( #Termico_Elevacion )
      Contact( #TMP_EnTension.QU )
   END_RUNG wire#w1
   // the same network as SCL:
   IF #Termico_Elevacion AND #EstadoZona.Rearme_CBx THEN
       #EstadoMAQ.Err_Termico_Elevacion := FALSE;   // RS flip-flop
   END_IF;
   IF NOT #Termico_Elevacion AND #TMP_EnTension.QU THEN #EstadoMAQ.Err_Termico_Elevacion := TRUE; END_IF;
   IF #EstadoMAQ.Err_Termico_Elevacion THEN #EstadoMAQ.Error_MAQx := TRUE; END_IF;
END_REGION

REGION Network 42: ERROR - Termico de Horquilla Derecha
   RUNG wire#powerrail
      Contact( #Termico_HorqDch )
      Contact( #EstadoZona.Rearme_CBx )
      S_RS(operand := #EstadoMAQ.Err_Termico_HorquillaDch, s1 := wire#w1)
      S_Coil( #EstadoMAQ.Error_MAQx )
   END_RUNG
   RUNG wire#powerrail
      I_Contact( #Termico_HorqDch )
      Contact( #TMP_EnTension.QU )
   END_RUNG wire#w1
   // the same network as SCL:
   IF #Termico_HorqDch AND #EstadoZona.Rearme_CBx THEN
       #EstadoMAQ.Err_Termico_HorquillaDch := FALSE;   // RS flip-flop
   END_IF;
   IF NOT #Termico_HorqDch AND #TMP_EnTension.QU THEN #EstadoMAQ.Err_Termico_HorquillaDch := TRUE; END_IF;
   IF #EstadoMAQ.Err_Termico_HorquillaDch THEN #EstadoMAQ.Error_MAQx := TRUE; END_IF;
END_REGION

REGION Network 43: ERROR - Termico de Horquilla Izquierda
   RUNG wire#powerrail
      Contact( #Termico_HorqIzq )
      Contact( #EstadoZona.Rearme_CBx )
      S_RS(operand := #EstadoMAQ.Err_Termico_HorquillaIzq, s1 := wire#w1)
      S_Coil( #EstadoMAQ.Error_MAQx )
   END_RUNG
   RUNG wire#powerrail
      I_Contact( #Termico_HorqIzq )
      Contact( #TMP_EnTension.QU )
   END_RUNG wire#w1
   // the same network as SCL:
   IF #Termico_HorqIzq AND #EstadoZona.Rearme_CBx THEN
       #EstadoMAQ.Err_Termico_HorquillaIzq := FALSE;   // RS flip-flop
   END_IF;
   IF NOT #Termico_HorqIzq AND #TMP_EnTension.QU THEN #EstadoMAQ.Err_Termico_HorquillaIzq := TRUE; END_IF;
   IF #EstadoMAQ.Err_Termico_HorquillaIzq THEN #EstadoMAQ.Error_MAQx := TRUE; END_IF;
END_REGION

REGION Network 44: TOUT - ERROR - TimeOut de Elevacion
   RUNG wire#powerrail
      #TOut_Elevacion(IN := wire#w2, R := wire#w3, PV := #V_TOut_Elevacion, BaseUnidades_ms := "CTE_BaseUnidades_1ms", QU =>, QD =>, CVU =>, CVD =>)
   END_RUNG
   RUNG wire#powerrail
      Contact( #MA_Ir_Up )
      wire#w1
      Contact( #EnMovimiento_Elevacion )
      I_Contact( #EstadoZona.Manual_CBx )
   END_RUNG wire#w2
   RUNG wire#powerrail
      Contact( #MA_Ir_Mid_Subiendo )
   END_RUNG wire#w1
   RUNG wire#powerrail
      Contact( #MA_Ir_Mid_Bajando )
   END_RUNG wire#w1
   RUNG wire#powerrail
      Contact( #MA_Ir_Dw )
   END_RUNG wire#w1
   RUNG wire#powerrail
      I_Contact( #EnMovimiento_Elevacion )
   END_RUNG wire#w3
   // the same network as SCL:
   #TOut_Elevacion(IN := (#MA_Ir_Up OR #MA_Ir_Mid_Subiendo OR #MA_Ir_Mid_Bajando OR #MA_Ir_Dw) AND #EnMovimiento_Elevacion AND NOT #EstadoZona.Manual_CBx,   // "FB910_CNT_UHS"
                   R := NOT #EnMovimiento_Elevacion,
                   PV := #V_TOut_Elevacion,
                   BaseUnidades_ms := "CTE_BaseUnidades_1ms");
END_REGION

REGION Network 45: ERROR - TimeOut de Elevacion
   RUNG wire#powerrail
      Contact( #EstadoZona.Rearme_CBx )
      S_RS(operand := #EstadoMAQ.Err_TOut_Elevacion, s1 := #TOut_Elevacion.QU)
      S_Coil( #EstadoMAQ.Error_MAQx )
   END_RUNG
   // the same network as SCL:
   IF #EstadoZona.Rearme_CBx THEN
       #EstadoMAQ.Err_TOut_Elevacion := FALSE;   // RS flip-flop
   END_IF;
   IF #TOut_Elevacion.QU THEN #EstadoMAQ.Err_TOut_Elevacion := TRUE; END_IF;
   IF #EstadoMAQ.Err_TOut_Elevacion THEN #EstadoMAQ.Error_MAQx := TRUE; END_IF;
END_REGION

REGION Network 46: TOUT - ERROR - TimeOut de Horqillado - Abriendo o Cerrando la Horquilla
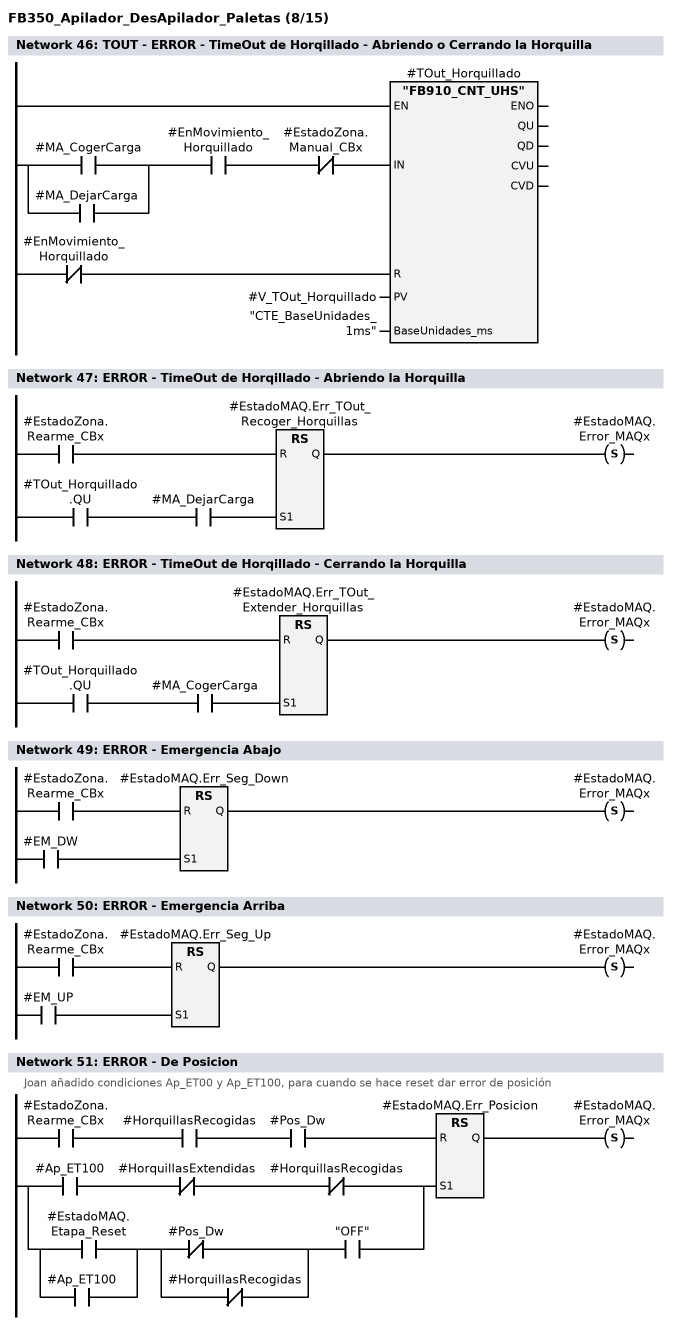
   RUNG wire#powerrail
      #TOut_Horquillado(IN := wire#w2, R := wire#w3, PV := #V_TOut_Horquillado, BaseUnidades_ms := "CTE_BaseUnidades_1ms", QU =>, QD =>, CVU =>, CVD =>)
   END_RUNG
   RUNG wire#powerrail
      Contact( #MA_CogerCarga )
      wire#w1
      Contact( #EnMovimiento_Horquillado )
      I_Contact( #EstadoZona.Manual_CBx )
   END_RUNG wire#w2
   RUNG wire#powerrail
      Contact( #MA_DejarCarga )
   END_RUNG wire#w1
   RUNG wire#powerrail
      I_Contact( #EnMovimiento_Horquillado )
   END_RUNG wire#w3
   // the same network as SCL:
   #TOut_Horquillado(IN := (#MA_CogerCarga OR #MA_DejarCarga) AND #EnMovimiento_Horquillado AND NOT #EstadoZona.Manual_CBx,   // "FB910_CNT_UHS"
                     R := NOT #EnMovimiento_Horquillado,
                     PV := #V_TOut_Horquillado,
                     BaseUnidades_ms := "CTE_BaseUnidades_1ms");
END_REGION

REGION Network 47: ERROR - TimeOut de Horqillado - Abriendo la Horquilla
   RUNG wire#powerrail
      Contact( #EstadoZona.Rearme_CBx )
      S_RS(operand := #EstadoMAQ.Err_TOut_Recoger_Horquillas, s1 := wire#w1)
      S_Coil( #EstadoMAQ.Error_MAQx )
   END_RUNG
   RUNG wire#powerrail
      Contact( #TOut_Horquillado.QU )
      Contact( #MA_DejarCarga )
   END_RUNG wire#w1
   // the same network as SCL:
   IF #EstadoZona.Rearme_CBx THEN
       #EstadoMAQ.Err_TOut_Recoger_Horquillas := FALSE;   // RS flip-flop
   END_IF;
   IF #TOut_Horquillado.QU AND #MA_DejarCarga THEN #EstadoMAQ.Err_TOut_Recoger_Horquillas := TRUE; END_IF;
   IF #EstadoMAQ.Err_TOut_Recoger_Horquillas THEN #EstadoMAQ.Error_MAQx := TRUE; END_IF;
END_REGION

REGION Network 48: ERROR - TimeOut de Horqillado - Cerrando la Horquilla
   RUNG wire#powerrail
      Contact( #EstadoZona.Rearme_CBx )
      S_RS(operand := #EstadoMAQ.Err_TOut_Extender_Horquillas, s1 := wire#w1)
      S_Coil( #EstadoMAQ.Error_MAQx )
   END_RUNG
   RUNG wire#powerrail
      Contact( #TOut_Horquillado.QU )
      Contact( #MA_CogerCarga )
   END_RUNG wire#w1
   // the same network as SCL:
   IF #EstadoZona.Rearme_CBx THEN
       #EstadoMAQ.Err_TOut_Extender_Horquillas := FALSE;   // RS flip-flop
   END_IF;
   IF #TOut_Horquillado.QU AND #MA_CogerCarga THEN #EstadoMAQ.Err_TOut_Extender_Horquillas := TRUE; END_IF;
   IF #EstadoMAQ.Err_TOut_Extender_Horquillas THEN #EstadoMAQ.Error_MAQx := TRUE; END_IF;
END_REGION

REGION Network 49: ERROR - Emergencia Abajo
   RUNG wire#powerrail
      Contact( #EstadoZona.Rearme_CBx )
      S_RS(operand := #EstadoMAQ.Err_Seg_Down, s1 := wire#w1)
      S_Coil( #EstadoMAQ.Error_MAQx )
   END_RUNG
   RUNG wire#powerrail
      Contact( #EM_DW )
   END_RUNG wire#w1
   // the same network as SCL:
   IF #EstadoZona.Rearme_CBx THEN
       #EstadoMAQ.Err_Seg_Down := FALSE;   // RS flip-flop
   END_IF;
   IF #EM_DW THEN #EstadoMAQ.Err_Seg_Down := TRUE; END_IF;
   IF #EstadoMAQ.Err_Seg_Down THEN #EstadoMAQ.Error_MAQx := TRUE; END_IF;
END_REGION

REGION Network 50: ERROR - Emergencia Arriba
   RUNG wire#powerrail
      Contact( #EstadoZona.Rearme_CBx )
      S_RS(operand := #EstadoMAQ.Err_Seg_Up, s1 := wire#w1)
      S_Coil( #EstadoMAQ.Error_MAQx )
   END_RUNG
   RUNG wire#powerrail
      Contact( #EM_UP )
   END_RUNG wire#w1
   // the same network as SCL:
   IF #EstadoZona.Rearme_CBx THEN
       #EstadoMAQ.Err_Seg_Up := FALSE;   // RS flip-flop
   END_IF;
   IF #EM_UP THEN #EstadoMAQ.Err_Seg_Up := TRUE; END_IF;
   IF #EstadoMAQ.Err_Seg_Up THEN #EstadoMAQ.Error_MAQx := TRUE; END_IF;
END_REGION

REGION Network 51: ERROR - De Posicion
   // Joan añadido condiciones Ap_ET00 y Ap_ET100, para cuando se hace reset dar error de posición
   RUNG wire#powerrail
      Contact( #EstadoZona.Rearme_CBx )
      Contact( #HorquillasRecogidas )
      Contact( #Pos_Dw )
      S_RS(operand := #EstadoMAQ.Err_Posicion, s1 := wire#w3)
      S_Coil( #EstadoMAQ.Error_MAQx )
   END_RUNG
   RUNG wire#powerrail
      Contact( #Ap_ET100 )
      I_Contact( #HorquillasExtendidas )
      I_Contact( #HorquillasRecogidas )
   END_RUNG wire#w3
   RUNG wire#powerrail
      Contact( #EstadoMAQ.Etapa_Reset )
      wire#w1
      I_Contact( #Pos_Dw )
      wire#w2
      Contact( "OFF" )
   END_RUNG wire#w3
   RUNG wire#powerrail
      Contact( #Ap_ET100 )
   END_RUNG wire#w1
   RUNG wire#w1
      I_Contact( #HorquillasRecogidas )
   END_RUNG wire#w2
   // the same network as SCL:
   IF #EstadoZona.Rearme_CBx AND #HorquillasRecogidas AND #Pos_Dw THEN
       #EstadoMAQ.Err_Posicion := FALSE;   // RS flip-flop
   END_IF;
   IF (#Ap_ET100 AND NOT #HorquillasExtendidas AND NOT #HorquillasRecogidas) OR ((#EstadoMAQ.Etapa_Reset OR #Ap_ET100) AND (NOT #Pos_Dw OR NOT #HorquillasRecogidas) AND "OFF") THEN
       #EstadoMAQ.Err_Posicion := TRUE;
   END_IF;
   IF #EstadoMAQ.Err_Posicion THEN #EstadoMAQ.Error_MAQx := TRUE; END_IF;
END_REGION

REGION Network 52: TEMPORIZADOR - ESTABILIDAD para Fin de los Movimientos
